D6321 CHANNEL  ; 进料伺服Z轴JOG运行速度SV
D6322 CHANNEL  ; 进料伺服Z轴JOG运行速度SV
D6331 CHANNEL  ; 进料伺服Z轴JOG停止速度SV
D6332 CHANNEL  ; 进料伺服Z轴JOG停止速度SV
D634 CHANNEL  ; #2-2腔体自检保压时间（S_UInt）
D6350 CHANNEL  ; 进料伺服Z轴待料位SV
D6351 CHANNEL  ; 进料伺服Z轴待料位SV
D6352 CHANNEL  ; 进料伺服Z轴取料位SV
D6353 CHANNEL  ; 进料伺服Z轴取料位SV
D6354 CHANNEL  ; 进料伺服Z轴#1腔放料位SV
D6355 CHANNEL  ; 进料伺服Z轴#1腔放料位SV
D6356 CHANNEL  ; 进料伺服Z轴#2腔放料位SV
D6357 CHANNEL  ; 进料伺服Z轴#2腔放料位SV
D6358 CHANNEL  ; 进料伺服Z轴#3腔放料位SV
D6359 CHANNEL  ; 进料伺服Z轴#3腔放料位SV
D636 CHANNEL  ; #2-2腔体自检保压前真空（Pa_Float）
D6360 CHANNEL  ; 进料伺服Z轴#1夹爪扫码NG放料位SV
D6361 CHANNEL  ; 进料伺服Z轴#1夹爪扫码NG放料位SV
D6362 CHANNEL  ; 进料伺服Z轴#2夹爪扫码NG放料位SV
D6363 CHANNEL  ; 进料伺服Z轴#2夹爪扫码NG放料位SV
D6364 CHANNEL  ; 进料伺服Z轴#1夹爪配对取放料位SV
D6365 CHANNEL  ; 进料伺服Z轴#1夹爪配对取放料位SV
D6366 CHANNEL  ; 进料伺服Z轴#2夹爪配对取放料位SV
D6367 CHANNEL  ; 进料伺服Z轴#2夹爪配对取放料位SV
D638 CHANNEL  ; #2-2腔体自检保压后真空（Pa_Float）
D640 CHANNEL  ; #2-2腔体自检泄漏量（Pa_Float）
D6400 CHANNEL  ; 出料伺服X轴加速比率
D6401 CHANNEL  ; 出料伺服X轴减速比率
D6402 CHANNEL  ; 出料伺服X轴目标速度
D6403 CHANNEL  ; 出料伺服X轴目标速度
D6404 CHANNEL  ; 出料伺服X轴目标位置
D6405 CHANNEL  ; 出料伺服X轴目标位置
D6406 CHANNEL  ; 出料伺服X轴启动频率
D6407 CHANNEL  ; 出料伺服X轴启动频率
D6410 CHANNEL  ; 出料伺服X轴自动加速比率SV
D6411 CHANNEL  ; 出料伺服X轴自动减速比率SV
D6412 CHANNEL  ; 出料伺服X轴自动目标速度SV
D6414 CHANNEL  ; 出料伺服X轴自动目标位置
D6416 CHANNEL  ; 出料伺服X轴自动启动频率
D642 CHANNEL  ; #2-2腔体自检结果（1-OK，2-NG,3-抽真空NG）
D6420 CHANNEL  ; 出料伺服X轴JOG运行加减速
D6421 CHANNEL  ; 出料伺服X轴JOG运行速度
D6422 CHANNEL  ; 出料伺服X轴JOG运行速度
D6430 CHANNEL  ; 出料伺服X轴JOG停止加减速
D6431 CHANNEL  ; 出料伺服X轴JOG停止速度
D6432 CHANNEL  ; 出料伺服X轴JOG停止速度
D6440 CHANNEL  ; 出料伺服X轴当前位置
D6441 CHANNEL  ; 出料伺服X轴当前位置
D6442 CHANNEL  ; 出料伺服X轴当前速度
D6443 CHANNEL  ; 出料伺服X轴当前速度
D6450 CHANNEL  ; 下料Z模组当前位置（CAENNEL）
D6500 CHANNEL  ; 出料伺服X轴加速比率SV
D6501 CHANNEL  ; 出料伺服X轴减速比率SV
D6502 CHANNEL  ; 出料伺服X轴目标速度SV
D6503 CHANNEL  ; 出料伺服X轴目标速度SV
D6504 CHANNEL  ; 出料伺服X轴目标位置（CHANNEL)
D6506 CHANNEL  ; 出料伺服X轴启动频率SV
D6507 CHANNEL  ; 出料伺服X轴启动频率SV
D6520 CHANNEL  ; 出料伺服X轴JOG运行/停止加减速SV
D6521 CHANNEL  ; 出料伺服X轴JOG运行速度SV
D6522 CHANNEL  ; 出料伺服X轴JOG运行速度SV
D6530 CHANNEL  ; 出料伺服X轴JOG停止加减速
D6531 CHANNEL  ; 出料伺服X轴JOG停止速度SV
D6532 CHANNEL  ; 出料伺服X轴JOG停止速度SV
D6540 CHANNEL  ; 出料伺服X轴当前位置（CAENNEL）
D6542 CHANNEL  ; 出料伺服X轴当前速度
D6544 CHANNEL  ; 出料伺服X轴当前位置（REAL）（mm）
D6550 CHANNEL  ; 出料伺服X轴出料OK位（设定）
D6552 CHANNEL  ; 出料伺服X轴放料位SV
D6553 CHANNEL  ; 出料伺服X轴放料位SV
D6554 CHANNEL  ; 出料伺服X轴#1腔取料位SV
D6555 CHANNEL  ; 出料伺服X轴#1腔取料位SV
D6556 CHANNEL  ; 出料伺服X轴#2腔取料位SV
D6557 CHANNEL  ; 出料伺服X轴#2腔取料位SV
D6558 CHANNEL  ; 出料伺服X轴#3腔取料位SV
D6559 CHANNEL  ; 出料伺服X轴#3腔取料位SV
D6560 CHANNEL  ; 出料伺服X轴#1夹爪氦检NG放料位SV
D6561 CHANNEL  ; 出料伺服X轴#1夹爪氦检NG放料位SV
D6562 CHANNEL  ; 出料伺服X轴#2夹爪氦检NG放料位SV
D6563 CHANNEL  ; 出料伺服X轴#2夹爪氦检NG放料位SV
D6564 CHANNEL  ; 出料伺服X轴#1夹爪配对取放料位SV
D6565 CHANNEL  ; 出料伺服X轴#1夹爪配对取放料位SV
D6566 CHANNEL  ; 出料伺服X轴#2夹爪配对取放料位SV
D6567 CHANNEL  ; 出料伺服X轴#2夹爪配对取放料位SV
D66 CHANNEL  ; 设定条码长度
D660 CHANNEL  ; #2-2氦检时真空值（标漏）
D6600 CHANNEL  ; 出料伺服Z轴加速比率
D6601 CHANNEL  ; 出料伺服Z轴减速比率
D6602 CHANNEL  ; 出料伺服Z轴目标速度
D6603 CHANNEL  ; 出料伺服Z轴目标速度
D6604 CHANNEL  ; 出料伺服Z轴目标位置
D6605 CHANNEL  ; 出料伺服Z轴目标位置
D6606 CHANNEL  ; 出料伺服Z轴启动频率
D6607 CHANNEL  ; 出料伺服Z轴启动频率
D6610 CHANNEL  ; 出料伺服Z轴自动加速比率SV
D6611 CHANNEL  ; 出料伺服Z轴自动减速比率SV
D6612 CHANNEL  ; 出料伺服Z轴自动目标速度SV
D6614 CHANNEL  ; 出料伺服Z轴自动目标位置
D6616 CHANNEL  ; 出料伺服Z轴自动启动频率
D662 CHANNEL  ; #2-2氦检漏率（标漏）
D6620 CHANNEL  ; 出料伺服Z轴JOG运行加减速
D6621 CHANNEL  ; 出料伺服Z轴JOG运行速度
D6622 CHANNEL  ; 出料伺服Z轴JOG运行速度
D6630 CHANNEL  ; 出料伺服Z轴JOG停止加减速
D6631 CHANNEL  ; 出料伺服Z轴JOG停止速度
D6632 CHANNEL  ; 出料伺服Z轴JOG停止速度
D6640 CHANNEL  ; 出料伺服Z轴当前位置
D6641 CHANNEL  ; 出料伺服Z轴当前位置
D6642 CHANNEL  ; 出料伺服Z轴当前速度
D6643 CHANNEL  ; 出料伺服Z轴当前速度
D6650 CHANNEL  ; 出料伺服X轴出料OK位
D6654 CHANNEL  ; 出料伺服Z轴#1腔取料位SV1
D6655 CHANNEL  ; 出料伺服Z轴#1腔取料位SV1
D6656 CHANNEL  ; 出料伺服Z轴#2腔取料位SV1
D6657 CHANNEL  ; 出料伺服Z轴#2腔取料位SV1
D6658 CHANNEL  ; 出料伺服Z轴#3腔取料位SV1
D6659 CHANNEL  ; 出料伺服Z轴#3腔取料位SV1
D6700 CHANNEL  ; 出料伺服Z轴加速比率SV
D6701 CHANNEL  ; 出料伺服Z轴减速比率SV
D6702 CHANNEL  ; 出料伺服Z轴目标速度SV
D6703 CHANNEL  ; 出料伺服Z轴目标速度SV
D6704 CHANNEL  ; 出料伺服Z轴目标位置(CHANNEL）
D6706 CHANNEL  ; 出料伺服Z轴启动频率SV
D6707 CHANNEL  ; 出料伺服Z轴启动频率SV
D6720 CHANNEL  ; 出料伺服Z轴JOG运行/停止加减速SV
D6721 CHANNEL  ; 出料伺服Z轴JOG运行速度SV
D6722 CHANNEL  ; 出料伺服Z轴JOG运行速度SV
D6730 CHANNEL  ; 出料伺服Z轴JOG停止加减速
D6731 CHANNEL  ; 出料伺服Z轴JOG停止速度SV
D6732 CHANNEL  ; 出料伺服Z轴JOG停止速度SV
D6742 CHANNEL  ; 出料伺服Z轴当前速度
D6750 CHANNEL  ; 出料伺服Z轴待料位SV
D6751 CHANNEL  ; 出料伺服Z轴待料位SV
D6752 CHANNEL  ; 出料伺服Z轴放料位SV
D6753 CHANNEL  ; 出料伺服Z轴放料位SV
D6754 CHANNEL  ; 出料伺服Z轴#1腔取料位SV
D6755 CHANNEL  ; 出料伺服Z轴#1腔取料位SV
D6756 CHANNEL  ; 出料伺服Z轴#2腔取料位SV
D6757 CHANNEL  ; 出料伺服Z轴#2腔取料位SV
D6758 CHANNEL  ; 出料伺服Z轴#3腔取料位SV
D6759 CHANNEL  ; 出料伺服Z轴#3腔取料位SV
D6760 CHANNEL  ; 出料伺服Z轴#1夹爪氦检NG放料位SV
D6761 CHANNEL  ; 出料伺服Z轴#1夹爪氦检NG放料位SV
D6762 CHANNEL  ; 出料伺服Z轴#2夹爪氦检NG放料位SV
D6763 CHANNEL  ; 出料伺服Z轴#2夹爪氦检NG放料位SV
D6764 CHANNEL  ; 出料伺服Z轴#1夹爪配对取放料位SV
D6765 CHANNEL  ; 出料伺服Z轴#1夹爪配对取放料位SV
D6766 CHANNEL  ; 出料伺服Z轴#2夹爪配对取放料位SV
D6767 CHANNEL  ; 出料伺服Z轴#2夹爪配对取放料位SV
D68 CHANNEL  ; 设定条码字长度
D70 CHANNEL  ; 设定条码批次号
D700 CHANNEL  ; #3-2腔体状态（0停用，1待料中，2测试中，3测试完成，4-清氦中）
D702 CHANNEL  ; #3-2腔体测试漏率（Pa.m3/s_Float）
D704 CHANNEL  ; #3-2腔体测试检漏口压力（Pa_Float）
D706 CHANNEL  ; #3-2电池充氦压力（Pa_Float）
D708 CHANNEL  ; #3-2腔体测试结果（1 OK，2腔体泄漏，3气密NG，4注氦超时，5氦检异常，6电池泄漏，7注氦NG，8氦嘴泄漏）
D710 CHANNEL  ; #3-2充氦嘴压力（Pa_Float）
D712 CHANNEL  ; #3-2腔体抽气时间（S_UInt）
D714 CHANNEL  ; #3-2腔体真空压力（Pa_Float）
D716 CHANNEL  ; #3-2电池抽气时间（S_UInt）
D718 CHANNEL  ; #3-2电池真空压力（Pa_Float）
D730 CHANNEL  ; #3-2腔体自检抽气时间（S_UInt）
D732 CHANNEL  ; #3-2腔体自检前保压时间（S_UInt）
D734 CHANNEL  ; #3-2腔体自检保压时间（S_UInt）
D736 CHANNEL  ; #3-2腔体自检保压前真空（Pa_Float）
D738 CHANNEL  ; #3-2腔体自检保压后真空（Pa_Float）
D740 CHANNEL  ; #3-2腔体自检泄漏量（Pa_Float）
D742 CHANNEL  ; #3-2腔体自检结果（1-OK，2-NG,3-抽真空NG）
D760 CHANNEL  ; #3-2氦检时真空值（标漏）
D762 CHANNEL  ; #3-2氦检漏率（标漏）
D80 CHANNEL  ; 进料#1扫码接收条码长度
D900 CHANNEL  ; #1-1电池真空偏值设定(Float)
D902 CHANNEL  ; #1-1电池实际真空值(Float)
D904 CHANNEL  ; #1-1电池真空模拟量读数(Int)
D906 CHANNEL  ; #1-1电池设定时间实际真空值(Float)
D908 CHANNEL  ; #1-2电池设定时间实际真空值(Float)
D910 CHANNEL  ; #1-2电池真空偏值设定(Float)
D912 CHANNEL  ; #1-2电池实际真空值(Float)
D914 CHANNEL  ; #1-2电池真空模拟量读数(Int)
D920 CHANNEL  ; #2-1电池真空偏值设定(Float)
D922 CHANNEL  ; #2-1电池实际真空值(Float)
D924 CHANNEL  ; #2-1电池真空模拟量读数(Int)
D926 CHANNEL  ; #2-1电池设定时间实际真空值(Float)
D928 CHANNEL  ; #2-2电池设定时间实际真空值(Float)
D930 CHANNEL  ; #2-2电池真空偏值设定(Float)
D932 CHANNEL  ; #2-2电池实际真空值(Float)
D934 CHANNEL  ; #2-2电池真空模拟量读数(Int)
D940 CHANNEL  ; #3-1电池真空偏值设定(Float)
D942 CHANNEL  ; #3-1电池实际真空值(Float)
D944 CHANNEL  ; #3-1电池真空模拟量读数(Int)
D946 CHANNEL  ; #3-1电池设定时间实际真空值(Float)
D948 CHANNEL  ; #3-2电池设定时间实际真空值(Float)
D950 CHANNEL  ; #3-2电池真空偏值设定(Float)
D952 CHANNEL  ; #3-2电池实际真空值(Float)
D954 CHANNEL  ; #3-2电池真空模拟量读数(Int)
D962 CHANNEL  ; #1腔体实际真空值(Float)
D964 CHANNEL  ; #1腔体真空模拟量读数(Int)
D968 CHANNEL  ; #1腔体读设定时间实际真空值(Float)
D972 CHANNEL  ; #2腔体实际真空值(Float)
D974 CHANNEL  ; #2腔体真空模拟量读数(Int)
D978 CHANNEL  ; #2腔体读设定时间真空值
D982 CHANNEL  ; #3腔体实际真空值(Float)
D984 CHANNEL  ; #3腔体真空模拟量读数(Int)
D988 CHANNEL  ; #3腔体读设定时间实际真空值(Float)
D990 CHANNEL  ; 实时漏率（Pa.m3/s_Float）
D992 CHANNEL  ; 实时检漏口压力（Pa_Float）
D994 CHANNEL  ; 泄漏率设定值（Pa.m3/s_Float）
D996 CHANNEL  ; 检漏口压力设定值（Pa_Float）
D998 CHANNEL  ; 清氦漏率设定值（Pa_Float）
E0_0 CHANNEL  ; PC&PLC通讯心跳检测
E0_10 CHANNEL  ; 进料拉带机构#1扫码MES入站就绪通知
E0_1000 CHANNEL  ; 进料#1扫码MES出站读取条码开始字
E0_104 CHANNEL  ; 工艺参数变更通知to pc
E0_1049 CHANNEL  ; 进料#1扫码MES出站读取条码结束字
E0_105 CHANNEL  ; 工艺变更确认
E0_1050 CHANNEL  ; 出料伺服机构#1夹爪MES出站生产数据开始字
E0_1099 CHANNEL  ; 出料伺服机构#1夹爪MES出站生产数据结束字
E0_11 CHANNEL  ; 进料拉带机构#2扫码MES入站就绪通知
E0_1100 CHANNEL  ; 进料#2扫码MES入站读取条码开始字
E0_1149 CHANNEL  ; 进料#2扫码MES入站读取条码结束字
E0_1150 CHANNEL  ; 出料伺服机构#2夹爪MES出站生产数据开始字
E0_1199 CHANNEL  ; 出料伺服机构#2夹爪MES出站生产数据结束字
E0_1.00 BOOL  ; 设备上电状态
E0_1.01 BOOL  ; 设备复位状态
E0_1.02 BOOL  ; 设备自动状态
E0_1.03 BOOL  ; 设备停止状态
E0_1.04 BOOL  ; 设备启动状态
E0_1.05 BOOL  ; 设备待料状态
E0_1.06 BOOL  ; 设备手动状态
E0_1.07 BOOL  ; 设备故障状态
E0_1.08 BOOL  ; 设备急停状态
E0_1.09 BOOL  ; 设备关电状态
E0_20 CHANNEL  ; 进料拉带机构#1扫码MES入站就绪确认
E0_2000 CHANNEL  ; 进料#1扫码MES入站读取条码开始字
E0_2049 CHANNEL  ; 进料#1扫码MES入站读取条码结束字
E0_2050 CHANNEL  ; 进料#2扫码MES入站读取条码开始字
E0_2099 CHANNEL  ; 进料#2扫码MES入站读取条码结束字
E0_21 CHANNEL  ; 进料拉带机构#2扫码MES入站就绪确认
E0_300 CHANNEL  ; 泄漏率设定值to pc（Pa.m3/s_Float)to pc
E0_302 CHANNEL  ; 检漏口压力设定值（Pa_Float）to pc
E0_304 CHANNEL  ; 腔体测试设定氦检时间（S_UInt）to pc
E0_306 CHANNEL  ; 腔体测试设定真空阈值（Pa_Float）to pc
E0_308 CHANNEL  ; 电池测试设定真空阈值（Pa_Float）to pc
E0_310 CHANNEL  ; 电池测试设定#1-1注氦压力（Pa_Float）to pc
E0_312 CHANNEL  ; 电池测试设定#1-1注氦压力（Pa_Float）to pc
E0_316 CHANNEL  ; 腔体测试设定抽真空时间上限（S_UInt）to pc
E0_318 CHANNEL  ; 电池测试设定抽真空时间上限（S_UInt）to pc
E0_320 CHANNEL  ; 腔体测试设定腔体预抽检测时间（S_UInt）to pc
E0_322 CHANNEL  ; 电池测试设定预抽检测压力（Pa_Float）to pc
E0_324 CHANNEL  ; 腔体测试设定清氦压力（Pa_Float）to pc
E0_326 CHANNEL  ; 清氦漏率设定值（Pa_Float）to pc
E0_328 CHANNEL  ; 清氦漏率设定值（Pa_Float）to pc
E0_349 CHANNEL  ; 出料伺服机构#1夹爪MES出站工艺参数结束字
E0_350 CHANNEL  ; 出料伺服机构#2夹爪MES出站工艺参数开始字
E0_399 CHANNEL  ; 出料伺服机构#2夹爪MES出站工艺参数结束字
E0_50 CHANNEL  ; 出料伺服机构#1夹爪MES出站就绪通知
E0_51 CHANNEL  ; 出料伺服机构#2夹爪MES出站就绪通知
E0_60 CHANNEL  ; 出料伺服机构#1夹爪MES出站就绪确认
E0_61 CHANNEL  ; 出料伺服机构#2夹爪MES出站就绪确认
E0_900 CHANNEL  ; 工站故障
E2_1000 CHANNEL  ; 进料#1扫码条码开始字（传递）
E2_1001 CHANNEL  ; 进料#1扫码条码开始字（传递）
E2_1030 CHANNEL  ; 进料#1扫码条码结束字（传递）
E2_1100 CHANNEL  ; 进料#2扫码条码开始字（传递）
E2_1130 CHANNEL  ; 进料#2扫码条码结束字（传递）
E2_1200 CHANNEL  ; #1进料位条码开始字（传递）
E2_1299 CHANNEL  ; #1进料位数据结束字（传递）
E2_1300 CHANNEL  ; #2进料位条码开始字（传递）
E2_1399 CHANNEL  ; #2进料位数据结束字（传递）
E2_1400 CHANNEL  ; #1进料夹爪条码开始字（传递）
E2_1499 CHANNEL  ; #1进料夹爪数据结束字（传递）
E2_1500 CHANNEL  ; #2进料夹爪条码开始字（传递）
E2_1599 CHANNEL  ; #2进料夹爪数据结束字（传递）
E2_1600 CHANNEL  ; 扫码OK缓存条码开始字（传递）
E2_1699 CHANNEL  ; 扫码OK缓存数据结束字（传递）
E2_1800 CHANNEL  ; #1-1氦检腔条码开始字（传递）
E2_1850 CHANNEL  ; #1-1氦检腔工位开始字（传递）
E2_1899 CHANNEL  ; #1-1氦检腔数据结束字（传递）
E2_1900 CHANNEL  ; #1-2氦检腔条码开始字（传递）
E2_1950 CHANNEL  ; #1-2氦检腔工位开始字（传递）
E2_1999 CHANNEL  ; #1-2氦检腔数据结束字（传递）
E2_2000 CHANNEL  ; #2-1氦检腔条码开始字（传递）
E2_2050 CHANNEL  ; #2-1氦检腔工位开始字（传递）
E2_2099 CHANNEL  ; #2-1氦检腔数据结束字（传递）
E2_2100 CHANNEL  ; #2-2氦检腔条码开始字（传递）
E2_2150 CHANNEL  ; #2-2氦检腔工位开始字（传递）
E2_2199 CHANNEL  ; #2-2氦检腔数据结束字（传递）
E2_2200 CHANNEL  ; #3-1氦检腔条码开始字（传递）
E2_2250 CHANNEL  ; #3-1氦检腔工位开始字（传递）
E2_2299 CHANNEL  ; #3-1氦检腔数据结束字（传递）
E2_2300 CHANNEL  ; #3-2氦检腔条码开始字（传递）
E2_2350 CHANNEL  ; #3-2氦检腔工位开始字（传递）
E2_2399 CHANNEL  ; #3-2氦检腔数据结束字（传递）
E2_2400 CHANNEL  ; #1出料夹爪条码开始字（传递）
E2_2450 CHANNEL  ; #1出料夹爪工位开始字（传递）
E2_2499 CHANNEL  ; #1出料夹爪数据结束字（传递）
E2_2500 CHANNEL  ; #2出料夹爪条码开始字（传递）
E2_2550 CHANNEL  ; #2出料夹爪工位开始字（传递）
E2_2599 CHANNEL  ; #2出料夹爪数据结束字（传递）
H100.00 BOOL  ; #1扫码阻挡气缸缩回位屏蔽
H100.01 BOOL  ; #1扫码阻挡气缸伸出位屏蔽
H100.02 BOOL  ; #1隔离气缸缩回位屏蔽
H100.03 BOOL  ; 0屏蔽
H100.04 BOOL  ; #2扫码阻挡气缸缩回位屏蔽
H100.05 BOOL  ; #2扫码阻挡气缸伸出位屏蔽
H100.06 BOOL  ; #2隔离气缸缩回位屏蔽
H100.07 BOOL  ; 0屏蔽
H100.08 BOOL  ; #1进料夹爪夹紧位屏蔽
H100.09 BOOL  ; #1进料夹爪松开位屏蔽
H100.10 BOOL  ; #2进料夹爪夹紧位屏蔽
H100.11 BOOL  ; #2进料夹爪松开位屏蔽
H100.12 BOOL  ; 进料夹爪变距气缸伸出位屏蔽
H100.13 BOOL  ; 进料夹爪变距气缸缩回位屏蔽
H100.14 BOOL  ; #1出料夹爪夹紧位屏蔽
H100.15 BOOL  ; #1出料夹爪松开位屏蔽
H101.00 BOOL  ; #2出料夹爪夹紧位屏蔽
H101.01 BOOL  ; #2出料夹爪松开位屏蔽
H101.02 BOOL  ; 出料夹爪变距气缸伸出位屏蔽
H101.03 BOOL  ; 出料夹爪变距气缸缩回位屏蔽
H101.04 BOOL  ; #1腔体平移一级气缸缩回位屏蔽
H101.05 BOOL  ; #1腔体平移一级气缸伸出位屏蔽
H101.06 BOOL  ; #1腔体平移二级气缸缩回位屏蔽
H101.07 BOOL  ; #1腔体平移二级气缸伸出位屏蔽
H101.08 BOOL  ; #1腔体顶伸气缸上升位屏蔽
H101.09 BOOL  ; #1腔体顶伸气缸下降位屏蔽
H101.10 BOOL  ; #1腔体氦检阀开到位屏蔽
H101.11 BOOL  ; #1腔体氦检阀关到位屏蔽
H101.12 BOOL  ; 0屏蔽
H101.13 BOOL  ; 0屏蔽
H101.14 BOOL  ; 0屏蔽
H101.15 BOOL  ; 0屏蔽
H102.00 BOOL  ; 0屏蔽
H102.01 BOOL  ; #2腔体平移一级气缸缩回位屏蔽
H102.02 BOOL  ; #2腔体平移一级气缸伸出位屏蔽
H102.03 BOOL  ; #2腔体平移二级气缸缩回位屏蔽
H102.04 BOOL  ; #2腔体平移二级气缸伸出位屏蔽
H102.05 BOOL  ; #2腔体顶伸气缸上升位屏蔽
H102.06 BOOL  ; #2腔体顶伸气缸下降位屏蔽
H102.07 BOOL  ; #2腔体氦检阀开到位屏蔽
H102.08 BOOL  ; #2腔体氦检阀关到位屏蔽
H102.09 BOOL  ; 0屏蔽
H102.10 BOOL  ; 0屏蔽
H102.11 BOOL  ; 0屏蔽
H102.12 BOOL  ; 0屏蔽
H102.13 BOOL  ; 0屏蔽
H102.14 BOOL  ; #3腔体平移一级气缸缩回位屏蔽
H102.15 BOOL  ; #3腔体平移一级气缸伸出位屏蔽
H103.00 BOOL  ; #3腔体平移二级气缸缩回位屏蔽
H103.01 BOOL  ; #3腔体平移二级气缸伸出位屏蔽
H103.02 BOOL  ; #3腔体顶伸气缸上升位屏蔽
H103.03 BOOL  ; #3腔体顶伸气缸下降位屏蔽
H103.04 BOOL  ; #3腔体氦检阀开到位屏蔽
H103.05 BOOL  ; #3腔体氦检阀关到位屏蔽
H103.06 BOOL  ; 氦检仪准备好了信号屏蔽
H103.07 BOOL  ; 氦检仪故障信号屏蔽
H103.08 BOOL  ; 0屏蔽
H103.09 BOOL  ; 0屏蔽
H103.10 BOOL  ; 0屏蔽
H103.11 BOOL  ; 进料伺服X轴准备好了信号屏蔽
H103.12 BOOL  ; 进料伺服X轴故障信号屏蔽
H103.13 BOOL  ; 进料伺服Z轴准备好了信号屏蔽
H103.14 BOOL  ; 进料伺服Z轴故障信号屏蔽
H103.15 BOOL  ; 0屏蔽
H104.00 BOOL  ; 出料伺服X轴准备好了信号屏蔽
H104.01 BOOL  ; 出料伺服X轴故障信号屏蔽
H104.02 BOOL  ; 出料伺服Z轴准备好了信号屏蔽
H104.03 BOOL  ; 出料伺服Z轴故障信号屏蔽
H104.04 BOOL  ; 0屏蔽
H104.05 BOOL  ; 腔体抽真空泵运行信号屏蔽
H104.06 BOOL  ; 腔体抽真空泵过载信号屏蔽
H104.07 BOOL  ; 氦检前置泵运行信号屏蔽
H104.08 BOOL  ; 氦检前置泵过载信号屏蔽
H104.09 BOOL  ; 启动按钮屏蔽
H104.10 BOOL  ; 停止按钮屏蔽
H104.11 BOOL  ; 复位按钮屏蔽
H104.12 BOOL  ; 急停按钮屏蔽
H104.13 BOOL  ; 手自动选择屏蔽
H104.14 BOOL  ; #1进料夹爪防下坠感应屏蔽
H104.15 BOOL  ; #2进料夹爪防下坠感应屏蔽
H105.00 BOOL  ; #1出料夹爪防下坠感应屏蔽
H105.01 BOOL  ; #2出料夹爪防下坠感应屏蔽
H105.02 BOOL  ; 0屏蔽
H105.03 BOOL  ; 进料对接输入屏蔽
H105.04 BOOL  ; 出料对接输入屏蔽
H105.05 BOOL  ; 0屏蔽
H105.06 BOOL  ; 0屏蔽
H105.07 BOOL  ; 设备总气压信号屏蔽
H105.08 BOOL  ; #1来料位有料感应屏蔽
H105.09 BOOL  ; #2来料位有料感应屏蔽
H105.10 BOOL  ; #1隔离位有料感应屏蔽
H105.11 BOOL  ; #2隔离位有料感应屏蔽
H105.12 BOOL  ; #1扫码位有料感应屏蔽
H105.13 BOOL  ; #2扫码位有料感应屏蔽
H105.14 BOOL  ; #1-1进料位有料感应屏蔽
H105.15 BOOL  ; #1-2进料位有料感应屏蔽
H106.00 BOOL  ; #2-1进料位有料感应屏蔽
H106.01 BOOL  ; #2-2进料位有料感应屏蔽
H106.02 BOOL  ; 进料夹爪柔性感应屏蔽
H106.03 BOOL  ; 出料夹爪柔性感应屏蔽
H106.04 BOOL  ; #1进料夹爪对应腔体有料感应屏蔽
H106.05 BOOL  ; #2进料夹爪对应腔体有料感应屏蔽
H106.06 BOOL  ; 扫码NG放料#1位有料感应屏蔽
H106.07 BOOL  ; 扫码NG放料#2位有料感应屏蔽
H106.08 BOOL  ; 扫码NG料满位有料感应屏蔽
H106.09 BOOL  ; 进料配对位有料感应屏蔽
H106.10 BOOL  ; 出料配对位有料感应屏蔽
H106.11 BOOL  ; 氦检NG放料#1位有料感应屏蔽
H106.12 BOOL  ; 氦检NG放料#2位有料感应屏蔽
H106.13 BOOL  ; 氦检NG料满位有料感应屏蔽
H106.14 BOOL  ; #1-1出料位有料感应屏蔽
H106.15 BOOL  ; #1-2出料位有料感应屏蔽
H107.00 BOOL  ; #2-1出料位有料感应屏蔽
H107.01 BOOL  ; #2-2出料位有料感应屏蔽
H107.02 BOOL  ; #1门磁开关屏蔽
H107.03 BOOL  ; #2门磁开关屏蔽
H107.04 BOOL  ; #3门磁开关屏蔽
H107.05 BOOL  ; #4门磁开关屏蔽
H107.06 BOOL  ; #5门磁开关屏蔽
H107.07 BOOL  ; #6门磁开关屏蔽
H107.08 BOOL  ; #7门磁开关屏蔽
H107.09 BOOL  ; #8门磁开关屏蔽
H107.10 BOOL  ; #9门磁开关屏蔽
H107.11 BOOL  ; #10门磁开关屏蔽
H107.12 BOOL  ; #11门磁开关屏蔽
H107.13 BOOL  ; 设备真空压力信号屏蔽
H107.14 BOOL  ; 设备氦气压力信号屏蔽
H107.15 BOOL  ; 精密调压阀信号屏蔽
H10.00 BOOL  ; #1扫码阻挡有料记忆
H10.01 BOOL  ; #1进料位有料记忆
H10.02 BOOL  ; #1进料位有OK料记忆
H10.03 BOOL  ; #1进料位有NG料记忆
H10.04 BOOL  ; #1扫码阻挡有OK料记忆
H10.05 BOOL  ; #1扫码阻挡有NG料记忆
H10.06 BOOL  ; #1扫码阻挡扫码完成记忆
H10.07 BOOL  ; #1扫码阻挡扫码OK料记忆
H10.08 BOOL  ; #1扫码阻挡扫码NG料记忆
H10.09 BOOL  ; #1扫码阻挡MES校验完成记忆
H10.10 BOOL  ; #1扫码阻挡MES校验OK料记忆
H10.11 BOOL  ; #1扫码阻挡MES校验NG料记忆
H11.00 BOOL  ; #1隔离气缸放料中记忆
H11.01 BOOL  ; #1扫码阻挡气缸放料中记忆
H12.00 BOOL  ; #2扫码阻挡有料记忆
H12.01 BOOL  ; #2进料位有料记忆
H12.02 BOOL  ; #2进料位有OK料记忆
H12.03 BOOL  ; #2进料位有NG料记忆
H12.04 BOOL  ; #2扫码阻挡有OK料记忆
H12.05 BOOL  ; #2扫码阻挡有NG料记忆
H12.06 BOOL  ; #2扫码阻挡扫码完成记忆
H12.07 BOOL  ; #2扫码阻挡扫码OK料记忆
H12.08 BOOL  ; #2扫码阻挡扫码NG料记忆
H12.09 BOOL  ; #2扫码阻挡MES校验完成记忆
H12.10 BOOL  ; #2扫码阻挡MES校验OK料记忆
H12.11 BOOL  ; #2扫码阻挡MES校验NG料记忆
H13.00 BOOL  ; #2隔离气缸放料中记忆
H13.01 BOOL  ; #2扫码阻挡气缸放料中记忆
H15.00 BOOL  ; 扫码NG放料位有料记忆
H17.00 BOOL  ; 氦检NG放料位有料记忆
H20.00 BOOL  ; #1进料夹爪有料记忆
H20.01 BOOL  ; #2进料夹爪有料记忆
H20.02 BOOL  ; 进料配对位有料记忆
H20.03 BOOL  ; #1进料夹爪有OK料记忆
H20.04 BOOL  ; #1进料夹爪有NG料记忆
H20.05 BOOL  ; #2进料夹爪有OK料记忆
H20.06 BOOL  ; #2进料夹爪有NG料记忆
H24.00 BOOL  ; 进料伺服X轴回原点记忆
H24.01 BOOL  ; 进料伺服Z轴回原点记Z忆
H24.02 BOOL  ; 出料伺服X轴回原点记忆
H24.03 BOOL  ; 出料伺服Z轴回原点记忆
H25.00 BOOL  ; #1-1腔体有料记忆
H25.01 BOOL  ; #1-2腔体有料记忆
H25.02 BOOL  ; #1-1腔体有OK料记忆
H25.03 BOOL  ; #1-1腔体有NG料记忆
H25.04 BOOL  ; #1-2腔体有OK料记忆
H25.05 BOOL  ; #1-2腔体有NG料记忆
H25.06 BOOL  ; #1-1腔体测试完成记忆
H25.07 BOOL  ; #1-2腔体测试完成记忆
H26.00 BOOL  ; #1-1电池泄漏
H26.01 BOOL  ; #1-2电池泄漏
H26.02 BOOL  ; #1-1电池注氦超时
H26.03 BOOL  ; #1-2电池注氦超时
H26.04 BOOL  ; #1-1腔体抽真空NG
H26.05 BOOL  ; #1-2腔体抽真空NG
H26.06 BOOL  ; #1-1腔体氦检时腔体压力过高
H26.07 BOOL  ; #1-2腔体氦检时腔体压力过高
H27.00 BOOL  ; #1腔体有清氦需求
H27.05 BOOL  ; 腔体有复测需求
H27.10 BOOL  ; #1-1腔体清氦失败，重新进行清氦流程
H30.00 BOOL  ; #2-1腔体有料记忆
H30.01 BOOL  ; #2-2腔体有料记忆
H30.02 BOOL  ; #2-1腔体有OK料记忆
H30.03 BOOL  ; #2-1腔体有NG料记忆
H30.04 BOOL  ; #2-2腔体有OK料记忆
H30.05 BOOL  ; #2-2腔体有NG料记忆
H30.06 BOOL  ; #2-1腔体测试完成记忆
H30.07 BOOL  ; #2-2腔体测试完成记忆
H31.00 BOOL  ; #2-1电池泄漏
H31.01 BOOL  ; #2-2电池泄漏
H31.02 BOOL  ; #2-1电池注氦超时
H31.03 BOOL  ; #2-2电池注氦超时
H31.04 BOOL  ; #2-1腔体抽真空NG
H31.05 BOOL  ; #2-2腔体抽真空NG
H31.06 BOOL  ; #2-1腔体氦检时腔体压力过高
H31.07 BOOL  ; #2-2腔体氦检时腔体压力过高
H32.00 BOOL  ; #2腔体有清氦需求
H32.05 BOOL  ; 腔体有复测需求
H32.10 BOOL  ; #2-1腔体清氦失败，重新进行清氦流程
H35.00 BOOL  ; #3-1腔体有料记忆
H35.01 BOOL  ; #3-2腔体有料记忆
H35.02 BOOL  ; #3-1腔体有OK料记忆
H35.03 BOOL  ; #3-1腔体有NG料记忆
H35.04 BOOL  ; #3-2腔体有OK料记忆
H35.05 BOOL  ; #3-2腔体有NG料记忆
H35.06 BOOL  ; #3-1腔体测试完成记忆
H35.07 BOOL  ; #3-2腔体测试完成记忆
H36.00 BOOL  ; #3-1电池泄漏
H36.01 BOOL  ; #3-2电池泄漏
H36.02 BOOL  ; #3-1电池注氦超时
H36.03 BOOL  ; #3-2电池注氦超时
H36.04 BOOL  ; #3-1腔体抽真空NG
H36.05 BOOL  ; #3-2腔体抽真空NG
H36.06 BOOL  ; #3-1腔体氦检时腔体压力过高
H36.07 BOOL  ; #3-2腔体氦检时腔体压力过高
H37.00 BOOL  ; #3腔体有清氦需求
H37.05 BOOL  ; 腔体有复测需求
H37.10 BOOL  ; #3-1腔体清氦失败，重新进行清氦流程
H40.00 BOOL  ; #1出料夹爪有料记忆
H40.01 BOOL  ; #2出料夹爪有料记忆
H40.02 BOOL  ; 出料配对位有料记忆
H40.03 BOOL  ; #1出料夹爪有OK料记忆
H40.04 BOOL  ; #1出料夹爪有NG料记忆
H40.05 BOOL  ; #2出料夹爪有OK料记忆
H40.06 BOOL  ; #2出料夹爪有NG料记忆
H40.07 BOOL  ; #1出料夹爪MES校验完成记忆
H40.08 BOOL  ; #2出料夹爪MES校验完成记忆
H40.15 BOOL  ; 出料变距缩回记忆
H41.00 BOOL  ; 1#取料完成
H41.01 BOOL  ; 2#取料完成
H41.02 BOOL  ; 3#取料完成
H41.03 BOOL  ; 1#放NG，2#放缓存
H41.04 BOOL  ; 1#放NG，1#取缓存
H41.05 BOOL  ; 2#放NG,1#放缓存
H41.06 BOOL  ; 2#放NG,2#取缓存
H43.00 BOOL  ; 1#腔体下料需求
H43.01 BOOL  ; 2#腔体下料需求
H43.02 BOOL  ; 3#腔体下料需求
H44.00 BOOL  ; 出料伺服X轴回原点记忆
H44.01 BOOL  ; 出料伺服Z轴回原点记忆
H5.00 BOOL  ; 扫码屏蔽（SW）
H5.01 BOOL  ; 进料拉带重新扫码模式选择（0=使用/1=屏蔽）
H5.02 BOOL  ; 氦检仪屏蔽
H5.03 BOOL  ; 1#腔体屏蔽（0=使用）
H5.04 BOOL  ; 2#腔体屏蔽（0=使用）
H5.05 BOOL  ; 3#腔体屏蔽（0=使用）
H5.07 BOOL  ; 电脑屏蔽-HMI
H5.08 BOOL  ; 门磁屏蔽(1-屏蔽)
H5.09 BOOL  ; 出料机械手放完NG料后回待料位（1-停用）
H5.10 BOOL  ; 空跑程序
H5.12 BOOL  ; 氦气源压力检测屏蔽
H5.13 BOOL  ; 复测模式（0-关闭 1-打开）
H5.14 BOOL  ; 测试模式（0-双检 1-单检）
H5.15 BOOL  ; 腔体模式（0-正压 1-负压）
H6.00 BOOL  ; 清氦模式（0-使用 1-不使用）
H6.01 BOOL  ; 氦气回收机使用（1-使用）
H6.06 BOOL  ; 出站MES校验使用（1-使用）
T0000 BOOL  ; PLC上电延时100ms
T0001 BOOL  ; 手动模式延时
T0002 BOOL  ; 自动模式延时
T0006 BOOL  ; 复位延时
T0007 BOOL  ; 自动停止完成延时
T0008 BOOL  ; 启动按钮按下1s延时
T0009 BOOL  ; 停止按钮按下延时
T0015 BOOL  ; 扫码NG取料延时
T0016 BOOL  ; 检测NG料满取料延时
T0019 BOOL  ; 清料停止完成延时
T0020 BOOL  ; 设备待料状态延时（参考进料）
T0021 BOOL  ; 设备待料状态延时（参考出料）
T0022 BOOL  ; 蜂鸣器屏蔽时间
T0024 BOOL  ; 氦检仪真空阀打开安全判定延时
T0030 BOOL  ; 腔体真空泵停机1分钟内禁止启动保护延时
T0031 BOOL  ; 氦检前置泵泵停机1分钟内禁止启动保护延时
T0045 BOOL  ; 进料#1扫码枪通信异常
T0046 BOOL  ; 进料#2扫码枪通信异常
T0047 BOOL  ; 氦检仪通信异常
T0048 BOOL  ; 氦检仪启动异常
T0049 BOOL  ; 初次上电氦检仪故障延时
T0050 BOOL  ; PC&PLC通讯心跳检测异常延时
T0062 BOOL  ; 进料伺服X轴故障报警延时
T0063 BOOL  ; 进料伺服Z轴故障报警延时
T0072 BOOL  ; 出料伺服X轴故障报警延时
T0073 BOOL  ; 出料伺服Z轴故障报警延时
T0075 BOOL  ; 1#腔体读真空设定时间
T0076 BOOL  ; 1-1电池读真空设定时间
T0077 BOOL  ; 1-2电池读真空设定时间
T0078 BOOL  ; 2#腔体读真空设定时间
T0079 BOOL  ; 2-1电池读真空设定时间
T0080 BOOL  ; 2-2电池读真空设定时间
T0081 BOOL  ; 3#腔体读真空设定时间
T0082 BOOL  ; 3-1电池读真空设定时间
T0083 BOOL  ; 3-2电池读真空设定时间
T0100 BOOL  ; #1扫码阻挡气缸缩回位报警延时
T0101 BOOL  ; #1扫码阻挡气缸伸出位报警延时
T0102 BOOL  ; #1隔离气缸缩回位报警延时
T0103 BOOL  ; 0报警延时
T0104 BOOL  ; #2扫码阻挡气缸缩回位报警延时
T0105 BOOL  ; #2扫码阻挡气缸伸出位报警延时
T0106 BOOL  ; #2隔离气缸缩回位报警延时
T0107 BOOL  ; 0报警延时
T0108 BOOL  ; #1进料夹爪夹紧位报警延时
T0109 BOOL  ; #1进料夹爪松开位报警延时
T0110 BOOL  ; #2进料夹爪夹紧位报警延时
T0111 BOOL  ; #2进料夹爪松开位报警延时
T0112 BOOL  ; 进料夹爪变距气缸伸出位报警延时
T0113 BOOL  ; 进料夹爪变距气缸缩回位报警延时
T0114 BOOL  ; #1出料夹爪夹紧位报警延时
T0115 BOOL  ; #1出料夹爪松开位报警延时
T0116 BOOL  ; #2出料夹爪夹紧位报警延时
T0117 BOOL  ; #2出料夹爪松开位报警延时
T0118 BOOL  ; 出料夹爪变距气缸伸出位报警延时
T0119 BOOL  ; 出料夹爪变距气缸缩回位报警延时
T0120 BOOL  ; #1腔体平移一级气缸缩回位报警延时
T0121 BOOL  ; #1腔体平移一级气缸伸出位报警延时
T0122 BOOL  ; #1腔体平移二级气缸缩回位报警延时
T0123 BOOL  ; #1腔体平移二级气缸伸出位报警延时
T0124 BOOL  ; #1腔体顶伸气缸上升位报警延时
T0125 BOOL  ; #1腔体顶伸气缸下降位报警延时
T0126 BOOL  ; #1腔体氦检阀开到位报警延时
T0127 BOOL  ; #1腔体氦检阀关到位报警延时
T0128 BOOL  ; 0报警延时
T0129 BOOL  ; 0报警延时
T0130 BOOL  ; 0报警延时
T0131 BOOL  ; 0报警延时
T0132 BOOL  ; 0报警延时
T0133 BOOL  ; #2腔体平移一级气缸缩回位报警延时
T0134 BOOL  ; #2腔体平移一级气缸伸出位报警延时
T0135 BOOL  ; #2腔体平移二级气缸缩回位报警延时
T0136 BOOL  ; #2腔体平移二级气缸伸出位报警延时
T0137 BOOL  ; #2腔体顶伸气缸上升位报警延时
T0138 BOOL  ; #2腔体顶伸气缸下降位报警延时
T0139 BOOL  ; #2腔体氦检阀开到位报警延时
T0140 BOOL  ; #2腔体氦检阀关到位报警延时
T0141 BOOL  ; 0报警延时
T0142 BOOL  ; 0报警延时
T0143 BOOL  ; 0报警延时
T0144 BOOL  ; 0报警延时
T0145 BOOL  ; 0报警延时
T0146 BOOL  ; #3腔体平移一级气缸缩回位报警延时
T0147 BOOL  ; #3腔体平移一级气缸伸出位报警延时
T0148 BOOL  ; #3腔体平移二级气缸缩回位报警延时
T0149 BOOL  ; #3腔体平移二级气缸伸出位报警延时
T0150 BOOL  ; #3腔体顶伸气缸上升位报警延时
T0151 BOOL  ; #3腔体顶伸气缸下降位报警延时
T0152 BOOL  ; #3腔体氦检阀开到位报警延时
T0153 BOOL  ; #3腔体氦检阀关到位报警延时
T0154 BOOL  ; 氦检仪准备好了信号报警延时
T0155 BOOL  ; 氦检仪故障信号报警延时
T0156 BOOL  ; 0报警延时
T0157 BOOL  ; 0报警延时
T0158 BOOL  ; 0报警延时
T0159 BOOL  ; 进料伺服X轴准备好了信号报警延时
T0160 BOOL  ; 进料伺服X轴故障信号报警延时
T0161 BOOL  ; 进料伺服Z轴准备好了信号报警延时
T0162 BOOL  ; 进料伺服Z轴故障信号报警延时
T0163 BOOL  ; 0报警延时
T0164 BOOL  ; 出料伺服X轴准备好了信号报警延时
T0165 BOOL  ; 出料伺服X轴故障信号报警延时
T0166 BOOL  ; 出料伺服Z轴准备好了信号报警延时
T0167 BOOL  ; 出料伺服Z轴故障信号报警延时
T0168 BOOL  ; 0报警延时
T0169 BOOL  ; 腔体抽真空泵运行信号报警延时
T0170 BOOL  ; 腔体抽真空泵过载信号报警延时
T0171 BOOL  ; 氦检前置泵运行信号报警延时
T0172 BOOL  ; 氦检前置泵过载信号报警延时
T0173 BOOL  ; 启动按钮报警延时
T0174 BOOL  ; 停止按钮报警延时
T0175 BOOL  ; 复位按钮报警延时
T0176 BOOL  ; 急停按钮报警延时
T0177 BOOL  ; 手自动选择报警延时
T0178 BOOL  ; #1进料夹爪防下坠感应报警延时
T0179 BOOL  ; #2进料夹爪防下坠感应报警延时
T0180 BOOL  ; #1出料夹爪防下坠感应报警延时
T0181 BOOL  ; #2出料夹爪防下坠感应报警延时
T0182 BOOL  ; 0报警延时
T0183 BOOL  ; 进料对接输入报警延时
T0184 BOOL  ; 出料对接输入报警延时
T0185 BOOL  ; 0报警延时
T0186 BOOL  ; 0报警延时
T0187 BOOL  ; 设备总气压信号报警延时
T0188 BOOL  ; #1来料位有料感应报警延时
T0189 BOOL  ; #2来料位有料感应报警延时
T0190 BOOL  ; #1隔离位有料感应报警延时
T0191 BOOL  ; #2隔离位有料感应报警延时
T0192 BOOL  ; #1扫码位有料感应报警延时
T0193 BOOL  ; #2扫码位有料感应报警延时
T0194 BOOL  ; #1-1进料位有料感应报警延时
T0195 BOOL  ; #1-2进料位有料感应报警延时
T0196 BOOL  ; #2-1进料位有料感应报警延时
T0197 BOOL  ; #2-2进料位有料感应报警延时
T0198 BOOL  ; 进料夹爪柔性感应报警延时
T0199 BOOL  ; 出料夹爪柔性感应报警延时
T0200 BOOL  ; #1进料夹爪对应腔体有料感应报警延时
T0201 BOOL  ; #2进料夹爪对应腔体有料感应报警延时
T0202 BOOL  ; 扫码NG放料#1位有料感应报警延时
T0203 BOOL  ; 扫码NG放料#2位有料感应报警延时
T0204 BOOL  ; 扫码NG料满位有料感应报警延时
T0205 BOOL  ; 进料配对位有料感应报警延时
T0206 BOOL  ; 出料配对位有料感应报警延时
T0207 BOOL  ; 氦检NG放料#1位有料感应报警延时
T0208 BOOL  ; 氦检NG放料#2位有料感应报警延时
T0209 BOOL  ; 氦检NG料满位有料感应报警延时
T0210 BOOL  ; #1-1出料位有料感应报警延时
T0211 BOOL  ; #1-2出料位有料感应报警延时
T0212 BOOL  ; #2-1出料位有料感应报警延时
T0213 BOOL  ; #2-2出料位有料感应报警延时
T0214 BOOL  ; #1门磁开关报警延时
T0215 BOOL  ; #2门磁开关报警延时
T0216 BOOL  ; #3门磁开关报警延时
T0217 BOOL  ; #4门磁开关报警延时
T0218 BOOL  ; #5门磁开关报警延时
T0219 BOOL  ; #6门磁开关报警延时
T0220 BOOL  ; #7门磁开关报警延时
T0221 BOOL  ; #8门磁开关报警延时
T0222 BOOL  ; #9门磁开关报警延时
T0223 BOOL  ; #10门磁开关报警延时
T0224 BOOL  ; #11门磁开关报警延时
T0225 BOOL  ; 设备真空压力信号报警延时
T0226 BOOL  ; 设备氦气压力信号报警延时
T0227 BOOL  ; 精密调压阀信号报警延时
T0280 BOOL  ; 进料扫码MES入站就绪通知&确认超时报警延时
T0281 BOOL  ; 出料伺服MES出站就绪通知&确认超时报警延时
T0308 BOOL  ; 进料伺服X轴正极限报警延时
T0309 BOOL  ; 进料伺服X轴负极限报警延时
T0310 BOOL  ; 进料伺服X轴原点报警延时
T0311 BOOL  ; 进料伺服Z轴正极限报警延时
T0312 BOOL  ; 进料伺服Z轴负极限报警延时
T0313 BOOL  ; 进料伺服Z轴原点报警延时
T0314 BOOL  ; 出料伺服X轴正极限报警延时
T0315 BOOL  ; 出料伺服X轴负极限报警延时
T0316 BOOL  ; 出料伺服X轴原点报警延时
T0317 BOOL  ; 出料伺服Z轴正极限报警延时
T0318 BOOL  ; 出料伺服Z轴负极限报警延时
T0319 BOOL  ; 出料伺服Z轴原点报警延时
T0324 BOOL  ; 氦检仪不在检漏状态[alm]
T0356 BOOL  ; #1来料位有料记忆报警延时
T0357 BOOL  ; #2来料位有料记忆报警延时
T0358 BOOL  ; #1隔离位有料记忆报警延时
T0359 BOOL  ; #2隔离位有料记忆报警延时
T0360 BOOL  ; #1扫码位有料记忆报警延时
T0361 BOOL  ; #2扫码位有料记忆报警延时
T0362 BOOL  ; #1进料位有料记忆报警延时
T0363 BOOL  ; #2进料位有料记忆报警延时
T0364 BOOL  ; #1进料夹爪有料记忆报警延时
T0365 BOOL  ; #2进料夹爪有料记忆报警延时
T0366 BOOL  ; #1出料夹爪有料记忆报警延时
T0367 BOOL  ; #2出料夹爪有料记忆报警延时
T0368 BOOL  ; #1-1腔体有料记忆报警延时
T0369 BOOL  ; #1-2腔体有料记忆报警延时
T0370 BOOL  ; #2-1腔体有料记忆报警延时
T0371 BOOL  ; #2-2腔体有料记忆报警延时
T0372 BOOL  ; #3-1腔体有料记忆报警延时
T0373 BOOL  ; #3-2腔体有料记忆报警延时
T0374 BOOL  ; 进料配对位有料记忆报警延时
T0375 BOOL  ; 出料配对位有料记忆报警延时
T0376 BOOL  ; #1出料位有料记忆报警延时
T0377 BOOL  ; #2出料位有料记忆报警延时
T0378 BOOL  ; 扫码NG放料位有料记忆报警延时
T0379 BOOL  ; 氦检NG拉带下料位有料记忆报警延时
T0388 BOOL  ; 整机复位超时报警延时
T0389 BOOL  ; 进料拉带工站复位超时报警延时
T0390 BOOL  ; 进料伺服工站复位超时报警延时
T0391 BOOL  ; #1氦检工站复位超时报警延时
T0392 BOOL  ; #2氦检工站复位超时报警延时
T0393 BOOL  ; #3氦检工站复位超时报警延时
T0394 BOOL  ; 出料伺服工站复位超时报警延时
T0400 BOOL  ; 开#1电池破真空法条件
T0401 BOOL  ; 开#2电池破真空法条件
T0402 BOOL  ; 开#3电池破真空法条件
T0500 BOOL  ; #1扫码阻挡气缸缩回延时[A]
T0501 BOOL  ; #1扫码阻挡气缸伸出延时[A]
T0502 BOOL  ; #1隔离气缸缩回延时[A]
T0503 BOOL  ; #1隔离气缸伸出延时[A]
T0504 BOOL  ; #2扫码阻挡气缸缩回延时[A]
T0505 BOOL  ; #2扫码阻挡气缸伸出延时[A]
T0506 BOOL  ; #2隔离气缸缩回延时[A]
T0507 BOOL  ; #2隔离气缸伸出延时[A]
T0508 BOOL  ; #1进料夹爪夹紧延时[A]
T0509 BOOL  ; #1进料夹爪松开延时[A]
T0510 BOOL  ; #2进料夹爪夹紧延时[A]
T0511 BOOL  ; #2进料夹爪松开延时[A]
T0512 BOOL  ; 进料夹爪变距气缸伸出延时[A]
T0513 BOOL  ; 进料夹爪变距气缸缩回延时[A]
T0514 BOOL  ; #1出料夹爪夹紧延时[A]
T0515 BOOL  ; #1出料夹爪松开延时[A]
T0516 BOOL  ; #2出料夹爪夹紧延时[A]
T0517 BOOL  ; #2出料夹爪松开延时[A]
T0518 BOOL  ; 出料夹爪变距气缸伸出延时[A]
T0519 BOOL  ; 出料夹爪变距气缸缩回延时[A]
T0520 BOOL  ; #1腔体平移一级气缸缩回延时[A]
T0521 BOOL  ; #1腔体平移一级气缸伸出延时[A]
T0522 BOOL  ; #1腔体平移二级气缸缩回延时[A]
T0523 BOOL  ; #1腔体平移二级气缸伸出延时[A]
T0524 BOOL  ; #1腔体顶伸气缸上升延时[A]
T0525 BOOL  ; #1腔体顶伸气缸下降延时[A]
T0526 BOOL  ; #1腔体氦检阀开延时[A]
T0527 BOOL  ; 氦检仪真空阀开延时[A]
T0528 BOOL  ; #1腔体抽真空阀开延时[A]
T0529 BOOL  ; #1-1腔体阀开延时[A]
T0530 BOOL  ; #1-2腔体阀开延时[A]
T0531 BOOL  ; #1腔体破真空阀开延时[A]
T0532 BOOL  ; #1腔体吹气阀开延时[A]
T0533 BOOL  ; #2腔体平移一级气缸缩回延时[A]
T0534 BOOL  ; #2腔体平移一级气缸伸出延时[A]
T0535 BOOL  ; #2腔体平移二级气缸缩回延时[A]
T0536 BOOL  ; #2腔体平移二级气缸伸出延时[A]
T0537 BOOL  ; #2腔体顶伸气缸上升延时[A]
T0538 BOOL  ; #2腔体顶伸气缸下降延时[A]
T0539 BOOL  ; #2腔体氦检阀开延时[A]
T0540 BOOL  ; 复检清洁阀开延时[A]
T0541 BOOL  ; #2腔体抽真空阀开延时[A]
T0542 BOOL  ; #2-1腔体阀开延时[A]
T0543 BOOL  ; #2-2腔体阀开延时[A]
T0544 BOOL  ; #2腔体破真空阀开延时[A]
T0545 BOOL  ; #2腔体吹气阀开延时[A]
T0546 BOOL  ; #3腔体平移一级气缸缩回延时[A]
T0547 BOOL  ; #3腔体平移一级气缸伸出延时[A]
T0548 BOOL  ; #3腔体平移二级气缸缩回延时[A]
T0549 BOOL  ; #3腔体平移二级气缸伸出延时[A]
T0550 BOOL  ; #3腔体顶伸气缸上升延时[A]
T0551 BOOL  ; #3腔体顶伸气缸下降延时[A]
T0552 BOOL  ; #3腔体氦检阀开延时[A]
T0553 BOOL  ; 0延时[A]
T0554 BOOL  ; #3腔体抽真空阀开延时[A]
T0555 BOOL  ; #3-1腔体阀开延时[A]
T0556 BOOL  ; #3-2腔体阀开延时[A]
T0557 BOOL  ; #3腔体破真空阀开延时[A]
T0558 BOOL  ; #3腔体吹气阀开延时[A]
T0559 BOOL  ; 进料伺服X轴使能延时[A]
T0560 BOOL  ; 进料伺服X轴故障复位延时[A]
T0561 BOOL  ; 进料伺服Z轴使能延时[A]
T0562 BOOL  ; 进料伺服Z轴故障复位延时[A]
T0563 BOOL  ; 进料伺服Z轴刹车延时[A]
T0564 BOOL  ; 出料伺服X轴使能延时[A]
T0565 BOOL  ; 出料伺服X轴故障复位延时[A]
T0566 BOOL  ; 出料伺服Z轴使能延时[A]
T0567 BOOL  ; 出料伺服Z轴故障复位延时[A]
T0568 BOOL  ; 出料伺服Z轴刹车延时[A]
T0569 BOOL  ; 腔体抽真空泵启动延时[A]
T0570 BOOL  ; 0延时[A]
T0571 BOOL  ; 氦检前置泵启动延时[A]
T0572 BOOL  ; 氦检仪供电延时[A]
T0573 BOOL  ; 启动按钮指示灯延时[A]
T0574 BOOL  ; 停止按钮指示灯延时[A]
T0575 BOOL  ; 复位按钮指示灯延时[A]
T0576 BOOL  ; 蜂鸣器延时[A]
T0577 BOOL  ; 三色灯（红）延时[A]
T0578 BOOL  ; 三色灯（绿）延时[A]
T0579 BOOL  ; 三色灯（黄）延时[A]
T0580 BOOL  ; 进料拉带电机启动延时[A]
T0581 BOOL  ; 扫码NG拉带电机启动延时[A]
T0582 BOOL  ; 氦检NG拉带电机启动延时[A]
T0583 BOOL  ; 进料对接输出延时[A]
T0584 BOOL  ; 出料对接输出延时[A]
T0585 BOOL  ; 0延时[A]
T0586 BOOL  ; 0延时[A]
T0587 BOOL  ; 0延时[A]
T0588 BOOL  ; 0延时[A]
T0589 BOOL  ; 0延时[A]
T0590 BOOL  ; 0延时[A]
T0591 BOOL  ; 0延时[A]
T0592 BOOL  ; 0延时[A]
T0593 BOOL  ; 0延时[A]
T0594 BOOL  ; 0延时[A]
T0595 BOOL  ; 0延时[A]
T0596 BOOL  ; #1-1电池抽真空阀开延时[A]
T0597 BOOL  ; #1-2电池抽真空阀开延时[A]
T0598 BOOL  ; #1-1电池注氦阀开延时[A]
T0599 BOOL  ; #1-2电池注氦阀开延时[A]
T0600 BOOL  ; #1-1电池破真空阀开延时[A]
T0601 BOOL  ; #1-2电池破真空阀开延时[A]
T0602 BOOL  ; #2-1电池抽真空阀开延时[A]
T0603 BOOL  ; #2-2电池抽真空阀开延时[A]
T0604 BOOL  ; #2-1电池注氦阀开延时[A]
T0605 BOOL  ; #2-2电池注氦阀开延时[A]
T0606 BOOL  ; #2-1电池破真空阀开延时[A]
T0607 BOOL  ; #2-2电池破真空阀开延时[A]
T0608 BOOL  ; #3-1电池抽真空阀开延时[A]
T0609 BOOL  ; #3-2电池抽真空阀开延时[A]
T0610 BOOL  ; #3-1电池注氦阀开延时[A]
T0611 BOOL  ; #3-2电池注氦阀开延时[A]
T0612 BOOL  ; #3-1电池破真空阀开延时[A]
T0613 BOOL  ; #3-2电池破真空阀开延时[A]
T0614 BOOL  ; 0延时[A]
T0615 BOOL  ; 0延时[A]
T0616 BOOL  ; 0延时[A]
T0617 BOOL  ; 0延时[A]
T0618 BOOL  ; 0延时[A]
T0619 BOOL  ; 0延时[A]
T0620 BOOL  ; 0延时[A]
T0621 BOOL  ; 0延时[A]
T0622 BOOL  ; 0延时[A]
T0623 BOOL  ; 0延时[A]
T0624 BOOL  ; 0延时[A]
T0625 BOOL  ; 0延时[A]
T0626 BOOL  ; 0延时[A]
T0627 BOOL  ; 0延时[A]
T0630 BOOL  ; #1扫码位有料延时
T0631 BOOL  ; #2扫码位有料延时
T0686 BOOL  ; #1腔体氦检阀关延时[A]
T0687 BOOL  ; 氦检仪真空阀关延时[A]
T0688 BOOL  ; #1腔体抽真空阀关延时[A]
T0689 BOOL  ; #1-1腔体阀关延时[A]
T0690 BOOL  ; #1-2腔体阀关延时[A]
T0691 BOOL  ; #1腔体破真空阀关延时[A]
T0692 BOOL  ; #1腔体吹气阀关延时[A]
T0693 BOOL  ; 延时[A]
T0694 BOOL  ; 延时[A]
T0695 BOOL  ; 延时[A]
T0696 BOOL  ; 延时[A]
T0697 BOOL  ; 延时[A]
T0698 BOOL  ; 延时[A]
T0699 BOOL  ; #2腔体氦检阀关延时[A]
T0700 BOOL  ; 复检清洁阀关延时[A]
T0701 BOOL  ; #2腔体抽真空阀关延时[A]
T0702 BOOL  ; #2-1腔体阀关延时[A]
T0703 BOOL  ; #2-2腔体阀关延时[A]
T0704 BOOL  ; #2腔体破真空阀关延时[A]
T0705 BOOL  ; #2腔体吹气阀关延时[A]
T0706 BOOL  ; 0延时[A]
T0707 BOOL  ; 延时[A]
T0708 BOOL  ; 延时[A]
T0709 BOOL  ; 延时[A]
T0710 BOOL  ; 延时[A]
T0711 BOOL  ; 延时[A]
T0712 BOOL  ; #3腔体氦检阀关延时[A]
T0713 BOOL  ; 0延时[A]
T0714 BOOL  ; #3腔体抽真空阀关延时[A]
T0715 BOOL  ; #3-1腔体阀关延时[A]
T0716 BOOL  ; #3-2腔体阀关延时[A]
T0717 BOOL  ; #3腔体破真空阀关延时[A]
T0718 BOOL  ; #3腔体吹气阀关延时[A]
T0719 BOOL  ; 延时[A]
T0720 BOOL  ; 延时[A]
T0721 BOOL  ; 延时[A]
T0722 BOOL  ; 延时[A]
T0723 BOOL  ; 延时[A]
T0724 BOOL  ; 延时[A]
T0725 BOOL  ; 延时[A]
T0726 BOOL  ; 延时[A]
T0727 BOOL  ; 延时[A]
T0728 BOOL  ; 延时[A]
T0729 BOOL  ; 腔体抽真空泵停止延时[A]
T0730 BOOL  ; 0延时[A]
T0731 BOOL  ; 氦检前置泵停止延时[A]
T0732 BOOL  ; 氦检仪停电延时[A]
T0733 BOOL  ; 延时[A]
T0734 BOOL  ; 延时[A]
T0735 BOOL  ; 延时[A]
T0736 BOOL  ; 延时[A]
T0737 BOOL  ; 延时[A]
T0738 BOOL  ; 延时[A]
T0739 BOOL  ; 延时[A]
T0740 BOOL  ; 进料拉带电机停止延时[A]
T0741 BOOL  ; 扫码NG拉带电机停止延时[A]
T0742 BOOL  ; 氦检NG拉带电机停止延时[A]
T0743 BOOL  ; 0延时[A]
T0744 BOOL  ; 延时[A]
T0745 BOOL  ; 延时[A]
T0746 BOOL  ; 延时[A]
T0747 BOOL  ; 延时[A]
T0748 BOOL  ; 延时[A]
T0749 BOOL  ; 延时[A]
T0750 BOOL  ; 延时[A]
T0751 BOOL  ; 延时[A]
T0752 BOOL  ; 延时[A]
T0753 BOOL  ; 延时[A]
T0754 BOOL  ; 延时[A]
T0755 BOOL  ; 延时[A]
T0756 BOOL  ; #1-1电池抽真空阀关延时[A]
T0757 BOOL  ; #1-2电池抽真空阀关延时[A]
T0758 BOOL  ; #1-1电池注氦阀关延时[A]
T0759 BOOL  ; #1-2电池注氦阀关延时[A]
T0760 BOOL  ; #1-1电池破真空阀关延时[A]
T0761 BOOL  ; #1-2电池破真空阀关延时[A]
T0762 BOOL  ; #2-1电池抽真空阀关延时[A]
T0763 BOOL  ; #2-2电池抽真空阀关延时[A]
T0764 BOOL  ; #2-1电池注氦阀关延时[A]
T0765 BOOL  ; #2-2电池注氦阀关延时[A]
T0766 BOOL  ; #2-1电池破真空阀关延时[A]
T0767 BOOL  ; #2-2电池破真空阀关延时[A]
T0768 BOOL  ; #3-1电池抽真空阀关延时[A]
T0769 BOOL  ; #3-2电池抽真空阀关延时[A]
T0770 BOOL  ; #3-1电池注氦阀关延时[A]
T0771 BOOL  ; #3-2电池注氦阀关延时[A]
T0772 BOOL  ; #3-1电池破真空阀关延时[A]
T0773 BOOL  ; #3-2电池破真空阀关延时[A]
T0774 BOOL  ; 延时[A]
T0775 BOOL  ; 延时[A]
T0776 BOOL  ; 延时[A]
T0777 BOOL  ; 延时[A]
T0778 BOOL  ; 延时[A]
T0779 BOOL  ; 延时[A]
T0780 BOOL  ; 延时[A]
T0781 BOOL  ; 延时[A]
T0782 BOOL  ; 延时[A]
T0783 BOOL  ; 延时[A]
T0784 BOOL  ; 延时[A]
T0785 BOOL  ; 延时[A]
T0786 BOOL  ; 延时[A]
T0787 BOOL  ; 延时[A]
T1000 BOOL  ; #1扫码阻挡气缸缩回位感应延时[0000.00]
T1001 BOOL  ; #1扫码阻挡气缸伸出位感应延时[0000.01]
T1002 BOOL  ; #1隔离气缸缩回位感应延时[0000.02]
T1003 BOOL  ; 0感应延时[0000.03]
T1004 BOOL  ; #2扫码阻挡气缸缩回位感应延时[0000.04]
T1005 BOOL  ; #2扫码阻挡气缸伸出位感应延时[0000.05]
T1006 BOOL  ; #2隔离气缸缩回位感应延时[0000.06]
T1007 BOOL  ; 0感应延时[0000.07]
T1008 BOOL  ; #1进料夹爪夹紧位感应延时[0000.08]
T1009 BOOL  ; #1进料夹爪松开位感应延时[0000.09]
T1010 BOOL  ; #2进料夹爪夹紧位感应延时[0000.10]
T1011 BOOL  ; #2进料夹爪松开位感应延时[0000.11]
T1012 BOOL  ; 进料夹爪变距气缸伸出位感应延时[0000.12]
T1013 BOOL  ; 进料夹爪变距气缸缩回位感应延时[0000.13]
T1014 BOOL  ; #1出料夹爪夹紧位感应延时[0000.14]
T1015 BOOL  ; #1出料夹爪松开位感应延时[0000.15]
T1016 BOOL  ; #2出料夹爪夹紧位感应延时[0001.00]
T1017 BOOL  ; #2出料夹爪松开位感应延时[0001.01]
T1018 BOOL  ; 出料夹爪变距气缸伸出位感应延时[0001.02]
T1019 BOOL  ; 出料夹爪变距气缸缩回位感应延时[0001.03]
T1020 BOOL  ; #1腔体平移一级气缸缩回位感应延时[0001.04]
T1021 BOOL  ; #1腔体平移一级气缸伸出位感应延时[0001.05]
T1022 BOOL  ; #1腔体平移二级气缸缩回位感应延时[0001.06]
T1023 BOOL  ; #1腔体平移二级气缸伸出位感应延时[0001.07]
T1024 BOOL  ; #1腔体顶伸气缸上升位感应延时[0001.08]
T1025 BOOL  ; #1腔体顶伸气缸下降位感应延时[0001.09]
T1026 BOOL  ; #1腔体氦检阀开到位感应延时[0001.10]
T1027 BOOL  ; #1腔体氦检阀关到位感应延时[0001.11]
T1028 BOOL  ; 0感应延时[0001.12]
T1029 BOOL  ; 0感应延时[0001.13]
T1030 BOOL  ; 0感应延时[0001.14]
T1031 BOOL  ; 0感应延时[0001.15]
T1032 BOOL  ; 0感应延时[0002.00]
T1033 BOOL  ; #2腔体平移一级气缸缩回位感应延时[0002.01]
T1034 BOOL  ; #2腔体平移一级气缸伸出位感应延时[0002.02]
T1035 BOOL  ; #2腔体平移二级气缸缩回位感应延时[0002.03]
T1036 BOOL  ; #2腔体平移二级气缸伸出位感应延时[0002.04]
T1037 BOOL  ; #2腔体顶伸气缸上升位感应延时[0002.05]
T1038 BOOL  ; #2腔体顶伸气缸下降位感应延时[0002.06]
T1039 BOOL  ; #2腔体氦检阀开到位感应延时[0002.07]
T1040 BOOL  ; #2腔体氦检阀关到位感应延时[0002.08]
T1041 BOOL  ; 0感应延时[0002.09]
T1042 BOOL  ; 0感应延时[0002.10]
T1043 BOOL  ; 0感应延时[0002.11]
T1044 BOOL  ; 0感应延时[0002.12]
T1045 BOOL  ; 0感应延时[0002.13]
T1046 BOOL  ; #3腔体平移一级气缸缩回位感应延时[0002.14]
T1047 BOOL  ; #3腔体平移一级气缸伸出位感应延时[0002.15]
T1048 BOOL  ; #3腔体平移二级气缸缩回位感应延时[0003.00]
T1049 BOOL  ; #3腔体平移二级气缸伸出位感应延时[0003.01]
T1050 BOOL  ; #3腔体顶伸气缸上升位感应延时[0003.02]
T1051 BOOL  ; #3腔体顶伸气缸下降位感应延时[0003.03]
T1052 BOOL  ; #3腔体氦检阀开到位感应延时[0003.04]
T1053 BOOL  ; #3腔体氦检阀关到位感应延时[0003.05]
T1054 BOOL  ; 氦检仪准备好了信号感应延时[0003.06]
T1055 BOOL  ; 氦检仪故障信号感应延时[0003.07]
T1056 BOOL  ; 0感应延时[0003.08]
T1057 BOOL  ; 0感应延时[0003.09]
T1058 BOOL  ; 0感应延时[0003.10]
T1059 BOOL  ; 进料伺服X轴准备好了信号感应延时[0003.11]
T1060 BOOL  ; 进料伺服X轴故障信号感应延时[0003.12]
T1061 BOOL  ; 进料伺服Z轴准备好了信号感应延时[0003.13]
T1062 BOOL  ; 进料伺服Z轴故障信号感应延时[0003.14]
T1063 BOOL  ; 0感应延时[0003.15]
T1064 BOOL  ; 出料伺服X轴准备好了信号感应延时[0004.00]
T1065 BOOL  ; 出料伺服X轴故障信号感应延时[0004.01]
T1066 BOOL  ; 出料伺服Z轴准备好了信号感应延时[0004.02]
T1067 BOOL  ; 出料伺服Z轴故障信号感应延时[0004.03]
T1068 BOOL  ; 0感应延时[0004.04]
T1069 BOOL  ; 腔体抽真空泵运行信号感应延时[0004.05]
T1070 BOOL  ; 腔体抽真空泵过载信号感应延时[0004.06]
T1071 BOOL  ; 氦检前置泵运行信号感应延时[0004.07]
T1072 BOOL  ; 氦检前置泵过载信号感应延时[0004.08]
T1073 BOOL  ; 启动按钮感应延时[0004.09]
T1074 BOOL  ; 停止按钮感应延时[0004.10]
T1075 BOOL  ; 复位按钮感应延时[0004.11]
T1076 BOOL  ; 急停按钮感应延时[0004.12]
T1077 BOOL  ; 手自动选择感应延时[0004.13]
T1078 BOOL  ; #1进料夹爪防下坠感应感应延时[0004.14]
T1079 BOOL  ; #2进料夹爪防下坠感应感应延时[0004.15]
T1080 BOOL  ; #1出料夹爪防下坠感应感应延时[0005.00]
T1081 BOOL  ; #2出料夹爪防下坠感应感应延时[0005.01]
T1082 BOOL  ; 0感应延时[0005.02]
T1083 BOOL  ; 进料对接输入感应延时[0005.03]
T1084 BOOL  ; 出料对接输入感应延时[0005.04]
T1085 BOOL  ; 0感应延时[0005.05]
T1086 BOOL  ; 0感应延时[0005.06]
T1087 BOOL  ; 设备总气压信号感应延时[0005.07]
T1088 BOOL  ; #1来料位有料感应感应延时[0005.08]
T1089 BOOL  ; #2来料位有料感应感应延时[0005.09]
T1090 BOOL  ; #1隔离位有料感应感应延时[0005.10]
T1091 BOOL  ; #2隔离位有料感应感应延时[0005.11]
T1092 BOOL  ; #1扫码位有料感应感应延时[0005.12]
T1093 BOOL  ; #2扫码位有料感应感应延时[0005.13]
T1094 BOOL  ; #1-1进料位有料感应感应延时[0005.14]
T1095 BOOL  ; #1-2进料位有料感应感应延时[0005.15]
T1096 BOOL  ; #2-1进料位有料感应感应延时[0006.00]
T1097 BOOL  ; #2-2进料位有料感应感应延时[0006.01]
T1098 BOOL  ; 进料夹爪柔性感应感应延时[0006.02]
T1099 BOOL  ; 出料夹爪柔性感应感应延时[0006.03]
T1100 BOOL  ; #1进料夹爪对应腔体有料感应感应延时[0006.04]
T1101 BOOL  ; #2进料夹爪对应腔体有料感应感应延时[0006.05]
T1102 BOOL  ; 扫码NG放料#1位有料感应感应延时[0006.06]
T1103 BOOL  ; 扫码NG放料#2位有料感应感应延时[0006.07]
T1104 BOOL  ; 扫码NG料满位有料感应感应延时[0006.08]
T1105 BOOL  ; 进料配对位有料感应感应延时[0006.09]
T1106 BOOL  ; 出料配对位有料感应感应延时[0006.10]
T1107 BOOL  ; 氦检NG放料#1位有料感应感应延时[0006.11]
T1108 BOOL  ; 氦检NG放料#2位有料感应感应延时[0006.12]
T1109 BOOL  ; 氦检NG料满位有料感应感应延时[0006.13]
T1110 BOOL  ; #1-1出料位有料感应感应延时[0006.14]
T1111 BOOL  ; #1-2出料位有料感应感应延时[0006.15]
T1112 BOOL  ; #2-1出料位有料感应感应延时[0007.00]
T1113 BOOL  ; #2-2出料位有料感应感应延时[0007.01]
T1114 BOOL  ; #1门磁开关感应延时[0007.02]
T1115 BOOL  ; #2门磁开关感应延时[0007.03]
T1116 BOOL  ; #3门磁开关感应延时[0007.04]
T1117 BOOL  ; #4门磁开关感应延时[0007.05]
T1118 BOOL  ; #5门磁开关感应延时[0007.06]
T1119 BOOL  ; #6门磁开关感应延时[0007.07]
T1120 BOOL  ; #7门磁开关感应延时[0007.08]
T1121 BOOL  ; #8门磁开关感应延时[0007.09]
T1122 BOOL  ; #9门磁开关感应延时[0007.10]
T1123 BOOL  ; #10门磁开关感应延时[0007.11]
T1124 BOOL  ; #11门磁开关感应延时[0007.12]
T1125 BOOL  ; 设备真空压力信号感应延时[0007.13]
T1126 BOOL  ; 设备氦气压力信号感应延时[0007.14]
T1127 BOOL  ; 精密调压阀信号感应延时[0007.15]
T1163 BOOL  ; $?St$Bk?_#[114] / #1隔离气缸伸出位感应延时 / $?St$Bk?_#[114]
T1167 BOOL  ; $?St$Bk?_#[115] / #2隔离气缸伸出位感应延时 / $?St$Bk?_#[115]
T1220 BOOL  ; 进料伺服X轴停止延时
T1221 BOOL  ; 进料伺服Z轴停止延时
T1222 BOOL  ; 出料伺服X轴停止延时
T1223 BOOL  ; 出料伺服Z轴停止延时
T1328 BOOL  ; $?St$Bk?_#[116] / 标漏阀开到位感应延时 / $?St$Bk?_#[116]
T1329 BOOL  ; $?St$Bk?_#[117] / 标漏阀关到位感应延时 / $?St$Bk?_#[117]
T1330 BOOL  ; 氦检仪真空阀开到位感应延时
T1331 BOOL  ; 氦检仪真空阀关到位感应延时
T1332 BOOL  ; 复检清洁阀开到位感应延时
T1333 BOOL  ; 复检清洁阀关到位感应延时
T1334 BOOL  ; #1腔体抽真空阀开到位感应延时
T1335 BOOL  ; #1腔体抽真空阀关到位感应延时
T1336 BOOL  ; #1-1腔体阀开到位感应延时
T1337 BOOL  ; #1-1腔体阀关到位感应延时
T1338 BOOL  ; #1-2腔体阀开到位感应延时
T1339 BOOL  ; #1-2腔体阀关到位感应延时
T1340 BOOL  ; #1腔体破真空阀开到位感应延时
T1341 BOOL  ; #1腔体破真空阀关到位感应延时
T1342 BOOL  ; #1腔体吹气阀开到位感应延时
T1343 BOOL  ; #1腔体吹气阀关到位感应延时
T1344 BOOL  ; #2腔体抽真空阀开到位感应延时
T1345 BOOL  ; #2腔体抽真空阀关到位感应延时
T1346 BOOL  ; #2-1腔体阀开到位感应延时
T1347 BOOL  ; #2-1腔体阀关到位感应延时
T1348 BOOL  ; #2-2腔体阀开到位感应延时
T1349 BOOL  ; #2-2腔体阀关到位感应延时
T1350 BOOL  ; #2腔体破真空阀开到位感应延时
T1351 BOOL  ; #2腔体破真空阀关到位感应延时
T1352 BOOL  ; #2腔体吹气阀开到位感应延时
T1353 BOOL  ; #2腔体吹气阀关到位感应延时
T1354 BOOL  ; #3腔体抽真空阀开到位感应延时
T1355 BOOL  ; #3腔体抽真空阀关到位感应延时
T1356 BOOL  ; #3-1腔体阀开到位感应延时
T1357 BOOL  ; #3-1腔体阀关到位感应延时
T1358 BOOL  ; #3-2腔体阀开到位感应延时
T1359 BOOL  ; #3-2腔体阀关到位感应延时
T1360 BOOL  ; #3腔体破真空阀开到位感应延时
T1361 BOOL  ; #3腔体破真空阀关到位感应延时
T1362 BOOL  ; #3腔体吹气阀开到位感应延时
T1363 BOOL  ; #3腔体吹气阀关到位感应延时
T1364 BOOL  ; #1-1电池抽真空阀开到位感应延时
T1365 BOOL  ; #1-1电池抽真空阀关到位感应延时
T1366 BOOL  ; #1-2电池抽真空阀开到位感应延时
T1367 BOOL  ; #1-2电池抽真空阀关到位感应延时
T1368 BOOL  ; #1-1电池注氦阀开到位感应延时
T1369 BOOL  ; #1-1电池注氦阀关到位感应延时
T1370 BOOL  ; #1-2电池注氦阀开到位感应延时
T1371 BOOL  ; #1-2电池注氦阀关到位感应延时
T1372 BOOL  ; #1-1电池破真空阀开到位感应延时
T1373 BOOL  ; #1-1电池破真空阀关到位感应延时
T1374 BOOL  ; #1-2电池破真空阀开到位感应延时
T1375 BOOL  ; #1-2电池破真空阀关到位感应延时
T1376 BOOL  ; #2-1电池抽真空阀开到位感应延时
T1377 BOOL  ; #2-1电池抽真空阀关到位感应延时
T1378 BOOL  ; #2-2电池抽真空阀开到位感应延时
T1379 BOOL  ; #2-2电池抽真空阀关到位感应延时
T1380 BOOL  ; #2-1电池注氦阀开到位感应延时
T1381 BOOL  ; #2-1电池注氦阀关到位感应延时
T1382 BOOL  ; #2-2电池注氦阀开到位感应延时
T1383 BOOL  ; #2-2电池注氦阀关到位感应延时
T1384 BOOL  ; #2-1电池破真空阀开到位感应延时
T1385 BOOL  ; #2-1电池破真空阀关到位感应延时
T1386 BOOL  ; #2-2电池破真空阀开到位感应延时
T1387 BOOL  ; #2-2电池破真空阀关到位感应延时
T1388 BOOL  ; #3-1电池抽真空阀开到位感应延时
T1389 BOOL  ; #3-1电池抽真空阀关到位感应延时
T1390 BOOL  ; #3-2电池抽真空阀开到位感应延时
T1391 BOOL  ; #3-2电池抽真空阀关到位感应延时
T1392 BOOL  ; #3-1电池注氦阀开到位感应延时
T1393 BOOL  ; #3-1电池注氦阀关到位感应延时
T1394 BOOL  ; #3-2电池注氦阀开到位感应延时
T1395 BOOL  ; #3-2电池注氦阀关到位感应延时
T1396 BOOL  ; #3-1电池破真空阀开到位感应延时
T1397 BOOL  ; #3-1电池破真空阀关到位感应延时
T1398 BOOL  ; #3-2电池破真空阀开到位感应延时
T1399 BOOL  ; #3-2电池破真空阀关到位感应延时
T1500 BOOL  ; 进料拉带机构开始运行条件延时
T1509 BOOL  ; 进料拉带机构复位完成延时
T1520 BOOL  ; 进料伺服机构开始运行条件1延时（进料拉带取料）
T1521 BOOL  ; 进料伺服机构开始运行条件2延时（扫码NG放料）
T1522 BOOL  ; 进料伺服机构开始运行条件3延时（扫码配对取/放料）
T1523 BOOL  ; 进料伺服机构开始运行条件4延时（腔体放料）
T1527 BOOL  ; 进料伺服X轴定位延时
T1528 BOOL  ; 进料伺服Z轴定位延时
T1529 BOOL  ; 进料伺服机构复位完成延时
T1530 BOOL  ; #1腔体机构开始运行条件延时(自动步)
T1531 BOOL  ; #1腔体机构数据初始化延时（自动步）
T1535 BOOL  ; #1腔体机构开始运行条件延时（自动单检步）
T1536 BOOL  ; #1腔体机构开始运行延时（清氦步）
T1539 BOOL  ; #1腔体机构复位完成延时
T1540 BOOL  ; 除#1氦检阀均关闭
T1550 BOOL  ; #2腔体机构开始运行条件延时(自动步)
T1551 BOOL  ; #2腔体机构数据初始化延时（自动步）
T1555 BOOL  ; #2腔体机构开始运行条件延时（自动单检步）
T1556 BOOL  ; #2腔体机构开始运行延时（清氦步）
T1559 BOOL  ; #2腔体机构复位完成延时
T1560 BOOL  ; 除#2氦检阀均关闭
T1570 BOOL  ; #3腔体机构开始运行条件延时(自动步)
T1571 BOOL  ; #3腔体机构数据初始化延时（自动步）
T1575 BOOL  ; #3腔体机构开始运行条件延时（自动单检步）
T1576 BOOL  ; #3腔体机构开始运行延时（清氦步）
T1579 BOOL  ; #3腔体机构复位完成延时
T1580 BOOL  ; 除#3氦检阀均关闭
T1590 BOOL  ; 出料夹爪初始状态
T1600 BOOL  ; 自动模式下X模组定位需求
T1601 BOOL  ; 自动模式下Z模组定位需求
T1602 BOOL  ; 下料模组初始化X轴到待机位
T1603 BOOL  ; 下料模组初始化z轴到待机位
T1604 BOOL  ; 出料Z模组归零触发延迟
T1605 BOOL  ; 出料X模组归零触发延迟
T1606 BOOL  ; 出料Z模组柔性报警处理延迟
T1607 BOOL  ; 手动跟踪Z模组联动
T1608 BOOL  ; 手动跟踪X模组联动
T1609 BOOL  ; 跟踪需求触发延迟
T1620 BOOL  ; #1出料夹爪有料出站就绪通知延时
T1621 BOOL  ; #2出料夹爪有料出站就绪通知延时
T1700 BOOL  ; 扫码数据初始化延时
T1701 BOOL  ; 扫码触发前延时
T1900 BOOL  ; #1-1腔体抽真空阈值到达延时（测试）
T1901 BOOL  ; #1-1腔体抽真空时间上限到达延时（测试）
T1902 BOOL  ; #1-1腔体破真空阈值到达延时（测试）
T1904 BOOL  ; #1-1腔体氦检时间（测试）
T1905 BOOL  ; #1-1腔体抽气阀关闭延时（测试）
T1906 BOOL  ; #1-1腔体氦检数据取值判定延时（测试）
T1907 BOOL  ; #1-1腔体抽残气压力到达延时（测试）
T1908 BOOL  ; #1-1腔体抽残气时间上限到达延时（测试）
T1909 BOOL  ; #1-1腔体预抽时间到达延时（测试）
T1910 BOOL  ; $?St$Bk?_#[118] / #1-1腔体真空在可氦检状态（测试） / $?St$Bk?_#[118]
T1920 BOOL  ; #1-1电池抽真空阈值到达延时（测试）
T1921 BOOL  ; #1-1电池抽真空时间上限到达延时（测试）
T1922 BOOL  ; #1-1电池破真空阈值到达延时（测试）
T1923 BOOL  ; #1-1电池破真空时间上限到达延时（测试）
T1924 BOOL  ; #1-1电池注氦压力到达延时（测试）
T1925 BOOL  ; #1-1电池注氦时间上限到达延时（测试）
T1926 BOOL  ; #1-1电池抽残气压力到达延时（测试）
T1927 BOOL  ; #1-1电池抽残气时间上限到达延时（测试）
T1928 BOOL  ; #1-1电池预抽压力正常判定延时（测试）
T1940 BOOL  ; 数据初始化延时（清氦）
T1941 BOOL  ; 清氦注氮时长（清氦）
T1980 BOOL  ; #1-1腔体数据初始化延时（标漏）
T1981 BOOL  ; #1-1腔体抽真空阀值到达延时（标漏）
T1982 BOOL  ; #1-1腔体抽真空时间上限到达延时（标漏）
T1984 BOOL  ; #1-1腔体氦检延时（标漏）
T1985 BOOL  ; #1-1腔体氦检数据取值完成判定（标漏）
T1986 BOOL  ; 氦检阀打开后，腔体压力超过氦检安全阀值，判氦检异常（标漏）
T1987 BOOL  ; 开氦检阀前抽气阀关延时（标漏）
T1990 BOOL  ; 氦检仪稳定延时（公共）
T2000 BOOL  ; #2-1腔体抽真空阈值到达延时（测试）
T2001 BOOL  ; #2-1腔体抽真空时间上限到达延时（测试）
T2002 BOOL  ; #2-1腔体破真空阈值到达延时（测试）
T2004 BOOL  ; #2-1腔体氦检时间（测试）
T2005 BOOL  ; #2-1腔体抽气阀关闭延时（测试）
T2006 BOOL  ; #2-1腔体氦检数据取值判定延时（测试）
T2007 BOOL  ; #2-1腔体抽残气压力到达延时（测试）
T2008 BOOL  ; #2-1腔体抽残气时间上限到达延时（测试）
T2009 BOOL  ; #2-1腔体预抽时间到达延时（测试）
T2010 BOOL  ; #2-1腔体真空在可氦检状态（测试）
T2020 BOOL  ; #2-1电池抽真空阈值到达延时（测试）
T2021 BOOL  ; #2-1电池抽真空时间上限到达延时（测试）
T2022 BOOL  ; #2-1电池破真空阈值到达延时（测试）
T2023 BOOL  ; #2-1电池破真空时间上限到达延时（测试）
T2024 BOOL  ; #2-1电池注氦压力到达延时（测试）
T2025 BOOL  ; #2-1电池注氦时间上限到达延时（测试）
T2026 BOOL  ; #2-1电池抽残气压力到达延时（测试）
T2027 BOOL  ; #2-1电池抽残气时间上限到达延时（测试）
T2028 BOOL  ; #2-1电池预抽压力正常判定延时（测试）
T2040 BOOL  ; #2-1数据初始化延时（清氦）
T2041 BOOL  ; #2-1清氦注氮时长（清氦）
T2081 BOOL  ; #2-1腔体抽真空阀值到达延时（标漏）
T2082 BOOL  ; #2-1腔体抽真空时间上限到达延时（标漏）
T2084 BOOL  ; #2-1腔体氦检延时（标漏）
T2085 BOOL  ; #2-1腔体氦检数据取值完成判定（标漏）
T2086 BOOL  ; #2-1氦检阀打开后，腔体压力超过氦检安全阀值，判氦检异常（标漏）
T2087 BOOL  ; #2-1开氦检阀前抽气阀关延时（标漏）
T2100 BOOL  ; #3-1腔体抽真空阈值到达延时（测试）
T2101 BOOL  ; #3-1腔体抽真空时间上限到达延时（测试）
T2102 BOOL  ; #3-1腔体破真空阈值到达延时（测试）
T2104 BOOL  ; #3-1腔体氦检时间（测试）
T2105 BOOL  ; #3-1腔体抽气阀关闭延时（测试）
T2106 BOOL  ; #3-1腔体氦检数据取值判定延时（测试）
T2107 BOOL  ; #3-1腔体抽残气压力到达延时（测试）
T2108 BOOL  ; #3-1腔体抽残气时间上限到达延时（测试）
T2109 BOOL  ; #3-1腔体预抽时间到达延时（测试）
T2110 BOOL  ; #3-1腔体真空在可氦检状态（测试）
T2120 BOOL  ; #3-1电池抽真空阈值到达延时（测试）
T2121 BOOL  ; #3-1电池抽真空时间上限到达延时（测试）
T2122 BOOL  ; #3-1电池破真空阈值到达延时（测试）
T2123 BOOL  ; #3-1电池破真空时间上限到达延时（测试）
T2124 BOOL  ; #3-1电池注氦压力到达延时（测试）
T2125 BOOL  ; #3-1电池注氦时间上限到达延时（测试）
T2126 BOOL  ; #3-1电池抽残气压力到达延时（测试）
T2127 BOOL  ; #3-1电池抽残气时间上限到达延时（测试）
T2128 BOOL  ; #3-1电池预抽压力正常判定延时（测试）
T2140 BOOL  ; #3-1数据初始化延时（清氦）
T2141 BOOL  ; #3-1清氦注氮时长（清氦）
T2181 BOOL  ; #3-1腔体抽真空阀值到达延时（标漏）
T2182 BOOL  ; #3-1腔体抽真空时间上限到达延时（标漏）
T2184 BOOL  ; #3-1腔体氦检延时（标漏）
T2185 BOOL  ; #3-1腔体氦检数据取值完成判定（标漏）
T2186 BOOL  ; #3-1氦检阀打开后，腔体压力超过氦检安全阀值，判氦检异常（标漏）
T2187 BOOL  ; #3-1开氦检阀前抽气阀关延时（标漏）
T2220 BOOL  ; #1-2电池抽真空阈值到达延时（测试）
T2221 BOOL  ; #1-2电池抽真空时间上限到达延时（测试）
T2222 BOOL  ; #1-2电池破真空阈值到达延时（测试）
T2223 BOOL  ; #1-2电池破真空时间上限到达延时（测试）
T2224 BOOL  ; #1-2电池注氦压力到达延时（测试）
T2225 BOOL  ; #1-2电池注氦时间上限到达延时（测试）
T2226 BOOL  ; #1-2电池抽残气压力到达延时（测试）
T2227 BOOL  ; #1-2电池抽残气时间上限到达延时（测试）
T2228 BOOL  ; #1-2电池预抽压力正常判定延时（测试）
T2281 BOOL  ; #1-2腔体抽真空阀值到达延时（标漏）
T2282 BOOL  ; #1-2腔体抽真空时间上限到达延时（标漏）
T2284 BOOL  ; #1-2腔体氦检延时（标漏）
T2286 BOOL  ; #1-2氦检阀打开后，腔体压力超过氦检安全阀值，判氦检异常（标漏）
T2287 BOOL  ; #1-2开氦检阀前抽气阀关延时（标漏）
T2320 BOOL  ; #2-2电池抽真空阈值到达延时（测试）
T2321 BOOL  ; #2-2电池抽真空时间上限到达延时（测试）
T2322 BOOL  ; #2-2电池破真空阈值到达延时（测试）
T2323 BOOL  ; #2-2电池破真空时间上限到达延时（测试）
T2324 BOOL  ; #2-2电池注氦压力到达延时（测试）
T2325 BOOL  ; #2-2电池注氦时间上限到达延时（测试）
T2326 BOOL  ; #2-2电池抽残气压力到达延时（测试）
T2327 BOOL  ; #2-2电池抽残气时间上限到达延时（测试）
T2328 BOOL  ; #2-2电池预抽压力正常判定延时（测试）
T2381 BOOL  ; #2-2腔体抽真空阀值到达延时（标漏）
T2382 BOOL  ; #2-2腔体抽真空时间上限到达延时（标漏）
T2384 BOOL  ; #2-2腔体氦检延时（标漏）
T2386 BOOL  ; #2-2氦检阀打开后，腔体压力超过氦检安全阀值，判氦检异常（标漏）
T2387 BOOL  ; #2-2开氦检阀前抽气阀关延时（标漏）
T2420 BOOL  ; #3-2电池抽真空阈值到达延时（测试）
T2421 BOOL  ; #3-2电池抽真空时间上限到达延时（测试）
T2422 BOOL  ; #3-2电池破真空阈值到达延时（测试）
T2423 BOOL  ; #3-2电池破真空时间上限到达延时（测试）
T2424 BOOL  ; #3-2电池注氦压力到达延时（测试）
T2425 BOOL  ; #3-2电池注氦时间上限到达延时（测试）
T2426 BOOL  ; #3-2电池抽残气压力到达延时（测试）
T2427 BOOL  ; #3-2电池抽残气时间上限到达延时（测试）
T2428 BOOL  ; #3-2电池预抽压力正常判定延时（测试）
T2481 BOOL  ; #3-2腔体抽真空阀值到达延时（标漏）
T2482 BOOL  ; #3-2腔体抽真空时间上限到达延时（标漏）
T2484 BOOL  ; #3-2腔体氦检延时（标漏）
T2486 BOOL  ; #3-2氦检阀打开后，腔体压力超过氦检安全阀值，判氦检异常（标漏）
T2487 BOOL  ; #3-2开氦检阀前抽气阀关延时（标漏）
T2521 BOOL  ; 进料#1扫码延时
T2522 BOOL  ; 接收数据清零延时发送无协议通讯TXD
T2523 BOOL  ; 进料#1扫码结果判定延时
T2524 BOOL  ; 进料#1扫码发送超时
T2531 BOOL  ; 进料#2扫码延时
T2532 BOOL  ; 扫码长度判定延时
W0.00 BOOL  ; 启动按钮（SW）
W0.01 BOOL  ; 停止按钮(SW)
W0.02 BOOL  ; 复位按钮（SW）
W0.04 BOOL  ; 整机复位按钮（SW）
W0.05 BOOL  ; 清料停止按钮（SW）
W0.06 BOOL  ; 整机记忆清除（SW）
W0.07 BOOL  ; 门磁屏蔽（SW）
W0.08 BOOL  ; 蜂鸣器屏蔽（SW）
W0.14 BOOL  ; 进料拉带#1扫码测试[SW]
W0.15 BOOL  ; 进料拉带#2扫码测试[SW]
W100.00 BOOL  ; 扫码NG料满位标志
W100.01 BOOL  ; 氦检NG料满标志
W1.00 BOOL  ; 手动模式
W1.01 BOOL  ; 自动模式
W1.09 BOOL  ; 伺服进料允许（允许=0）
W1.10 BOOL  ; 上料位有料模拟
W1.11 BOOL  ; 清料时单个料有效选择
W1.15 BOOL  ; 有料记忆异常屏蔽（手动调试）
W200.00 BOOL  ; 进料拉带机构隔离位&扫码位&进料位全有料标志
W200.01 BOOL  ; 调试1
W200.02 BOOL  ; 调试2
W200.03 BOOL  ; 调试3
W204.00 BOOL  ; 来料拉带机构单步标志
W20.00 BOOL  ; 腔体真空泵停机1分钟内禁止启动保护
W20.01 BOOL  ; 氦检前置泵停机1分钟内禁止启动保护
W210.00 BOOL  ; 进料伺服有取料需求标志
W210.01 BOOL  ; 进料伺服有放扫码NG料需求标志
W210.02 BOOL  ; 进料伺服有配对取/放料需求标志
W210.03 BOOL  ; 进料伺服有腔体放料需求标志
W211.00 BOOL  ; 进料伺服有配对放料需求标志
W211.01 BOOL  ; 进料伺服有配对取料需求标志
W211.02 BOOL  ; #1氦检腔有放料需求标志
W211.03 BOOL  ; #2氦检腔有放料需求标志
W211.04 BOOL  ; #3氦检腔有放料需求标志
W230.00 BOOL  ; 出料模组X轴初始化完成
W230.03 BOOL  ; 下料模组X/Z运行许可
W231.00 BOOL  ; 出料伺服Z轴到待机位
W231.01 BOOL  ; 出料伺服X轴到#1腔取料位
W231.02 BOOL  ; 出料伺服X轴到#2腔取料位
W231.03 BOOL  ; 出料伺服X轴到#3腔取料位
W231.04 BOOL  ; 出料伺服Z轴到#1腔取料位
W231.05 BOOL  ; 出料伺服Z轴到#2腔取料位
W231.06 BOOL  ; 出料伺服Z轴到#3腔取料位
W231.07 BOOL  ; $?St$Bk?_#[119] / 下料Z模组到待机位 / $?St$Bk?_#[119]
W231.08 BOOL  ; 下料X模组到OK下料位
W231.09 BOOL  ; 下料Z模组到OK下料位
W231.10 BOOL  ; 下料Z模组到待机位
W232 CHANNEL  ; INI_PV字
W234.00 BOOL  ; 出料Z轴到待机位
W234.01 BOOL  ; 出料X到2#爪放NG位置
W234.02 BOOL  ; 出料Z轴到2#爪放NG位置
W234.03 BOOL  ; 出料Z轴回待机位
W234.04 BOOL  ; 出料X到1#爪放NG位置
W234.05 BOOL  ; 出料Z轴到1#爪放NG位置
W234.06 BOOL  ; 出料Z轴回待机位
W236.00 BOOL  ; 出料Z模组到待机位
W236.01 BOOL  ; 出料伺服X轴到#2夹爪氦检NG放料位
W236.02 BOOL  ; 出料伺服X轴到#1夹爪氦检NG放料位
W236.03 BOOL  ; 出料伺服z轴到#2夹爪氦检NG放料位
W236.04 BOOL  ; 出料伺服Z轴到#1夹爪氦检NG放料位
W236.05 BOOL  ; 出料Z轴到待机位
W236.06 BOOL  ; 出料伺服X轴到#1夹爪配对取放料位
W236.07 BOOL  ; 出料伺服X轴到#2夹爪配对取放料位
W236.09 BOOL  ; 出料伺服Z轴到#1夹爪配对取放料位
W236.10 BOOL  ; 出料伺服Z轴到#2夹爪配对取放料位
W236.11 BOOL  ; 出料伺服Z轴到待机位
W236.12 BOOL  ; 出料伺服X轴到OK放料位
W236.13 BOOL  ; 出料伺服z轴到OK放料位
W236.14 BOOL  ; 出料Z轴到待机位
W240.00 BOOL  ; 出料模组Z轴初始化完成
W2.00 BOOL  ; 清料按钮（SW）
W2.01 BOOL  ; 设备PPM计数启动按钮（SW）
W30.00 BOOL  ; #1来料位有料标志
W30.01 BOOL  ; #1隔离位有料标志
W30.02 BOOL  ; #1扫码阻挡有料标志
W30.03 BOOL  ; #1进料位有料标志
W31.00 BOOL  ; #2来料位有料标志
W31.01 BOOL  ; #2隔离位有料标志
W31.02 BOOL  ; #2扫码阻挡有料标志
W31.03 BOOL  ; #2进料位有料标志
W360.03 BOOL  ; 进料伺服X轴取料位设定按钮(SW)
W360.04 BOOL  ; 进料伺服X轴#1腔放料位设定按钮(SW)
W360.05 BOOL  ; 进料伺服X轴#2腔放料位设定按钮(SW)
W360.06 BOOL  ; 进料伺服X轴#3腔放料位设定按钮(SW)
W360.07 BOOL  ; 进料伺服X轴#1夹爪扫码NG放料位设定按钮(SW)
W360.08 BOOL  ; 进料伺服X轴#2夹爪扫码NG放料位设定按钮(SW)
W360.09 BOOL  ; 进料伺服X轴#1夹爪配对取放料位设定按钮(SW)
W360.10 BOOL  ; 进料伺服X轴#2夹爪配对取放料位设定按钮(SW)
W360.11 BOOL  ; 进料伺服X轴#1腔有料检测位设定按钮(SW)
W360.12 BOOL  ; 进料伺服X轴#2腔有料检测位设定按钮(SW)
W360.13 BOOL  ; 进料伺服X轴#3腔有料检测位设定按钮(SW)
W361.03 BOOL  ; 进料伺服X轴取料位触发标志
W361.04 BOOL  ; 进料伺服X轴#1腔放料位触发标志
W361.05 BOOL  ; 进料伺服X轴#2腔放料位触发标志
W361.06 BOOL  ; 进料伺服X轴#3腔放料位触发标志
W361.07 BOOL  ; 进料伺服X轴#1夹爪扫码NG放料位触发标志
W361.08 BOOL  ; 进料伺服X轴#2夹爪扫码NG放料位触发标志
W361.09 BOOL  ; 进料伺服X轴#1夹爪配对取放料位触发标志
W361.10 BOOL  ; 进料伺服X轴#2夹爪配对取放料位触发标志
W361.11 BOOL  ; 进料伺服X轴#1腔有料检测位触发标志
W361.12 BOOL  ; 进料伺服X轴#2腔有料检测位触发标志
W361.13 BOOL  ; 进料伺服X轴#3腔有料检测位触发标志
W362.03 BOOL  ; 进料伺服Z轴待机位设定按钮(SW)
W363.03 BOOL  ; 进料伺服Z轴待机位触发标志
W363.04 BOOL  ; 进料伺服Z轴取料位触发标志
W363.05 BOOL  ; 进料伺服Z轴#1腔放料位触发标志
W363.06 BOOL  ; 进料伺服Z轴#2腔放料位触发标志
W363.07 BOOL  ; 进料伺服Z轴#3腔放料位触发标志
W363.08 BOOL  ; 进料伺服Z轴#1夹爪扫码NG放料位触发标志
W363.09 BOOL  ; 进料伺服Z轴#2夹爪扫码NG放料位触发标志
W363.10 BOOL  ; 进料伺服Z轴#1夹爪配对取放料位触发标志
W363.11 BOOL  ; 进料伺服Z轴#2夹爪配对取放料位触发标志
W370.03 BOOL  ; 出料伺服X轴放料位设定按钮(SW)
W370.04 BOOL  ; 出料伺服X轴#1腔取料位设定按钮(SW)
W370.05 BOOL  ; 出料伺服X轴#2腔取料位设定按钮(SW)
W370.06 BOOL  ; 出料伺服X轴#3腔取料位设定按钮(SW)
W370.07 BOOL  ; 出料伺服X轴#1夹爪氦检NG放料位设定按钮(SW)
W370.08 BOOL  ; 出料伺服X轴#2夹爪氦检NG放料位设定按钮(SW)
W370.09 BOOL  ; 出料伺服X轴#1夹爪配对取放料位设定按钮(SW)
W370.10 BOOL  ; 出料伺服X轴#2夹爪配对取放料位设定按钮(SW)
W371.03 BOOL  ; 出料伺服X轴放料位触发标志
W371.04 BOOL  ; 出料伺服X轴#1腔取料位触发标志
W371.05 BOOL  ; 出料伺服X轴#2腔取料位触发标志
W371.06 BOOL  ; 出料伺服X轴#3腔取料位触发标志
W371.07 BOOL  ; 出料伺服X轴#1夹爪氦检NG放料位触发标志
W371.08 BOOL  ; 出料伺服X轴#2夹爪氦检NG放料位触发标志
W371.09 BOOL  ; 出料伺服X轴#1夹爪配对取放料位触发标志
W371.10 BOOL  ; 出料伺服X轴#2夹爪配对取放料位触发标志
W372.03 BOOL  ; 出料伺服Z轴待机位设定按钮(SW)
W373.03 BOOL  ; 出料伺服Z轴待机位触发标志
W373.04 BOOL  ; 出料伺服Z轴放料位触发标志
W373.05 BOOL  ; 出料伺服Z轴#1腔取料位触发标志
W373.06 BOOL  ; 出料伺服Z轴#2腔取料位触发标志
W373.07 BOOL  ; 出料伺服Z轴#3腔取料位触发标志
W373.08 BOOL  ; 出料伺服Z轴#1夹爪氦检NG放料位触发标志
W373.09 BOOL  ; 出料伺服Z轴#2夹爪氦检NG放料位触发标志
W373.10 BOOL  ; 出料伺服Z轴#1夹爪配对取放料位触发标志
W373.11 BOOL  ; 出料伺服Z轴#2夹爪配对取放料位触发标志
W380.01 BOOL  ; 读氦检仪状态完成
W380.06 BOOL  ; 读氦检仪检漏口压力完成
W380.11 BOOL  ; 读氦检仪漏率完成
W380.15 BOOL  ; 氦检仪漏率低于设定值（稳态）
W381.00 BOOL  ; 氦检仪在检漏状态
W381.03 BOOL  ; 氦检仪在启动状态
W3.00 BOOL  ; 氦检单双检测选择允许
W400 CHANNEL  ; 设备故障
W400.00 BOOL  ; #1扫码阻挡气缸缩回位[alm]
W400.01 BOOL  ; #1扫码阻挡气缸伸出位[alm]
W400.02 BOOL  ; #1隔离气缸缩回位[alm]
W400.03 BOOL  ; 0[alm]
W400.04 BOOL  ; #2扫码阻挡气缸缩回位[alm]
W400.05 BOOL  ; #2扫码阻挡气缸伸出位[alm]
W400.06 BOOL  ; #2隔离气缸缩回位[alm]
W400.07 BOOL  ; 0[alm]
W400.08 BOOL  ; #1进料夹爪夹紧位[alm]
W400.09 BOOL  ; #1进料夹爪松开位[alm]
W400.10 BOOL  ; #2进料夹爪夹紧位[alm]
W400.11 BOOL  ; #2进料夹爪松开位[alm]
W400.12 BOOL  ; 进料夹爪变距气缸伸出位[alm]
W400.13 BOOL  ; 进料夹爪变距气缸缩回位[alm]
W400.14 BOOL  ; #1出料夹爪夹紧位[alm]
W400.15 BOOL  ; #1出料夹爪松开位[alm]
W401.00 BOOL  ; #2出料夹爪夹紧位[alm]
W401.01 BOOL  ; #2出料夹爪松开位[alm]
W401.02 BOOL  ; 出料夹爪变距气缸伸出位[alm]
W401.03 BOOL  ; 出料夹爪变距气缸缩回位[alm]
W401.04 BOOL  ; #1腔体平移一级气缸缩回位[alm]
W401.05 BOOL  ; #1腔体平移一级气缸伸出位[alm]
W401.06 BOOL  ; #1腔体平移二级气缸缩回位[alm]
W401.07 BOOL  ; #1腔体平移二级气缸伸出位[alm]
W401.08 BOOL  ; #1腔体顶伸气缸上升位[alm]
W401.09 BOOL  ; #1腔体顶伸气缸下降位[alm]
W401.10 BOOL  ; #1腔体氦检阀开到位[alm]
W401.11 BOOL  ; #1腔体氦检阀关到位[alm]
W401.12 BOOL  ; 0[alm]
W401.13 BOOL  ; 0[alm]
W401.14 BOOL  ; 0[alm]
W401.15 BOOL  ; 0[alm]
W402.00 BOOL  ; 0[alm]
W402.01 BOOL  ; #2腔体平移一级气缸缩回位[alm]
W402.02 BOOL  ; #2腔体平移一级气缸伸出位[alm]
W402.03 BOOL  ; #2腔体平移二级气缸缩回位[alm]
W402.04 BOOL  ; #2腔体平移二级气缸伸出位[alm]
W402.05 BOOL  ; #2腔体顶伸气缸上升位[alm]
W402.06 BOOL  ; #2腔体顶伸气缸下降位[alm]
W402.07 BOOL  ; #2腔体氦检阀开到位[alm]
W402.08 BOOL  ; #2腔体氦检阀关到位[alm]
W402.09 BOOL  ; 0[alm]
W402.10 BOOL  ; 0[alm]
W402.11 BOOL  ; 0[alm]
W402.12 BOOL  ; 0[alm]
W402.13 BOOL  ; 0[alm]
W402.14 BOOL  ; #3腔体平移一级气缸缩回位[alm]
W402.15 BOOL  ; #3腔体平移一级气缸伸出位[alm]
W403.00 BOOL  ; #3腔体平移二级气缸缩回位[alm]
W403.01 BOOL  ; #3腔体平移二级气缸伸出位[alm]
W403.02 BOOL  ; #3腔体顶伸气缸上升位[alm]
W403.03 BOOL  ; #3腔体顶伸气缸下降位[alm]
W403.04 BOOL  ; #3腔体氦检阀开到位[alm]
W403.05 BOOL  ; #3腔体氦检阀关到位[alm]
W403.06 BOOL  ; 氦检仪准备好了信号[alm]
W403.07 BOOL  ; 氦检仪故障信号[alm]
W403.08 BOOL  ; 0[alm]
W403.09 BOOL  ; 0[alm]
W403.10 BOOL  ; 0[alm]
W403.11 BOOL  ; 进料伺服X轴准备好了信号[alm]
W403.12 BOOL  ; 进料伺服X轴故障信号[alm]
W403.13 BOOL  ; 进料伺服Z轴准备好了信号[alm]
W403.14 BOOL  ; 进料伺服Z轴故障信号[alm]
W403.15 BOOL  ; 0[alm]
W404.00 BOOL  ; 出料伺服X轴准备好了信号[alm]
W404.01 BOOL  ; 出料伺服X轴故障信号[alm]
W404.02 BOOL  ; 出料伺服Z轴准备好了信号[alm]
W404.03 BOOL  ; 出料伺服Z轴故障信号[alm]
W404.04 BOOL  ; 0[alm]
W404.05 BOOL  ; 腔体抽真空泵运行信号[alm]
W404.06 BOOL  ; 腔体抽真空泵过载信号[alm]
W404.07 BOOL  ; 氦检前置泵运行信号[alm]
W404.08 BOOL  ; 氦检前置泵过载信号[alm]
W404.09 BOOL  ; 启动按钮[alm]
W404.10 BOOL  ; 停止按钮[alm]
W404.11 BOOL  ; 复位按钮[alm]
W404.12 BOOL  ; 急停按钮[alm]
W404.13 BOOL  ; 手自动选择[alm]
W404.14 BOOL  ; #1进料夹爪防下坠感应[alm]
W404.15 BOOL  ; #2进料夹爪防下坠感应[alm]
W405.00 BOOL  ; #1出料夹爪防下坠感应[alm]
W405.01 BOOL  ; #2出料夹爪防下坠感应[alm]
W405.02 BOOL  ; 0[alm]
W405.03 BOOL  ; 进料对接输入[alm]
W405.04 BOOL  ; 出料对接输入[alm]
W405.05 BOOL  ; 0[alm]
W405.06 BOOL  ; 0[alm]
W405.07 BOOL  ; 设备总气压信号[alm]
W405.08 BOOL  ; #1来料位有料感应[alm]
W405.09 BOOL  ; #2来料位有料感应[alm]
W405.10 BOOL  ; #1隔离位有料感应[alm]
W405.11 BOOL  ; #2隔离位有料感应[alm]
W405.12 BOOL  ; #1扫码位有料感应[alm]
W405.13 BOOL  ; #2扫码位有料感应[alm]
W405.14 BOOL  ; #1-1进料位有料感应[alm]
W405.15 BOOL  ; #1-2进料位有料感应[alm]
W406.00 BOOL  ; #2-1进料位有料感应[alm]
W406.01 BOOL  ; #2-2进料位有料感应[alm]
W406.02 BOOL  ; 进料夹爪柔性感应[alm]
W406.03 BOOL  ; 出料夹爪柔性感应[alm]
W406.04 BOOL  ; #1进料夹爪对应腔体有料感应[alm]
W406.05 BOOL  ; #2进料夹爪对应腔体有料感应[alm]
W406.06 BOOL  ; 扫码NG放料#1位有料感应[alm]
W406.07 BOOL  ; 扫码NG放料#2位有料感应[alm]
W406.08 BOOL  ; 扫码NG料满位有料感应[alm]
W406.09 BOOL  ; 进料配对位有料感应[alm]
W406.10 BOOL  ; 出料配对位有料感应[alm]
W406.11 BOOL  ; 氦检NG放料#1位有料感应[alm]
W406.12 BOOL  ; 氦检NG放料#2位有料感应[alm]
W406.13 BOOL  ; 氦检NG料满位有料感应[alm]
W406.14 BOOL  ; #1-1出料位有料感应[alm]
W406.15 BOOL  ; #1-2出料位有料感应[alm]
W407.00 BOOL  ; #2-1出料位有料感应[alm]
W407.01 BOOL  ; #2-2出料位有料感应[alm]
W407.02 BOOL  ; #1门磁开关[alm]
W407.03 BOOL  ; #2门磁开关[alm]
W407.04 BOOL  ; #3门磁开关[alm]
W407.05 BOOL  ; #4门磁开关[alm]
W407.06 BOOL  ; #5门磁开关[alm]
W407.07 BOOL  ; #6门磁开关[alm]
W407.08 BOOL  ; #7门磁开关[alm]
W407.09 BOOL  ; #8门磁开关[alm]
W407.10 BOOL  ; #9门磁开关[alm]
W407.11 BOOL  ; #10门磁开关[alm]
W407.12 BOOL  ; #11门磁开关[alm]
W407.13 BOOL  ; 设备真空压力信号[alm]
W407.14 BOOL  ; 设备氦气压力信号[alm]
W407.15 BOOL  ; 精密调压阀信号[alm]
W411.00 BOOL  ; 电脑软件未启动[alm]
W411.01 BOOL  ; 氦检仪通信异常[alm]
W411.02 BOOL  ; #1扫码枪通讯异常[alm]
W411.03 BOOL  ; #2扫码枪通讯异常[alm]
W411.04 BOOL  ; 进料扫码MES入站就绪通知&确认超时[alm]
W411.05 BOOL  ; 出料伺服MES出站就绪通知&确认超时[alm]
W413.00 BOOL  ; 进料伺服X轴正极限[alm]
W413.01 BOOL  ; 进料伺服X轴负极限[alm]
W413.02 BOOL  ; 进料伺服X轴原点[alm]
W413.03 BOOL  ; 进料伺服Z轴正极限[alm]
W413.04 BOOL  ; 进料伺服Z轴负极限[alm]
W413.05 BOOL  ; 进料伺服Z轴原点[alm]
W413.06 BOOL  ; 出料伺服X轴正极限[alm]
W413.07 BOOL  ; 出料伺服X轴负极限[alm]
W413.08 BOOL  ; 出料伺服X轴原点[alm]
W413.09 BOOL  ; 出料伺服Z轴正极限[alm]
W413.10 BOOL  ; 出料伺服Z轴负极限[alm]
W413.11 BOOL  ; 出料伺服Z轴原点[alm]
W414.00 BOOL  ; 氦检仪不在检漏状态[alm]
W416.00 BOOL  ; #1来料位有料记忆[alm]
W416.01 BOOL  ; #2来料位有料记忆[alm]
W416.02 BOOL  ; #1隔离位有料记忆[alm]
W416.03 BOOL  ; #2隔离位有料记忆[alm]
W416.04 BOOL  ; #1扫码位有料记忆[alm]
W416.05 BOOL  ; #2扫码位有料记忆[alm]
W416.06 BOOL  ; #1进料位有料记忆[alm]
W416.07 BOOL  ; #2进料位有料记忆[alm]
W416.08 BOOL  ; #1进料夹爪有料记忆[alm]
W416.09 BOOL  ; #2进料夹爪有料记忆[alm]
W416.10 BOOL  ; #1出料夹爪有料记忆[alm]
W416.11 BOOL  ; #2出料夹爪有料记忆[alm]
W416.12 BOOL  ; #1-1腔体有料记忆[alm]
W416.13 BOOL  ; #1-2腔体有料记忆[alm]
W416.14 BOOL  ; #2-1腔体有料记忆[alm]
W416.15 BOOL  ; #2-2腔体有料记忆[alm]
W417.00 BOOL  ; #3-1腔体有料记忆[alm]
W417.01 BOOL  ; #3-2腔体有料记忆[alm]
W417.02 BOOL  ; 进料配对位有料记忆[alm]
W417.03 BOOL  ; 出料配对位有料记忆[alm]
W417.04 BOOL  ; #1出料位有料记忆[alm]
W417.05 BOOL  ; #2出料位有料记忆[alm]
W417.06 BOOL  ; 扫码NG放料位有料记忆[alm]
W417.07 BOOL  ; 氦检NG拉带下料位有料记忆[alm]
W418.00 BOOL  ; 整机复位超时[alm]
W418.01 BOOL  ; 进料拉带工站复位超时[alm]
W418.02 BOOL  ; 进料伺服工站复位超时[alm]
W418.03 BOOL  ; #1氦检工站复位超时[alm]
W418.04 BOOL  ; #2氦检工站复位超时[alm]
W418.05 BOOL  ; #3氦检工站复位超时[alm]
W418.06 BOOL  ; 出料伺服工站复位超时[alm]
W4.00 BOOL  ; 初次上电#1腔体平移一级气缸伸出条件
W4.01 BOOL  ; 初次上电#1腔体平移二级气缸伸出条件
W4.02 BOOL  ; 初次上电#2腔体平移一级气缸伸出条件
W4.03 BOOL  ; 初次上电#2腔体平移二级气缸伸出条件
W4.04 BOOL  ; 初次上电#3腔体平移一级气缸伸出条件
W4.05 BOOL  ; 初次上电#3腔体平移二级气缸伸出条件
W5.05 BOOL  ; #1扫码料到位
W5.06 BOOL  ; #2扫码料到位
W65.00 BOOL  ; 进料#1扫码
W65.01 BOOL  ; 进料#1扫码发送
W65.02 BOOL  ; 进料#1扫码失败
W65.03 BOOL  ; 进料#1扫码成功
W65.04 BOOL  ; 进料#1扫码接收
W65.05 BOOL  ; 进料扫码重新触发
W75.00 BOOL  ; 进料#2扫码
W75.01 BOOL  ; 进料#2扫码发送
W75.02 BOOL  ; 进料#2扫码失败
W75.03 BOOL  ; 进料#2扫码成功
W75.04 BOOL  ; 进料#2扫码接收
W75.05 BOOL  ; 进料#2扫码重新触发
Battery_Vaccum_1_1 SMC混压表
Battery_Vaccum_1_2 SMC混压表
Battery_Vaccum_2_1 SMC混压表
Battery_Vaccum_2_2 SMC混压表
Battery_Vaccum_3_1 SMC混压表
Battery_Vaccum_3_2 SMC混压表
HJY 氦检仪
Vaccum_1 真空计
Vaccum_2 真空计
Vaccum_3 真空计
二号腔体自检 腔体自检
三号腔体自检 腔体自检
一号腔体自检 腔体自检

## Program Main (cyclic task 0)
Local symbols
D CHANNEL  ; 进料#1扫码数据开始字

### Section Main

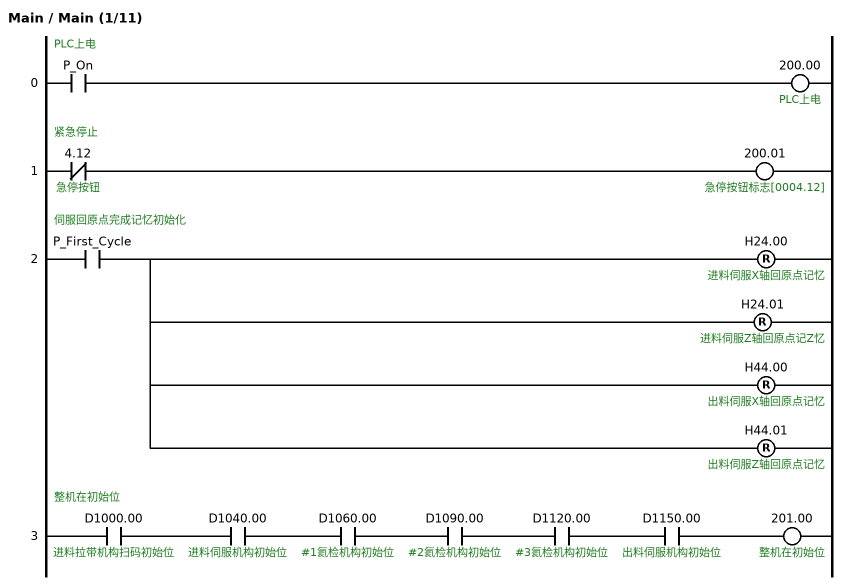
; rung 0: PLC上电
LD P_On
OUT 200.00  ; PLC上电
; rung 1: 紧急停止
LDNOT 4.12  ; 急停按钮
OUT 200.01  ; 急停按钮标志[0004.12]
; rung 2: 伺服回原点完成记忆初始化
LD P_First_Cycle
RSET H24.00  ; 进料伺服X轴回原点记忆
RSET H24.01  ; 进料伺服Z轴回原点记Z忆
RSET H44.00  ; 出料伺服X轴回原点记忆
RSET H44.01  ; 出料伺服Z轴回原点记忆
; rung 3: 整机在初始位
LD D1000.00  ; 进料拉带机构扫码初始位
AND D1040.00  ; 进料伺服机构初始位
AND D1060.00  ; #1氦检机构初始位
AND D1090.00  ; #2氦检机构初始位
AND D1120.00  ; #3氦检机构初始位
AND D1150.00  ; 出料伺服机构初始位
OUT 201.00  ; 整机在初始位

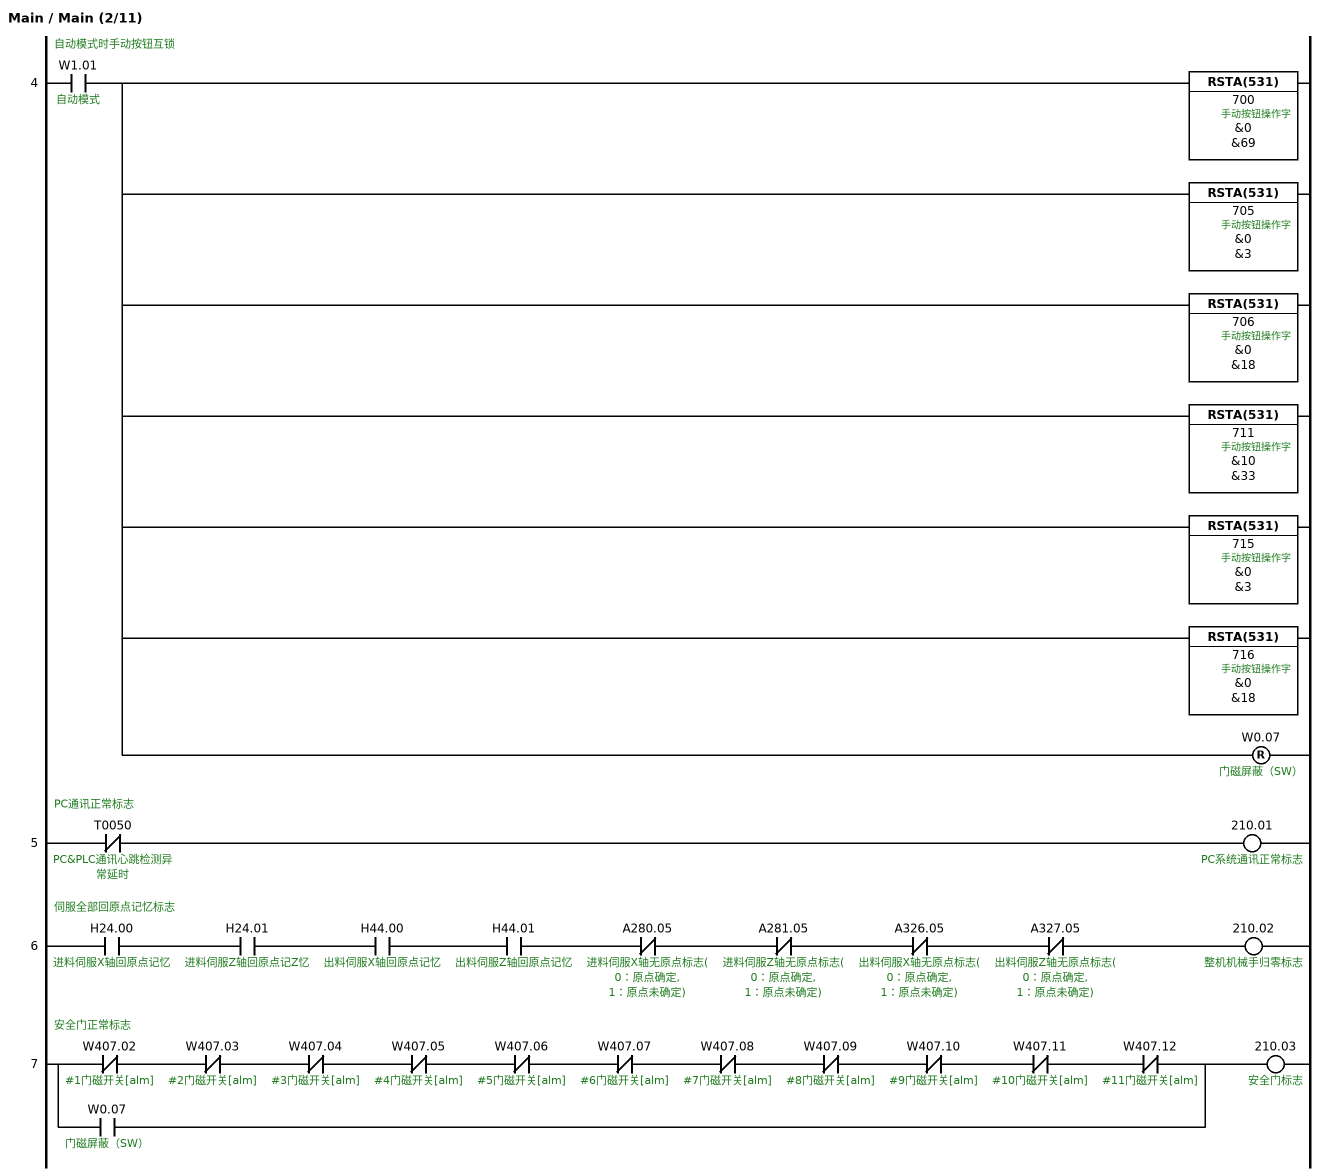
; rung 4: 自动模式时手动按钮互锁
LD W1.01  ; 自动模式
RSTA(531) 700 &0 &69  ; 手动按钮操作字
RSTA(531) 705 &0 &3  ; 手动按钮操作字
RSTA(531) 706 &0 &18  ; 手动按钮操作字
RSTA(531) 711 &10 &33  ; 手动按钮操作字
RSTA(531) 715 &0 &3  ; 手动按钮操作字
RSTA(531) 716 &0 &18  ; 手动按钮操作字
RSET W0.07  ; 门磁屏蔽（SW）
; rung 5: PC通讯正常标志
LDNOT T0050  ; PC&PLC通讯心跳检测异常延时
OUT 210.01  ; PC系统通讯正常标志
; rung 6: 伺服全部回原点记忆标志
LD H24.00  ; 进料伺服X轴回原点记忆
AND H24.01  ; 进料伺服Z轴回原点记Z忆
AND H44.00  ; 出料伺服X轴回原点记忆
AND H44.01  ; 出料伺服Z轴回原点记忆
ANDNOT A280.05  ; 进料伺服X轴无原点标志(0：原点确定,1：原点未确定)
ANDNOT A281.05  ; 进料伺服Z轴无原点标志(0：原点确定,1：原点未确定)
ANDNOT A326.05  ; 出料伺服X轴无原点标志(0：原点确定,1：原点未确定)
ANDNOT A327.05  ; 出料伺服Z轴无原点标志(0：原点确定,1：原点未确定)
OUT 210.02  ; 整机机械手归零标志
; rung 7: 安全门正常标志
LDNOT W407.02  ; #1门磁开关[alm]
ANDNOT W407.03  ; #2门磁开关[alm]
ANDNOT W407.04  ; #3门磁开关[alm]
ANDNOT W407.05  ; #4门磁开关[alm]
ANDNOT W407.06  ; #5门磁开关[alm]
ANDNOT W407.07  ; #6门磁开关[alm]
ANDNOT W407.08  ; #7门磁开关[alm]
ANDNOT W407.09  ; #8门磁开关[alm]
ANDNOT W407.10  ; #9门磁开关[alm]
ANDNOT W407.11  ; #10门磁开关[alm]
ANDNOT W407.12  ; #11门磁开关[alm]
OR W0.07  ; 门磁屏蔽（SW）
OUT 210.03  ; 安全门标志

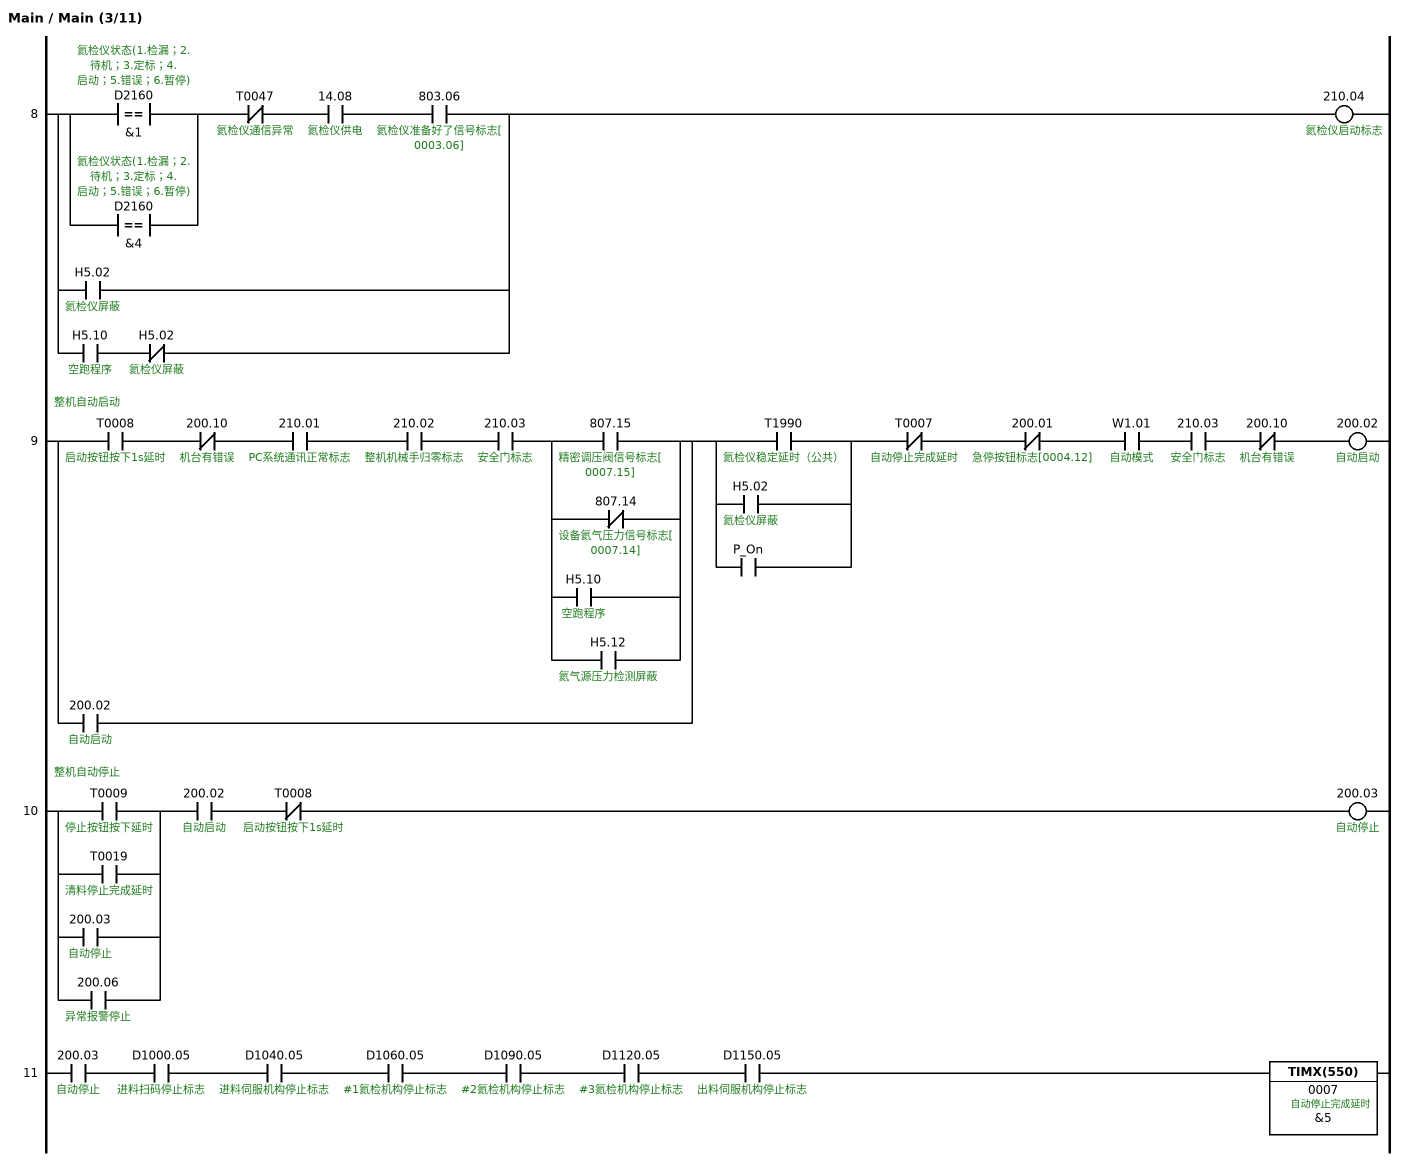
; rung 8
LD=(300) D2160 &1  ; 氦检仪状态(1.检漏；2.待机；3.定标；4.启动；5.错误；6.暂停)
OR=(300) D2160 &4  ; 氦检仪状态(1.检漏；2.待机；3.定标；4.启动；5.错误；6.暂停)
ANDNOT T0047  ; 氦检仪通信异常
AND 14.08  ; 氦检仪供电
AND 803.06  ; 氦检仪准备好了信号标志[0003.06]
OR H5.02  ; 氦检仪屏蔽
LD H5.10  ; 空跑程序
ANDNOT H5.02  ; 氦检仪屏蔽
ORLD
OUT 210.04  ; 氦检仪启动标志
; rung 9: 整机自动启动
LD T0008  ; 启动按钮按下1s延时
ANDNOT 200.10  ; 机台有错误
AND 210.01  ; PC系统通讯正常标志
AND 210.02  ; 整机机械手归零标志
AND 210.03  ; 安全门标志
LD 807.15  ; 精密调压阀信号标志[0007.15]
ORNOT 807.14  ; 设备氦气压力信号标志[0007.14]
OR H5.10  ; 空跑程序
OR H5.12  ; 氦气源压力检测屏蔽
ANDLD
OR 200.02  ; 自动启动
LD T1990  ; 氦检仪稳定延时（公共）
OR H5.02  ; 氦检仪屏蔽
OR P_On
ANDLD
ANDNOT T0007  ; 自动停止完成延时
ANDNOT 200.01  ; 急停按钮标志[0004.12]
AND W1.01  ; 自动模式
AND 210.03  ; 安全门标志
ANDNOT 200.10  ; 机台有错误
OUT 200.02  ; 自动启动
; rung 10: 整机自动停止
LD T0009  ; 停止按钮按下延时
OR T0019  ; 清料停止完成延时
OR 200.03  ; 自动停止
OR 200.06  ; 异常报警停止
AND 200.02  ; 自动启动
ANDNOT T0008  ; 启动按钮按下1s延时
OUT 200.03  ; 自动停止
; rung 11
LD 200.03  ; 自动停止
AND D1000.05  ; 进料扫码停止标志
AND D1040.05  ; 进料伺服机构停止标志
AND D1060.05  ; #1氦检机构停止标志
AND D1090.05  ; #2氦检机构停止标志
AND D1120.05  ; #3氦检机构停止标志
AND D1150.05  ; 出料伺服机构停止标志
TIMX(550) 0007 &5  ; 自动停止完成延时

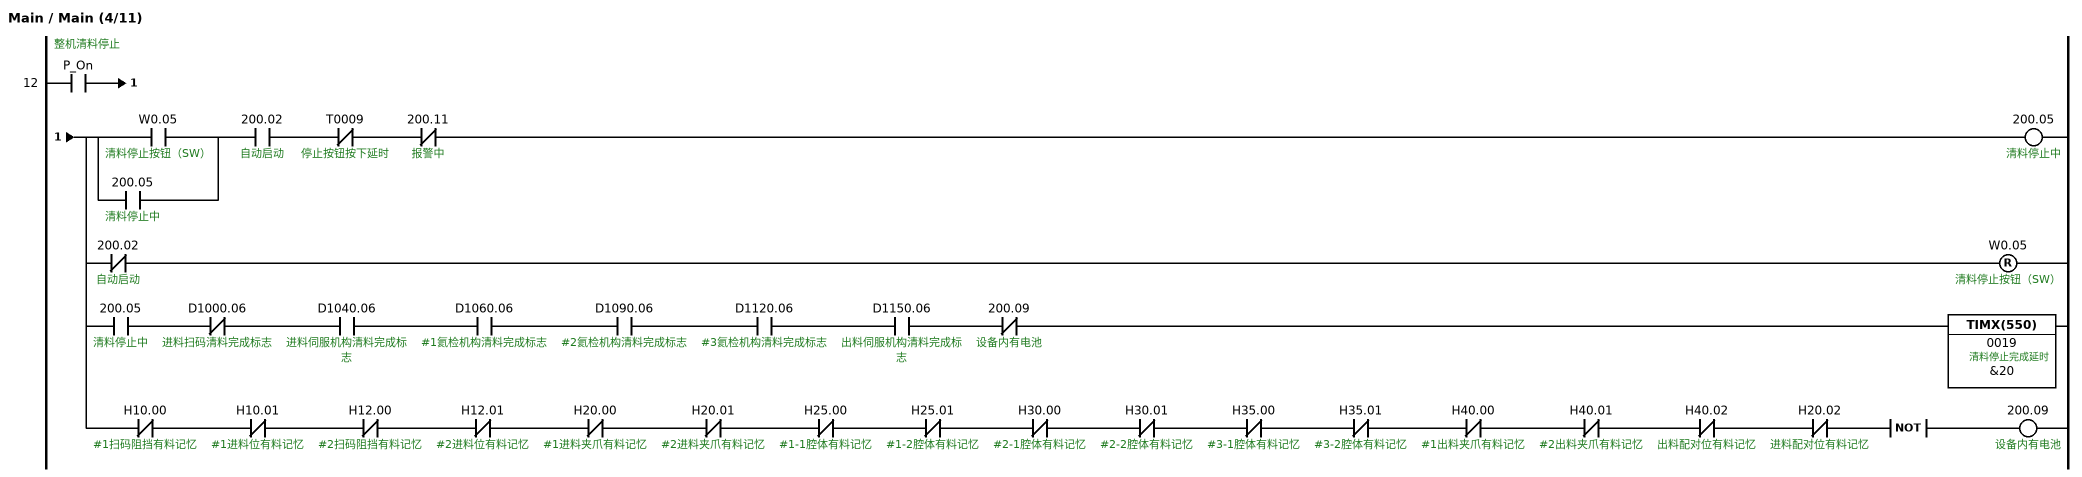
; rung 12: 整机清料停止
LD P_On
OUT TR0
LD W0.05  ; 清料停止按钮（SW）
OR 200.05  ; 清料停止中
ANDLD
AND 200.02  ; 自动启动
ANDNOT T0009  ; 停止按钮按下延时
ANDNOT 200.11  ; 报警中
OUT 200.05  ; 清料停止中
LD TR0
ANDNOT 200.02  ; 自动启动
RSET W0.05  ; 清料停止按钮（SW）
LD TR0
AND 200.05  ; 清料停止中
ANDNOT D1000.06  ; 进料扫码清料完成标志
AND D1040.06  ; 进料伺服机构清料完成标志
AND D1060.06  ; #1氦检机构清料完成标志
AND D1090.06  ; #2氦检机构清料完成标志
AND D1120.06  ; #3氦检机构清料完成标志
AND D1150.06  ; 出料伺服机构清料完成标志
ANDNOT 200.09  ; 设备内有电池
TIMX(550) 0019 &20  ; 清料停止完成延时
LD TR0
ANDNOT H10.00  ; #1扫码阻挡有料记忆
ANDNOT H10.01  ; #1进料位有料记忆
ANDNOT H12.00  ; #2扫码阻挡有料记忆
ANDNOT H12.01  ; #2进料位有料记忆
ANDNOT H20.00  ; #1进料夹爪有料记忆
ANDNOT H20.01  ; #2进料夹爪有料记忆
ANDNOT H25.00  ; #1-1腔体有料记忆
ANDNOT H25.01  ; #1-2腔体有料记忆
ANDNOT H30.00  ; #2-1腔体有料记忆
ANDNOT H30.01  ; #2-2腔体有料记忆
ANDNOT H35.00  ; #3-1腔体有料记忆
ANDNOT H35.01  ; #3-2腔体有料记忆
ANDNOT H40.00  ; #1出料夹爪有料记忆
ANDNOT H40.01  ; #2出料夹爪有料记忆
ANDNOT H40.02  ; 出料配对位有料记忆
ANDNOT H20.02  ; 进料配对位有料记忆
NOT(520)
OUT 200.09  ; 设备内有电池

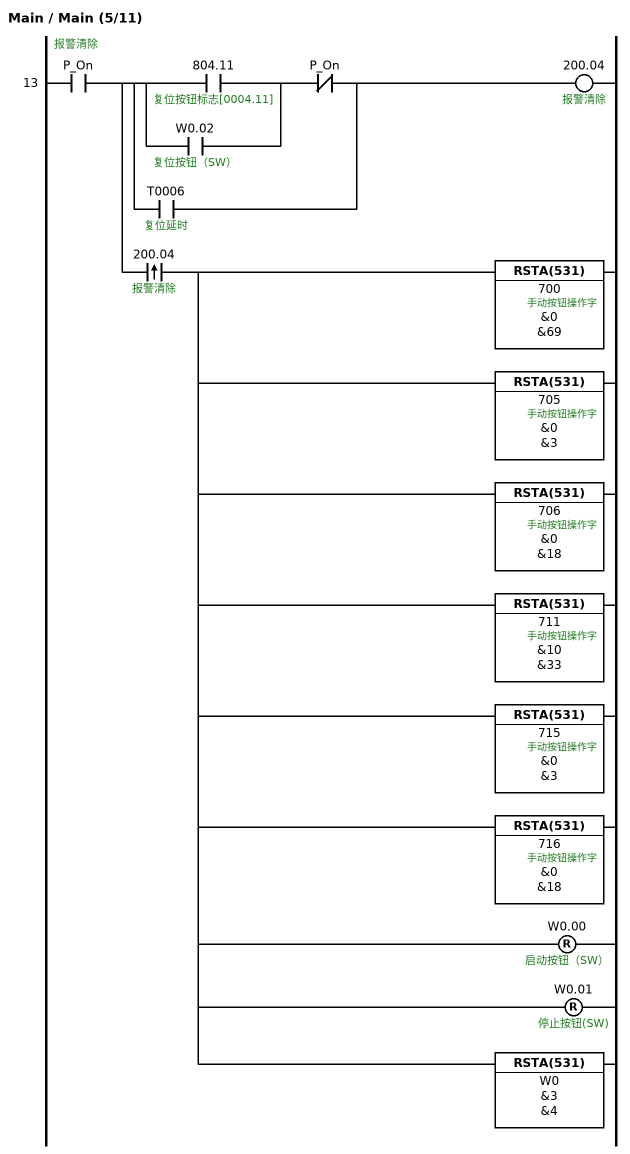
; rung 13: 报警清除
LD P_On
OUT TR0
LD 804.11  ; 复位按钮标志[0004.11]
OR W0.02  ; 复位按钮（SW）
ANDNOT P_On
OR T0006  ; 复位延时
ANDLD
OUT 200.04  ; 报警清除
LD TR0
@AND 200.04  ; 报警清除
RSTA(531) 700 &0 &69  ; 手动按钮操作字
RSTA(531) 705 &0 &3  ; 手动按钮操作字
RSTA(531) 706 &0 &18  ; 手动按钮操作字
RSTA(531) 711 &10 &33  ; 手动按钮操作字
RSTA(531) 715 &0 &3  ; 手动按钮操作字
RSTA(531) 716 &0 &18  ; 手动按钮操作字
RSET W0.00  ; 启动按钮（SW）
RSET W0.01  ; 停止按钮(SW)
RSTA(531) W0 &3 &4

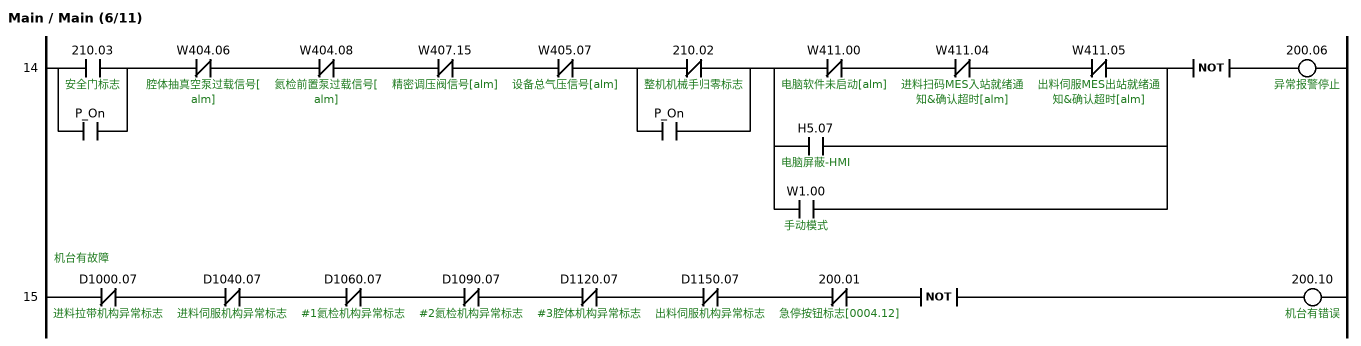
; rung 14
LD 210.03  ; 安全门标志
OR P_On
ANDNOT W404.06  ; 腔体抽真空泵过载信号[alm]
ANDNOT W404.08  ; 氦检前置泵过载信号[alm]
ANDNOT W407.15  ; 精密调压阀信号[alm]
ANDNOT W405.07  ; 设备总气压信号[alm]
LDNOT 210.02  ; 整机机械手归零标志
OR P_On
ANDLD
LDNOT W411.00  ; 电脑软件未启动[alm]
ANDNOT W411.04  ; 进料扫码MES入站就绪通知&确认超时[alm]
ANDNOT W411.05  ; 出料伺服MES出站就绪通知&确认超时[alm]
OR H5.07  ; 电脑屏蔽-HMI
OR W1.00  ; 手动模式
ANDLD
NOT(520)
OUT 200.06  ; 异常报警停止
; rung 15: 机台有故障
LDNOT D1000.07  ; 进料拉带机构异常标志
ANDNOT D1040.07  ; 进料伺服机构异常标志
ANDNOT D1060.07  ; #1氦检机构异常标志
ANDNOT D1090.07  ; #2氦检机构异常标志
ANDNOT D1120.07  ; #3腔体机构异常标志
ANDNOT D1150.07  ; 出料伺服机构异常标志
ANDNOT 200.01  ; 急停按钮标志[0004.12]
NOT(520)
OUT 200.10  ; 机台有错误

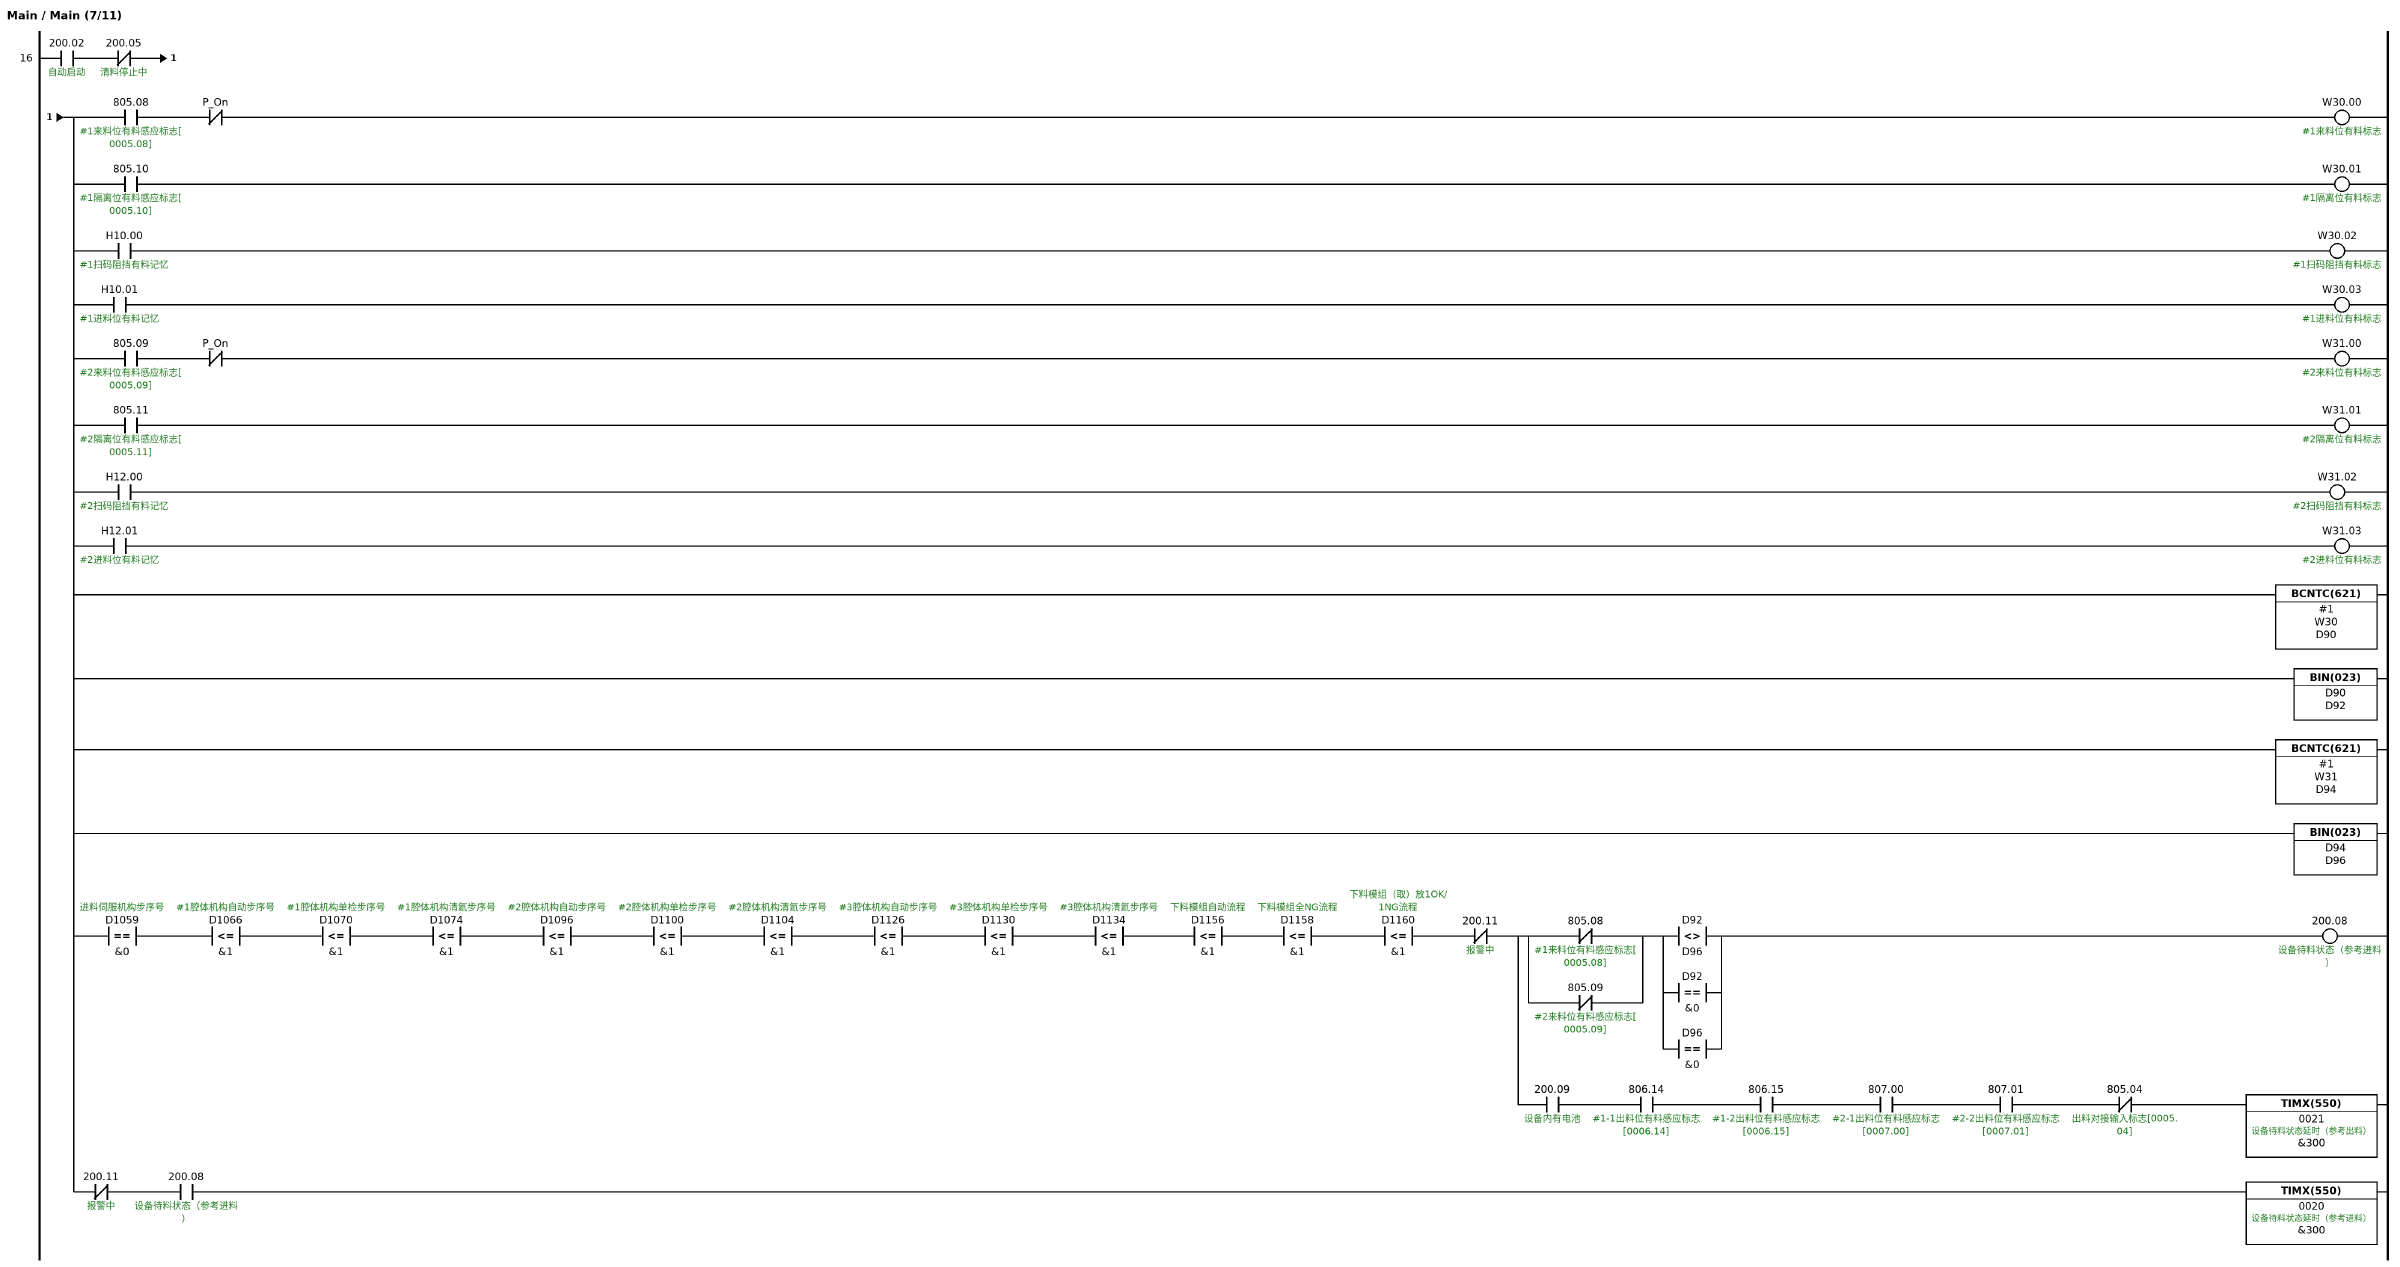
; rung 16
LD 200.02  ; 自动启动
ANDNOT 200.05  ; 清料停止中
OUT TR0
AND 805.08  ; #1来料位有料感应标志[0005.08]
ANDNOT P_On
OUT W30.00  ; #1来料位有料标志
LD TR0
AND 805.10  ; #1隔离位有料感应标志[0005.10]
OUT W30.01  ; #1隔离位有料标志
LD TR0
AND H10.00  ; #1扫码阻挡有料记忆
OUT W30.02  ; #1扫码阻挡有料标志
LD TR0
AND H10.01  ; #1进料位有料记忆
OUT W30.03  ; #1进料位有料标志
LD TR0
AND 805.09  ; #2来料位有料感应标志[0005.09]
ANDNOT P_On
OUT W31.00  ; #2来料位有料标志
LD TR0
AND 805.11  ; #2隔离位有料感应标志[0005.11]
OUT W31.01  ; #2隔离位有料标志
LD TR0
AND H12.00  ; #2扫码阻挡有料记忆
OUT W31.02  ; #2扫码阻挡有料标志
LD TR0
AND H12.01  ; #2进料位有料记忆
OUT W31.03  ; #2进料位有料标志
LD TR0
BCNTC(621) #1 W30 D90
BIN(023) D90 D92
BCNTC(621) #1 W31 D94
BIN(023) D94 D96
AND=(300) D1059 &0  ; 进料伺服机构步序号
AND<=L(316) D1066 &1  ; #1腔体机构自动步序号
AND<=L(316) D1070 &1  ; #1腔体机构单检步序号
AND<=L(316) D1074 &1  ; #1腔体机构清氦步序号
AND<=L(316) D1096 &1  ; #2腔体机构自动步序号
AND<=L(316) D1100 &1  ; #2腔体机构单检步序号
AND<=L(316) D1104 &1  ; #2腔体机构清氦步序号
AND<=L(316) D1126 &1  ; #3腔体机构自动步序号
AND<=L(316) D1130 &1  ; #3腔体机构单检步序号
AND<=L(316) D1134 &1  ; #3腔体机构清氦步序号
AND<=L(316) D1156 &1  ; 下料模组自动流程
AND<=L(316) D1158 &1  ; 下料模组全NG流程
AND<=L(316) D1160 &1  ; 下料模组（取）放1OK/1NG流程
ANDNOT 200.11  ; 报警中
OUT TR1
LDNOT 805.08  ; #1来料位有料感应标志[0005.08]
ORNOT 805.09  ; #2来料位有料感应标志[0005.09]
ANDLD
LD<>(305) D92 D96
OR=(300) D92 &0
OR=(300) D96 &0
ANDLD
OUT 200.08  ; 设备待料状态（参考进料）
LD TR1
AND 200.09  ; 设备内有电池
AND 806.14  ; #1-1出料位有料感应标志[0006.14]
AND 806.15  ; #1-2出料位有料感应标志[0006.15]
AND 807.00  ; #2-1出料位有料感应标志[0007.00]
AND 807.01  ; #2-2出料位有料感应标志[0007.01]
ANDNOT 805.04  ; 出料对接输入标志[0005.04]
TIMX(550) 0021 &300  ; 设备待料状态延时（参考出料）
LD TR0
ANDNOT 200.11  ; 报警中
AND 200.08  ; 设备待料状态（参考进料）
TIMX(550) 0020 &300  ; 设备待料状态延时（参考进料）

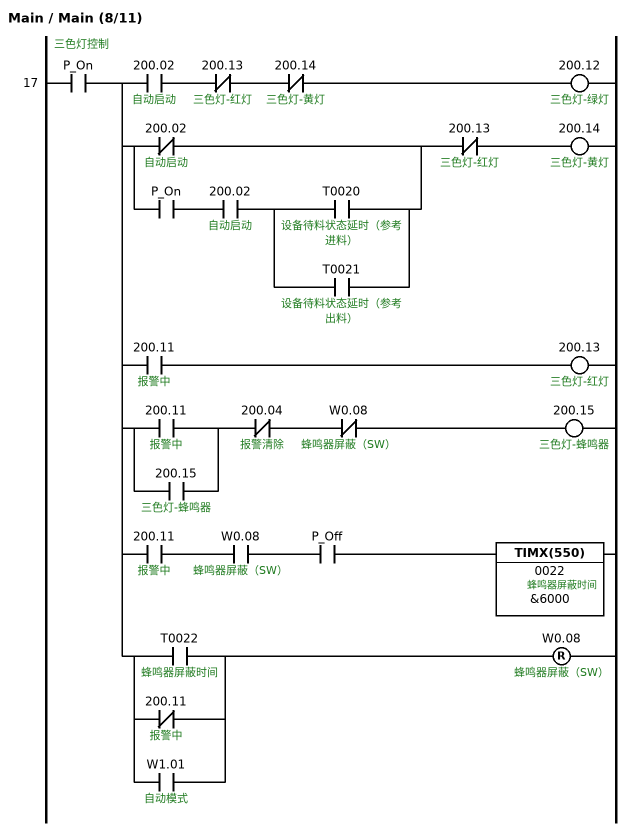
; rung 17: 三色灯控制
LD P_On
OUT TR0
AND 200.02  ; 自动启动
ANDNOT 200.13  ; 三色灯-红灯
ANDNOT 200.14  ; 三色灯-黄灯
OUT 200.12  ; 三色灯-绿灯
LD TR0
LDNOT 200.02  ; 自动启动
LD P_On
AND 200.02  ; 自动启动
LD T0020  ; 设备待料状态延时（参考进料）
OR T0021  ; 设备待料状态延时（参考出料）
ANDLD
ORLD
ANDLD
ANDNOT 200.13  ; 三色灯-红灯
OUT 200.14  ; 三色灯-黄灯
LD TR0
AND 200.11  ; 报警中
OUT 200.13  ; 三色灯-红灯
LD TR0
LD 200.11  ; 报警中
OR 200.15  ; 三色灯-蜂鸣器
ANDLD
ANDNOT 200.04  ; 报警清除
ANDNOT W0.08  ; 蜂鸣器屏蔽（SW）
OUT 200.15  ; 三色灯-蜂鸣器
LD TR0
AND 200.11  ; 报警中
AND W0.08  ; 蜂鸣器屏蔽（SW）
AND P_Off
TIMX(550) 0022 &6000  ; 蜂鸣器屏蔽时间
LD TR0
LD T0022  ; 蜂鸣器屏蔽时间
ORNOT 200.11  ; 报警中
OR W1.01  ; 自动模式
ANDLD
RSET W0.08  ; 蜂鸣器屏蔽（SW）

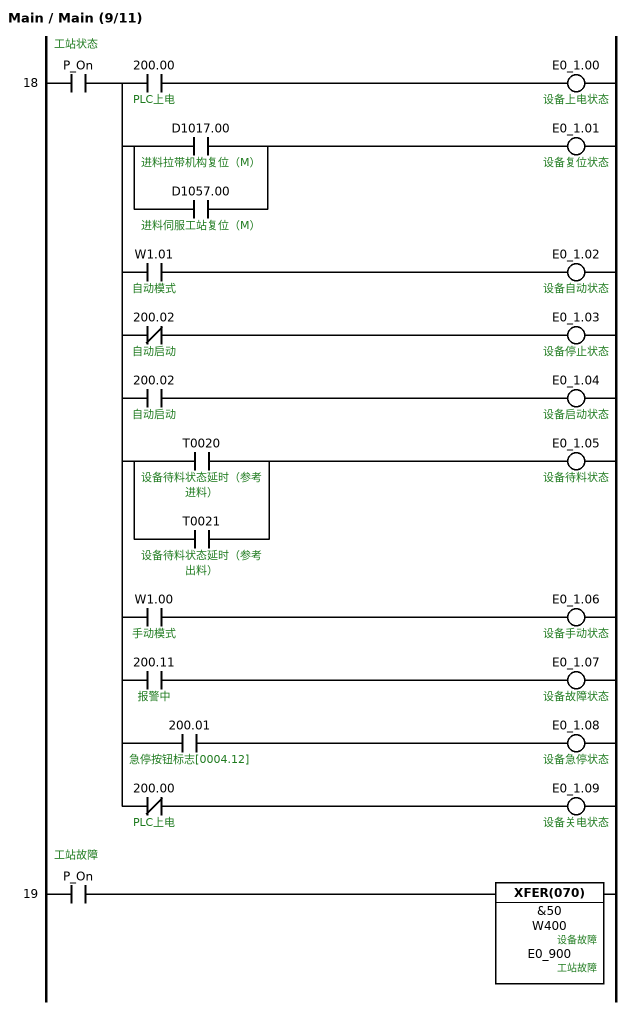
; rung 18: 工站状态
LD P_On
OUT TR0
AND 200.00  ; PLC上电
OUT E0_1.00  ; 设备上电状态
LD TR0
LD D1017.00  ; 进料拉带机构复位（M）
OR D1057.00  ; 进料伺服工站复位（M）
ANDLD
OUT E0_1.01  ; 设备复位状态
LD TR0
AND W1.01  ; 自动模式
OUT E0_1.02  ; 设备自动状态
LD TR0
ANDNOT 200.02  ; 自动启动
OUT E0_1.03  ; 设备停止状态
LD TR0
AND 200.02  ; 自动启动
OUT E0_1.04  ; 设备启动状态
LD TR0
LD T0020  ; 设备待料状态延时（参考进料）
OR T0021  ; 设备待料状态延时（参考出料）
ANDLD
OUT E0_1.05  ; 设备待料状态
LD TR0
AND W1.00  ; 手动模式
OUT E0_1.06  ; 设备手动状态
LD TR0
AND 200.11  ; 报警中
OUT E0_1.07  ; 设备故障状态
LD TR0
AND 200.01  ; 急停按钮标志[0004.12]
OUT E0_1.08  ; 设备急停状态
LD TR0
ANDNOT 200.00  ; PLC上电
OUT E0_1.09  ; 设备关电状态
; rung 19: 工站故障
LD P_On
XFER(070) &50 W400 E0_900  ; 设备故障, 工站故障

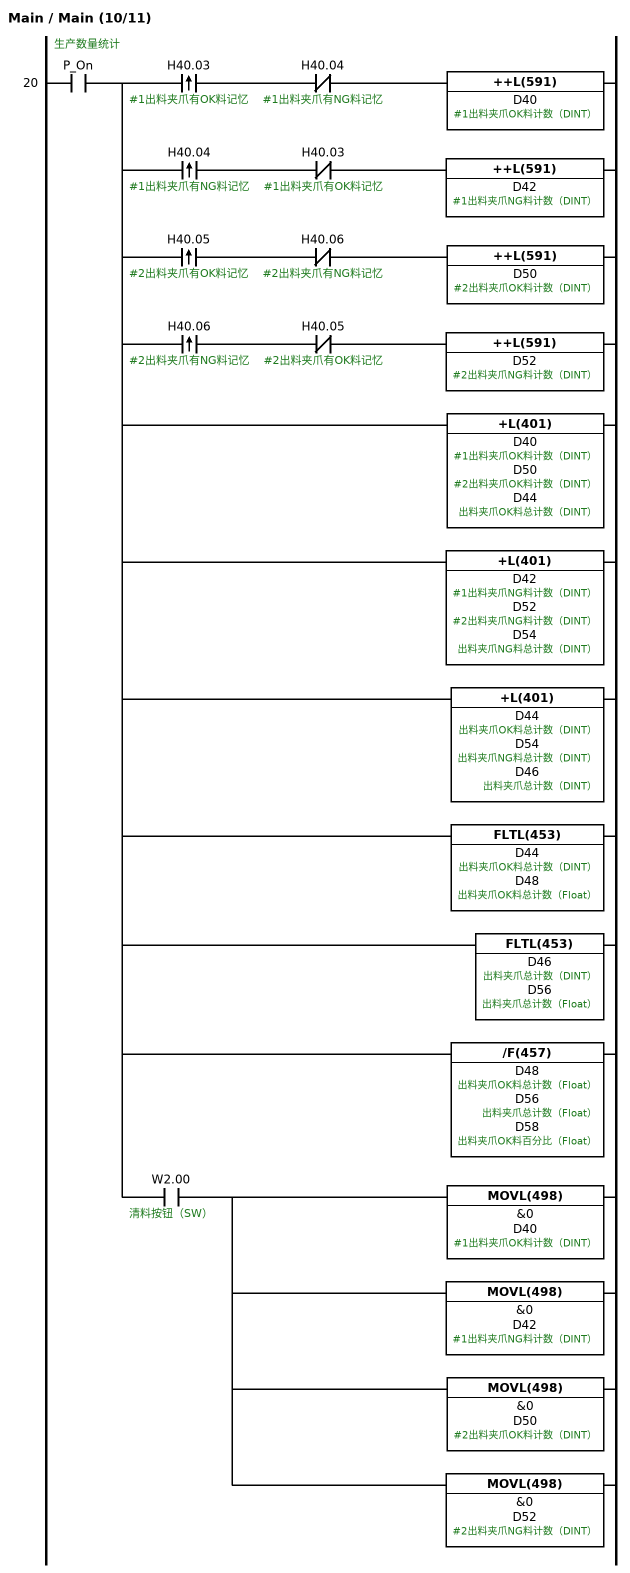
; rung 20: 生产数量统计
LD P_On
OUT TR0
@AND H40.03  ; #1出料夹爪有OK料记忆
ANDNOT H40.04  ; #1出料夹爪有NG料记忆
++L(591) D40  ; #1出料夹爪OK料计数（DINT）
LD TR0
@AND H40.04  ; #1出料夹爪有NG料记忆
ANDNOT H40.03  ; #1出料夹爪有OK料记忆
++L(591) D42  ; #1出料夹爪NG料计数（DINT）
LD TR0
@AND H40.05  ; #2出料夹爪有OK料记忆
ANDNOT H40.06  ; #2出料夹爪有NG料记忆
++L(591) D50  ; #2出料夹爪OK料计数（DINT）
LD TR0
@AND H40.06  ; #2出料夹爪有NG料记忆
ANDNOT H40.05  ; #2出料夹爪有OK料记忆
++L(591) D52  ; #2出料夹爪NG料计数（DINT）
LD TR0
+L(401) D40 D50 D44  ; #1出料夹爪OK料计数（DINT）, #2出料夹爪OK料计数（DINT）, 出料夹爪OK料总计数（DINT）
+L(401) D42 D52 D54  ; #1出料夹爪NG料计数（DINT）, #2出料夹爪NG料计数（DINT）, 出料夹爪NG料总计数（DINT）
+L(401) D44 D54 D46  ; 出料夹爪OK料总计数（DINT）, 出料夹爪NG料总计数（DINT）, 出料夹爪总计数（DINT）
FLTL(453) D44 D48  ; 出料夹爪OK料总计数（DINT）, 出料夹爪OK料总计数（Float）
FLTL(453) D46 D56  ; 出料夹爪总计数（DINT）, 出料夹爪总计数（Float）
/F(457) D48 D56 D58  ; 出料夹爪OK料总计数（Float）, 出料夹爪总计数（Float）, 出料夹爪OK料百分比（Float）
AND W2.00  ; 清料按钮（SW）
MOVL(498) &0 D40  ; #1出料夹爪OK料计数（DINT）
MOVL(498) &0 D42  ; #1出料夹爪NG料计数（DINT）
MOVL(498) &0 D50  ; #2出料夹爪OK料计数（DINT）
MOVL(498) &0 D52  ; #2出料夹爪NG料计数（DINT）

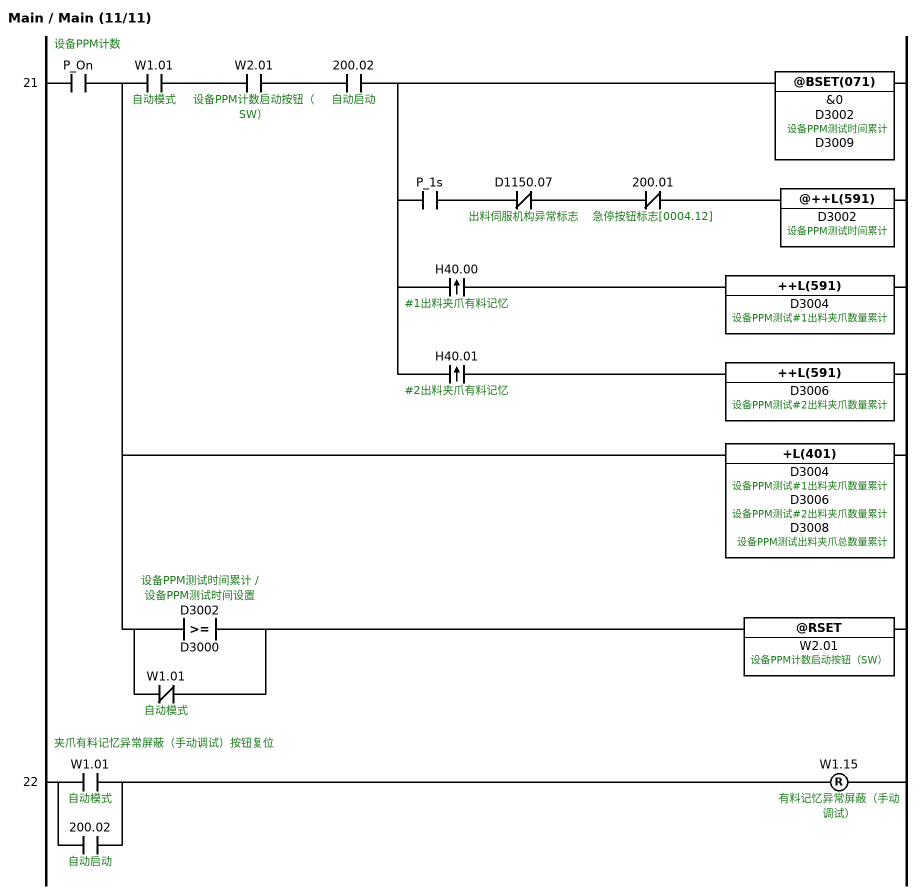
; rung 21: 设备PPM计数
LD P_On
OUT TR0
AND W1.01  ; 自动模式
AND W2.01  ; 设备PPM计数启动按钮（SW）  // HMI《切换开关》按钮
AND 200.02  ; 自动启动
OUT TR1
@BSET(071) &0 D3002 D3009  ; 设备PPM测试时间累计
AND P_1s
ANDNOT D1150.07  ; 出料伺服机构异常标志
ANDNOT 200.01  ; 急停按钮标志[0004.12]
@++L(591) D3002  ; 设备PPM测试时间累计
LD TR1
@AND H40.00  ; #1出料夹爪有料记忆
++L(591) D3004  ; 设备PPM测试#1出料夹爪数量累计
LD TR1
@AND H40.01  ; #2出料夹爪有料记忆
++L(591) D3006  ; 设备PPM测试#2出料夹爪数量累计
LD TR0
+L(401) D3004 D3006 D3008  ; 设备PPM测试#1出料夹爪数量累计, 设备PPM测试#2出料夹爪数量累计, 设备PPM测试出料夹爪总数量累计
LD>=L(326) D3002 D3000  ; 设备PPM测试时间累计, 设备PPM测试时间设置
ORNOT W1.01  ; 自动模式
ANDLD
@RSET W2.01  ; 设备PPM计数启动按钮（SW）
; rung 22: 夹爪有料记忆异常屏蔽（手动调试）按钮复位
LD W1.01  ; 自动模式
OR 200.02  ; 自动启动
RSET W1.15  ; 有料记忆异常屏蔽（手动调试）
; rung 23: 对接信号

### Section 氦检仪通讯

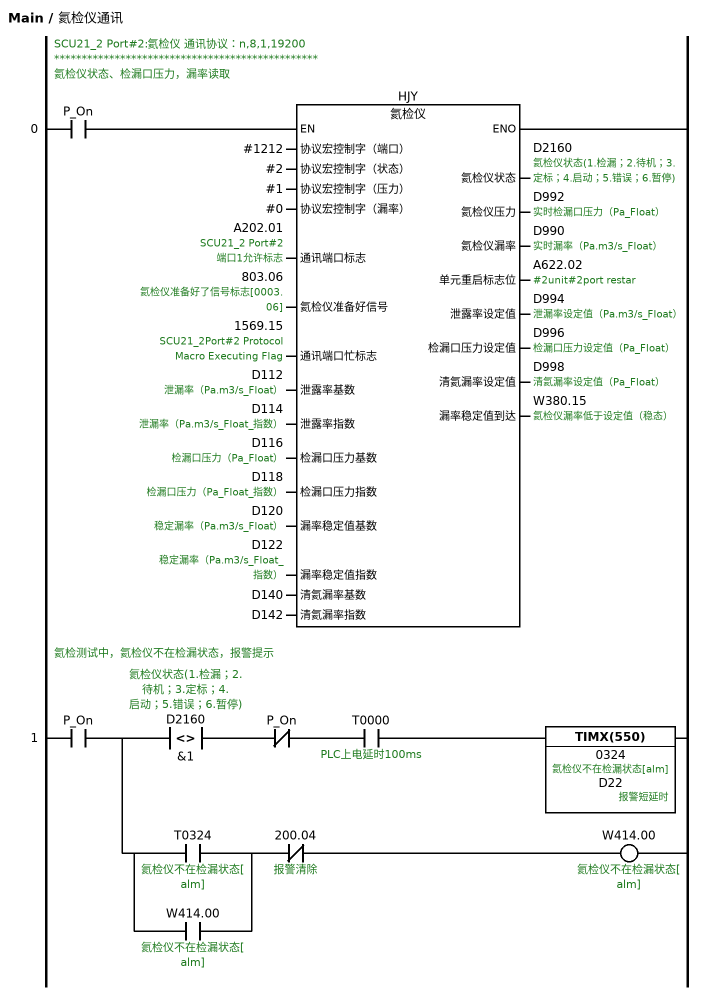
; rung 0: SCU21_2 Port#2:氦检仪 通讯协议：n,8,1,19200 / ************************************************ / 氦检仪状态、检漏口压力，漏率读取
LD P_On
CALL HJY : 氦检仪 (协议宏控制字（端口） := #1212, 协议宏控制字（状态） := #2, 协议宏控制字（压力） := #1, 协议宏控制字（漏率） := #0, 通讯端口标志 := A202.01, 氦检仪准备好信号 := 803.06, 通讯端口忙标志 := 1569.15, 泄露率基数 := D112, 泄露率指数 := D114, 检漏口压力基数 := D116, 检漏口压力指数 := D118, 漏率稳定值基数 := D120, 漏率稳定值指数 := D122, 清氦漏率基数 := D140, 清氦漏率指数 := D142, 氦检仪状态 => D2160, 氦检仪压力 => D992, 氦检仪漏率 => D990, 单元重启标志位 => A622.02, 泄露率设定值 => D994, 检漏口压力设定值 => D996, 清氦漏率设定值 => D998, 漏率稳定值到达 => W380.15)  ; SCU21_2 Port#2 端口1允许标志, 氦检仪准备好了信号标志[0003.06], SCU21_2Port#2 Protocol Macro Executing Flag, 泄漏率（Pa.m3/s_Float）, 泄漏率（Pa.m3/s_Float_指数）, 检漏口压力（Pa_Float）, 检漏口压力（Pa_Float_指数）, 稳定漏率（Pa.m3/s_Float）, 稳定漏率（Pa.m3/s_Float_指数）, 氦检仪状态(1.检漏；2.待机；3.定标；4.启动；5.错误；6.暂停), 实时检漏口压力（Pa_Float）, 实时漏率（Pa.m3/s_Float）, #2unit#2port restar, 泄漏率设定值（Pa.m3/s_Float）, 检漏口压力设定值（Pa_Float）, 清氦漏率设定值（Pa_Float）, 氦检仪漏率低于设定值（稳态）
; rung 1: 氦检测试中，氦检仪不在检漏状态，报警提示
LD P_On
OUT TR0
AND<>(305) D2160 &1  ; 氦检仪状态(1.检漏；2.待机；3.定标；4.启动；5.错误；6.暂停)
ANDNOT P_On  // 各腔体氦检步DXXXX.00=1
AND T0000  ; PLC上电延时100ms
TIMX(550) 0324 D22  ; 报警短延时, 氦检仪不在检漏状态[alm]
LD TR0
LD T0324  ; 氦检仪不在检漏状态[alm]
OR W414.00  ; 氦检仪不在检漏状态[alm]
ANDLD
ANDNOT 200.04  ; 报警清除
OUT W414.00  ; 氦检仪不在检漏状态[alm]

### Section 入料扫码通讯

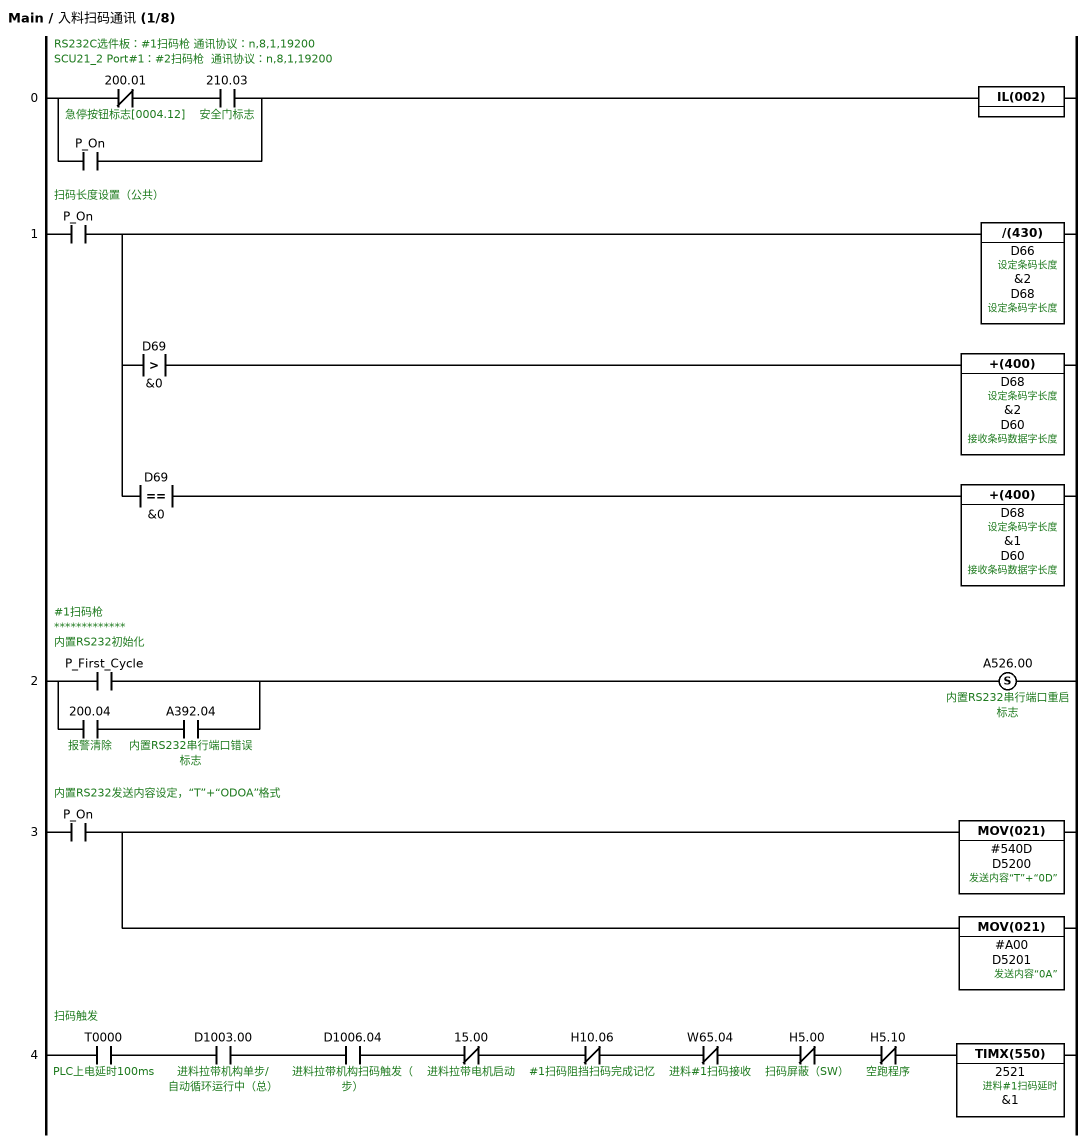
; rung 0: RS232C选件板：#1扫码枪 通讯协议：n,8,1,19200 / SCU21_2 Port#1：#2扫码枪  通讯协议：n,8,1,19200
LDNOT 200.01  ; 急停按钮标志[0004.12]
AND 210.03  ; 安全门标志
OR P_On
IL(002)
; rung 1: 扫码长度设置（公共）
LD P_On
OUT TR0
/(430) D66 &2 D68  ; 设定条码长度, 设定条码字长度
AND>(320) D69 &0
+(400) D68 &2 D60  ; 设定条码字长度, 接收条码数据字长度
LD TR0
AND=(300) D69 &0
+(400) D68 &1 D60  ; 设定条码字长度, 接收条码数据字长度
; rung 2: #1扫码枪 / ************* / 内置RS232初始化
LD P_First_Cycle
LD 200.04  ; 报警清除
AND A392.04  ; 内置RS232串行端口错误标志
ORLD
SET A526.00  ; 内置RS232串行端口重启标志
; rung 3: 内置RS232发送内容设定，“T”+“ODOA”格式
LD P_On
MOV(021) #540D D5200  ; 发送内容“T”+“0D”
MOV(021) #A00 D5201  ; 发送内容“0A”
; rung 4: 扫码触发
LD T0000  ; PLC上电延时100ms
AND D1003.00  ; 进料拉带机构单步/自动循环运行中（总）
AND D1006.04  ; 进料拉带机构扫码触发（步）
ANDNOT 15.00  ; 进料拉带电机启动
ANDNOT H10.06  ; #1扫码阻挡扫码完成记忆
ANDNOT W65.04  ; 进料#1扫码接收
ANDNOT H5.00  ; 扫码屏蔽（SW）
ANDNOT H5.10  ; 空跑程序
TIMX(550) 2521 &1  ; 进料#1扫码延时

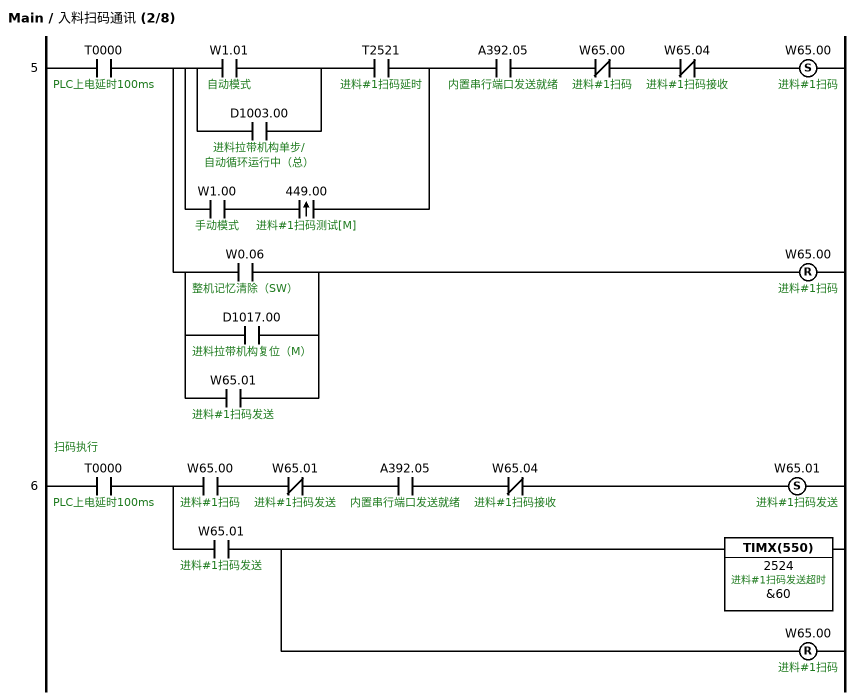
; rung 5
LD T0000  ; PLC上电延时100ms
OUT TR0
LD W1.01  ; 自动模式
OR D1003.00  ; 进料拉带机构单步/自动循环运行中（总）
AND T2521  ; 进料#1扫码延时
LD W1.00  ; 手动模式
@AND 449.00  ; 进料#1扫码测试[M]
ORLD
ANDLD
AND A392.05  ; 内置串行端口发送就绪
ANDNOT W65.00  ; 进料#1扫码
ANDNOT W65.04  ; 进料#1扫码接收
SET W65.00  ; 进料#1扫码
LD TR0
LD W0.06  ; 整机记忆清除（SW）
OR D1017.00  ; 进料拉带机构复位（M）
OR W65.01  ; 进料#1扫码发送
ANDLD
RSET W65.00  ; 进料#1扫码
; rung 6: 扫码执行
LD T0000  ; PLC上电延时100ms
OUT TR0
AND W65.00  ; 进料#1扫码
ANDNOT W65.01  ; 进料#1扫码发送
AND A392.05  ; 内置串行端口发送就绪
ANDNOT W65.04  ; 进料#1扫码接收
SET W65.01  ; 进料#1扫码发送
LD TR0
AND W65.01  ; 进料#1扫码发送
TIMX(550) 2524 &60  ; 进料#1扫码发送超时
RSET W65.00  ; 进料#1扫码

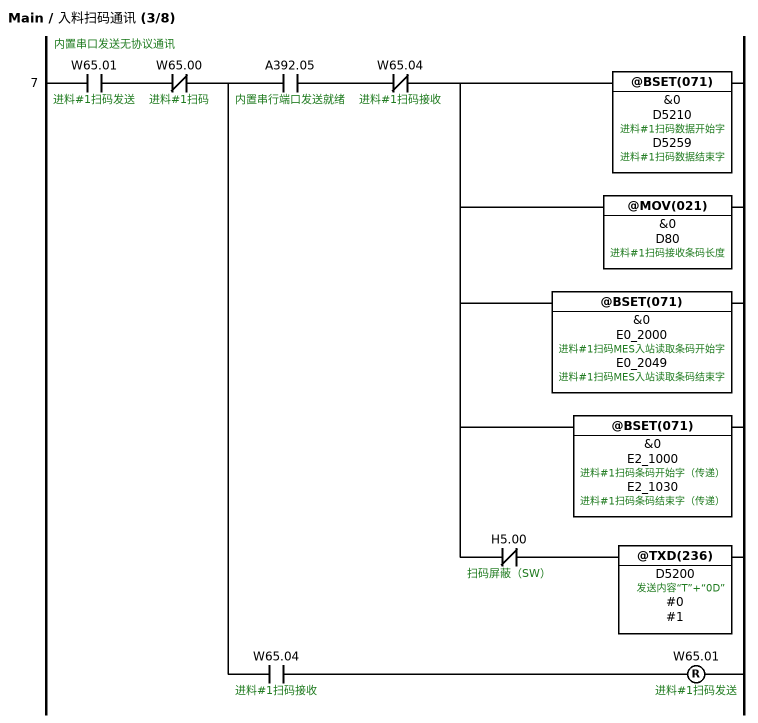
; rung 7: 内置串口发送无协议通讯
LD W65.01  ; 进料#1扫码发送
ANDNOT W65.00  ; 进料#1扫码
OUT TR0
AND A392.05  ; 内置串行端口发送就绪
ANDNOT W65.04  ; 进料#1扫码接收
@BSET(071) &0 D5210 D5259  ; 进料#1扫码数据开始字, 进料#1扫码数据结束字
@MOV(021) &0 D80  ; 进料#1扫码接收条码长度
@BSET(071) &0 E0_2000 E0_2049  ; 进料#1扫码MES入站读取条码开始字, 进料#1扫码MES入站读取条码结束字
@BSET(071) &0 E2_1000 E2_1030  ; 进料#1扫码条码开始字（传递）, 进料#1扫码条码结束字（传递）
ANDNOT H5.00  ; 扫码屏蔽（SW）
@TXD(236) D5200 #0 #1  ; 发送内容“T”+“0D”
LD TR0
AND W65.04  ; 进料#1扫码接收
RSET W65.01  ; 进料#1扫码发送

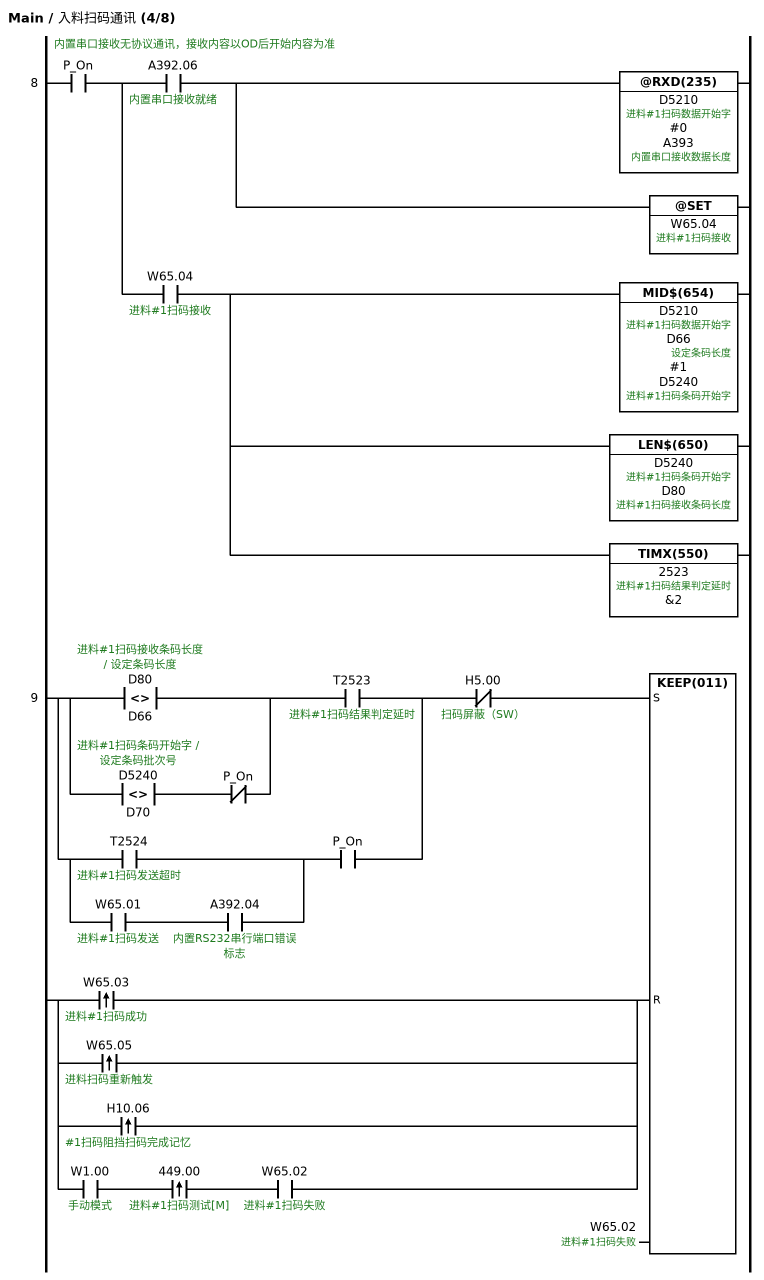
; rung 8: 内置串口接收无协议通讯，接收内容以OD后开始内容为准
LD P_On
OUT TR0
AND A392.06  ; 内置串口接收就绪
@RXD(235) D5210 #0 A393  ; 进料#1扫码数据开始字, 内置串口接收数据长度
@SET W65.04  ; 进料#1扫码接收
LD TR0
AND W65.04  ; 进料#1扫码接收
MID$(654) D5210 D66 #1 D5240  ; 进料#1扫码数据开始字, 设定条码长度, 进料#1扫码条码开始字
LEN$(650) D5240 D80  ; 进料#1扫码条码开始字, 进料#1扫码接收条码长度
TIMX(550) 2523 &2  ; 进料#1扫码结果判定延时
; rung 9
LD<>(305) D80 D66  ; 进料#1扫码接收条码长度, 设定条码长度
LD<>$(671) D5240 D70  ; 进料#1扫码条码开始字, 设定条码批次号
ANDNOT P_On
ORLD
AND T2523  ; 进料#1扫码结果判定延时
LD T2524  ; 进料#1扫码发送超时
LD W65.01  ; 进料#1扫码发送
AND A392.04  ; 内置RS232串行端口错误标志
ORLD
AND P_On
ORLD
ANDNOT H5.00  ; 扫码屏蔽（SW）
@LD W65.03  ; 进料#1扫码成功
@OR W65.05  ; 进料扫码重新触发
@OR H10.06  ; #1扫码阻挡扫码完成记忆
LD W1.00  ; 手动模式
@AND 449.00  ; 进料#1扫码测试[M]
AND W65.02  ; 进料#1扫码失败
ORLD
KEEP(011) W65.02  ; 进料#1扫码失败

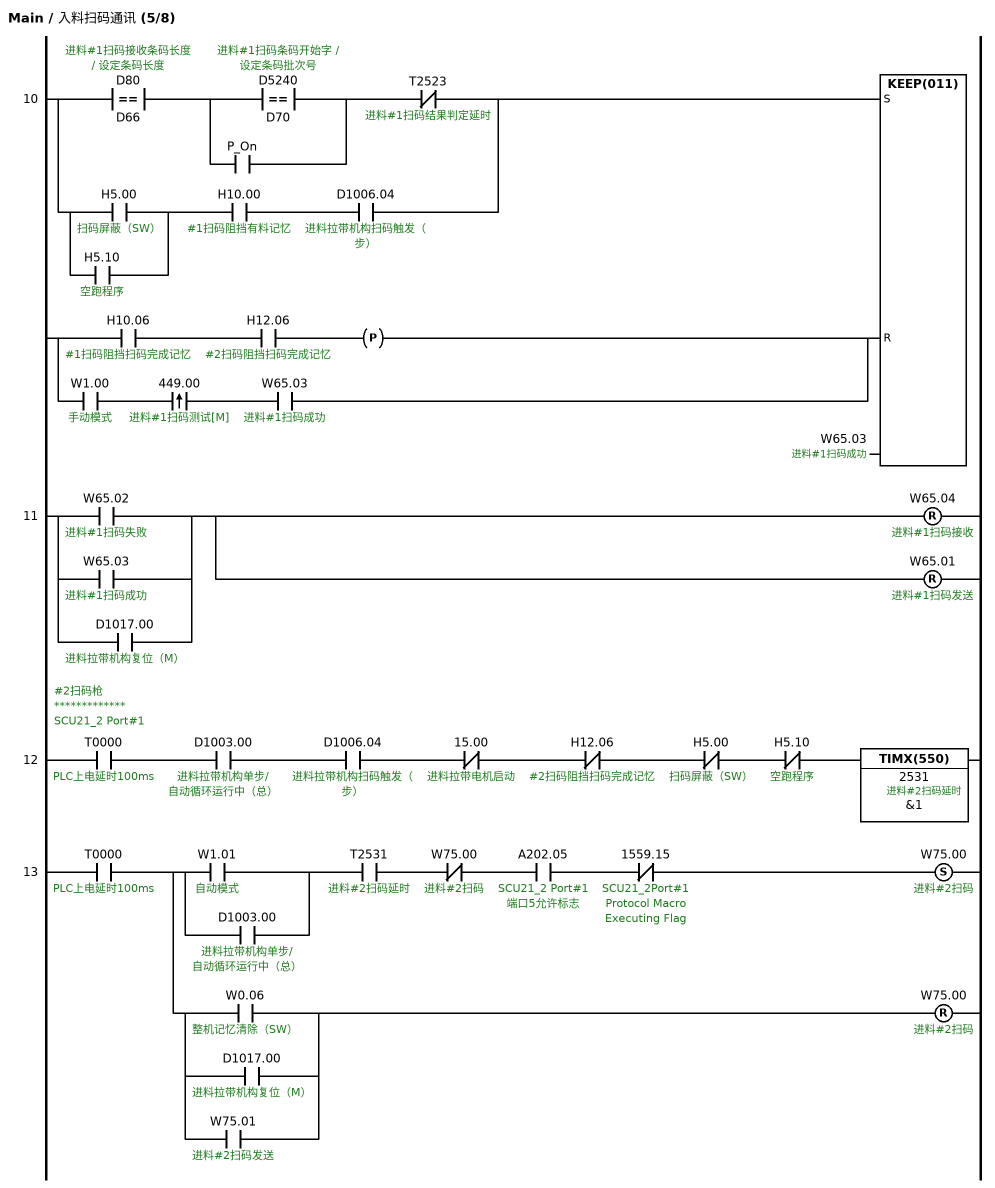
; rung 10
LD=(300) D80 D66  ; 进料#1扫码接收条码长度, 设定条码长度
LD=$(670) D5240 D70  ; 进料#1扫码条码开始字, 设定条码批次号
OR P_On
ANDLD
ANDNOT T2523  ; 进料#1扫码结果判定延时
LD H5.00  ; 扫码屏蔽（SW）
OR H5.10  ; 空跑程序
AND H10.00  ; #1扫码阻挡有料记忆
AND D1006.04  ; 进料拉带机构扫码触发（步）
ORLD
LD H10.06  ; #1扫码阻挡扫码完成记忆
AND H12.06  ; #2扫码阻挡扫码完成记忆
UP(521)
LD W1.00  ; 手动模式
@AND 449.00  ; 进料#1扫码测试[M]
AND W65.03  ; 进料#1扫码成功
ORLD
KEEP(011) W65.03  ; 进料#1扫码成功
; rung 11
LD W65.02  ; 进料#1扫码失败
OR W65.03  ; 进料#1扫码成功
OR D1017.00  ; 进料拉带机构复位（M）
RSET W65.04  ; 进料#1扫码接收
RSET W65.01  ; 进料#1扫码发送
; rung 12: #2扫码枪 / ************* / SCU21_2 Port#1
LD T0000  ; PLC上电延时100ms
AND D1003.00  ; 进料拉带机构单步/自动循环运行中（总）
AND D1006.04  ; 进料拉带机构扫码触发（步）
ANDNOT 15.00  ; 进料拉带电机启动
ANDNOT H12.06  ; #2扫码阻挡扫码完成记忆
ANDNOT H5.00  ; 扫码屏蔽（SW）
ANDNOT H5.10  ; 空跑程序
TIMX(550) 2531 &1  ; 进料#2扫码延时
; rung 13
LD T0000  ; PLC上电延时100ms
OUT TR0
LD W1.01  ; 自动模式
OR D1003.00  ; 进料拉带机构单步/自动循环运行中（总）
ANDLD
AND T2531  ; 进料#2扫码延时
ANDNOT W75.00  ; 进料#2扫码
AND A202.05  ; SCU21_2 Port#1 端口5允许标志
ANDNOT 1559.15  ; SCU21_2Port#1 Protocol Macro Executing Flag
SET W75.00  ; 进料#2扫码
LD TR0
LD W0.06  ; 整机记忆清除（SW）
OR D1017.00  ; 进料拉带机构复位（M）
OR W75.01  ; 进料#2扫码发送
ANDLD
RSET W75.00  ; 进料#2扫码

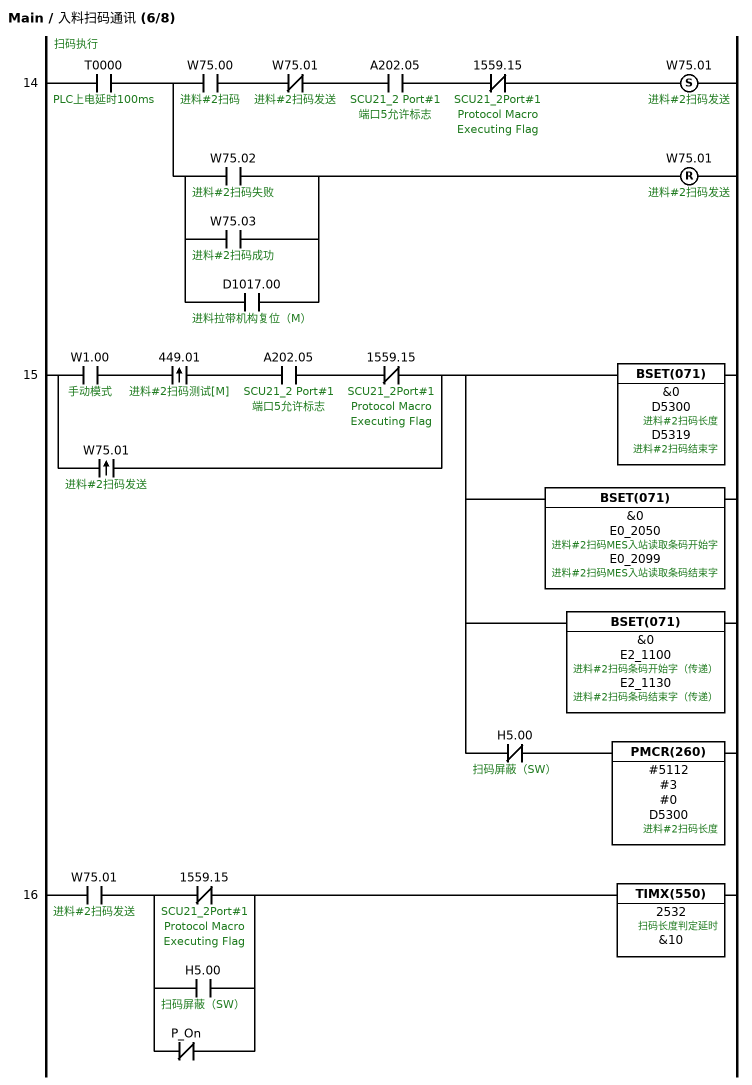
; rung 14: 扫码执行
LD T0000  ; PLC上电延时100ms
OUT TR0
AND W75.00  ; 进料#2扫码
ANDNOT W75.01  ; 进料#2扫码发送
AND A202.05  ; SCU21_2 Port#1 端口5允许标志
ANDNOT 1559.15  ; SCU21_2Port#1 Protocol Macro Executing Flag
SET W75.01  ; 进料#2扫码发送
LD TR0
LD W75.02  ; 进料#2扫码失败
OR W75.03  ; 进料#2扫码成功
OR D1017.00  ; 进料拉带机构复位（M）
ANDLD
RSET W75.01  ; 进料#2扫码发送
; rung 15
LD W1.00  ; 手动模式
@AND 449.01  ; 进料#2扫码测试[M]
AND A202.05  ; SCU21_2 Port#1 端口5允许标志
ANDNOT 1559.15  ; SCU21_2Port#1 Protocol Macro Executing Flag
@OR W75.01  ; 进料#2扫码发送
BSET(071) &0 D5300 D5319  ; 进料#2扫码长度, 进料#2扫码结束字
BSET(071) &0 E0_2050 E0_2099  ; 进料#2扫码MES入站读取条码开始字, 进料#2扫码MES入站读取条码结束字
BSET(071) &0 E2_1100 E2_1130  ; 进料#2扫码条码开始字（传递）, 进料#2扫码条码结束字（传递）
ANDNOT H5.00  ; 扫码屏蔽（SW）
PMCR(260) #5112 #3 #0 D5300  ; 进料#2扫码长度
; rung 16
LD W75.01  ; 进料#2扫码发送
LDNOT 1559.15  ; SCU21_2Port#1 Protocol Macro Executing Flag
OR H5.00  ; 扫码屏蔽（SW）
ORNOT P_On
ANDLD
TIMX(550) 2532 &10  ; 扫码长度判定延时

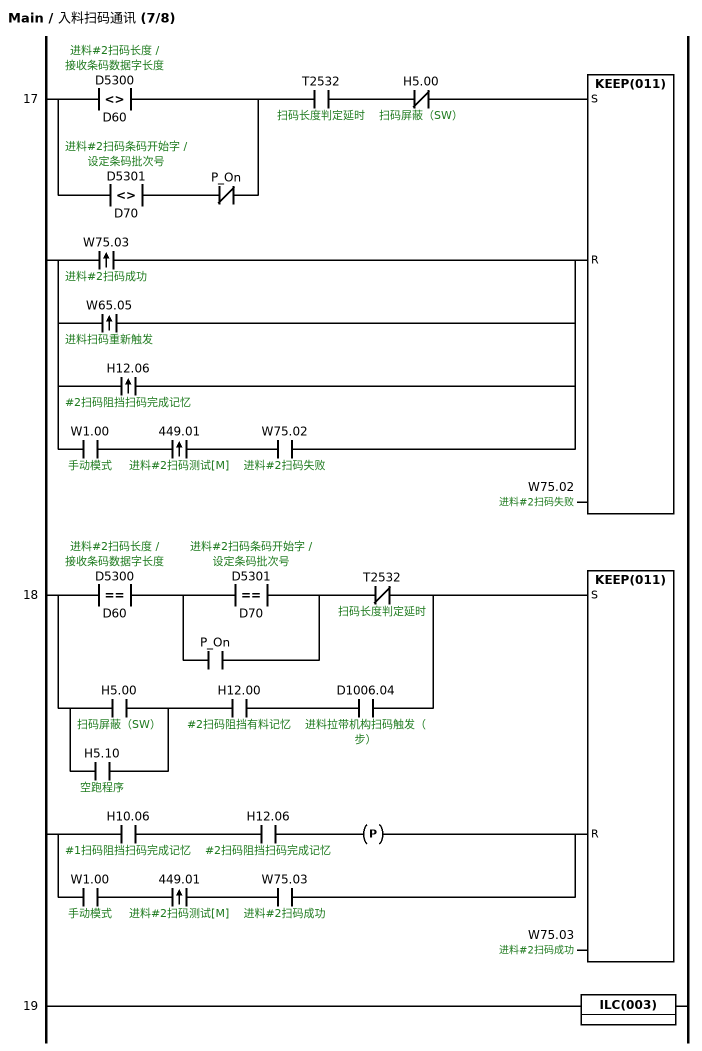
; rung 17
LD<>(305) D5300 D60  ; 进料#2扫码长度, 接收条码数据字长度
LD<>$(671) D5301 D70  ; 进料#2扫码条码开始字, 设定条码批次号
ANDNOT P_On
ORLD
AND T2532  ; 扫码长度判定延时
ANDNOT H5.00  ; 扫码屏蔽（SW）
@LD W75.03  ; 进料#2扫码成功
@OR W65.05  ; 进料扫码重新触发
@OR H12.06  ; #2扫码阻挡扫码完成记忆
LD W1.00  ; 手动模式
@AND 449.01  ; 进料#2扫码测试[M]
AND W75.02  ; 进料#2扫码失败
ORLD
KEEP(011) W75.02  ; 进料#2扫码失败
; rung 18
LD=(300) D5300 D60  ; 进料#2扫码长度, 接收条码数据字长度
LD=$(670) D5301 D70  ; 进料#2扫码条码开始字, 设定条码批次号
OR P_On
ANDLD
ANDNOT T2532  ; 扫码长度判定延时
LD H5.00  ; 扫码屏蔽（SW）
OR H5.10  ; 空跑程序
AND H12.00  ; #2扫码阻挡有料记忆
AND D1006.04  ; 进料拉带机构扫码触发（步）
ORLD
LD H10.06  ; #1扫码阻挡扫码完成记忆
AND H12.06  ; #2扫码阻挡扫码完成记忆
UP(521)
LD W1.00  ; 手动模式
@AND 449.01  ; 进料#2扫码测试[M]
AND W75.03  ; 进料#2扫码成功
ORLD
KEEP(011) W75.03  ; 进料#2扫码成功
; rung 19
ILC(003)

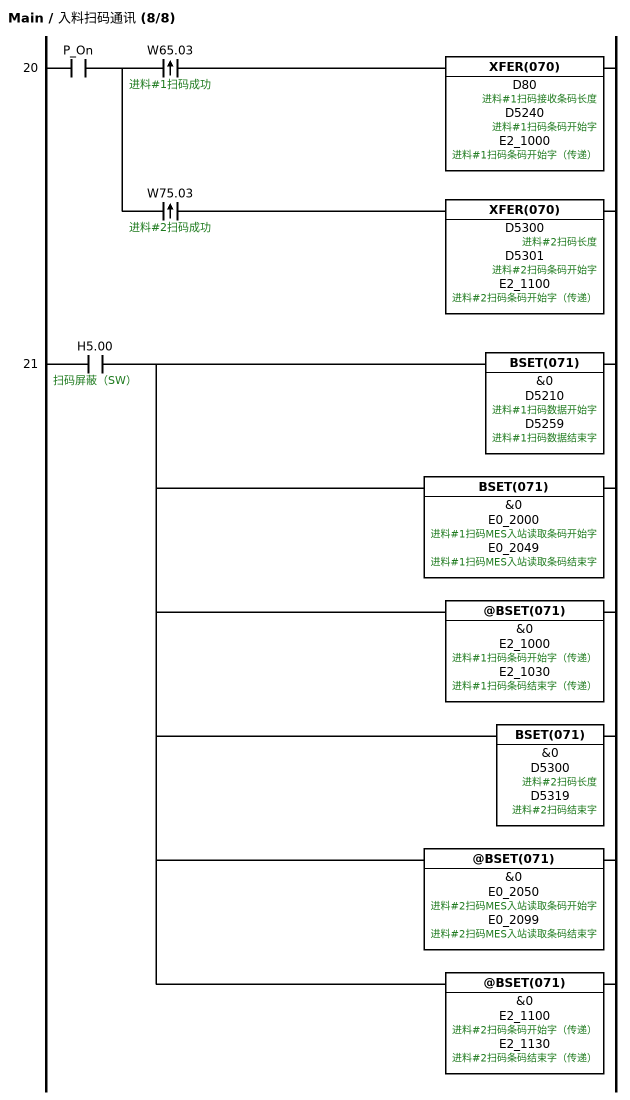
; rung 20
LD P_On
OUT TR0
@AND W65.03  ; 进料#1扫码成功
XFER(070) D80 D5240 E2_1000  ; 进料#1扫码接收条码长度, 进料#1扫码条码开始字, 进料#1扫码条码开始字（传递）
LD TR0
@AND W75.03  ; 进料#2扫码成功
XFER(070) D5300 D5301 E2_1100  ; 进料#2扫码长度, 进料#2扫码条码开始字, 进料#2扫码条码开始字（传递）
; rung 21
LD H5.00  ; 扫码屏蔽（SW）
BSET(071) &0 D5210 D5259  ; 进料#1扫码数据开始字, 进料#1扫码数据结束字
BSET(071) &0 E0_2000 E0_2049  ; 进料#1扫码MES入站读取条码开始字, 进料#1扫码MES入站读取条码结束字
@BSET(071) &0 E2_1000 E2_1030  ; 进料#1扫码条码开始字（传递）, 进料#1扫码条码结束字（传递）
BSET(071) &0 D5300 D5319  ; 进料#2扫码长度, 进料#2扫码结束字
@BSET(071) &0 E0_2050 E0_2099  ; 进料#2扫码MES入站读取条码开始字, 进料#2扫码MES入站读取条码结束字
@BSET(071) &0 E2_1100 E2_1130  ; 进料#2扫码条码开始字（传递）, 进料#2扫码条码结束字（传递）

### Section 真空计算

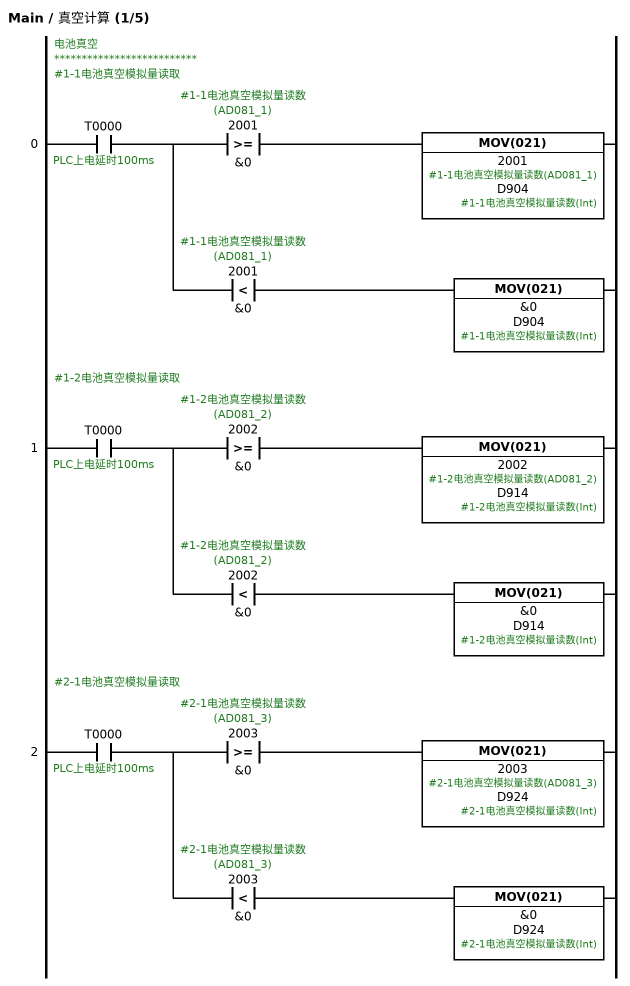
; rung 0: 电池真空 / ************************** / #1-1电池真空模拟量读取
LD T0000  ; PLC上电延时100ms
OUT TR0
AND>=S(327) 2001 &0  ; #1-1电池真空模拟量读数(AD081_1)
MOV(021) 2001 D904  ; #1-1电池真空模拟量读数(AD081_1), #1-1电池真空模拟量读数(Int)
LD TR0
AND<S(312) 2001 &0  ; #1-1电池真空模拟量读数(AD081_1)
MOV(021) &0 D904  ; #1-1电池真空模拟量读数(Int)
; rung 1: #1-2电池真空模拟量读取
LD T0000  ; PLC上电延时100ms
OUT TR0
AND>=S(327) 2002 &0  ; #1-2电池真空模拟量读数(AD081_2)
MOV(021) 2002 D914  ; #1-2电池真空模拟量读数(AD081_2), #1-2电池真空模拟量读数(Int)
LD TR0
AND<S(312) 2002 &0  ; #1-2电池真空模拟量读数(AD081_2)
MOV(021) &0 D914  ; #1-2电池真空模拟量读数(Int)
; rung 2: #2-1电池真空模拟量读取
LD T0000  ; PLC上电延时100ms
OUT TR0
AND>=S(327) 2003 &0  ; #2-1电池真空模拟量读数(AD081_3)
MOV(021) 2003 D924  ; #2-1电池真空模拟量读数(AD081_3), #2-1电池真空模拟量读数(Int)
LD TR0
AND<S(312) 2003 &0  ; #2-1电池真空模拟量读数(AD081_3)
MOV(021) &0 D924  ; #2-1电池真空模拟量读数(Int)

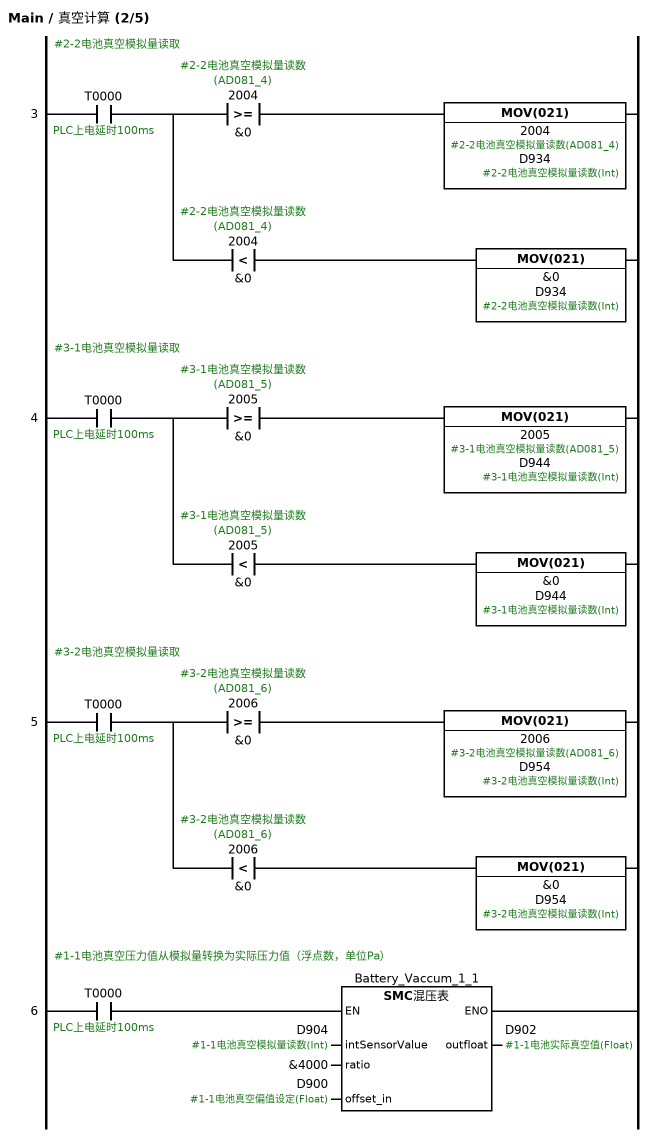
; rung 3: #2-2电池真空模拟量读取
LD T0000  ; PLC上电延时100ms
OUT TR0
AND>=S(327) 2004 &0  ; #2-2电池真空模拟量读数(AD081_4)
MOV(021) 2004 D934  ; #2-2电池真空模拟量读数(AD081_4), #2-2电池真空模拟量读数(Int)
LD TR0
AND<S(312) 2004 &0  ; #2-2电池真空模拟量读数(AD081_4)
MOV(021) &0 D934  ; #2-2电池真空模拟量读数(Int)
; rung 4: #3-1电池真空模拟量读取
LD T0000  ; PLC上电延时100ms
OUT TR0
AND>=S(327) 2005 &0  ; #3-1电池真空模拟量读数(AD081_5)
MOV(021) 2005 D944  ; #3-1电池真空模拟量读数(AD081_5), #3-1电池真空模拟量读数(Int)
LD TR0
AND<S(312) 2005 &0  ; #3-1电池真空模拟量读数(AD081_5)
MOV(021) &0 D944  ; #3-1电池真空模拟量读数(Int)
; rung 5: #3-2电池真空模拟量读取
LD T0000  ; PLC上电延时100ms
OUT TR0
AND>=S(327) 2006 &0  ; #3-2电池真空模拟量读数(AD081_6)
MOV(021) 2006 D954  ; #3-2电池真空模拟量读数(AD081_6), #3-2电池真空模拟量读数(Int)
LD TR0
AND<S(312) 2006 &0  ; #3-2电池真空模拟量读数(AD081_6)
MOV(021) &0 D954  ; #3-2电池真空模拟量读数(Int)
; rung 6: #1-1电池真空压力值从模拟量转换为实际压力值（浮点数，单位Pa）
LD T0000  ; PLC上电延时100ms
CALL Battery_Vaccum_1_1 : SMC混压表 (intSensorValue := D904, ratio := &4000, offset_in := D900, outfloat => D902)  ; #1-1电池真空模拟量读数(Int), #1-1电池真空偏值设定(Float), #1-1电池实际真空值(Float)

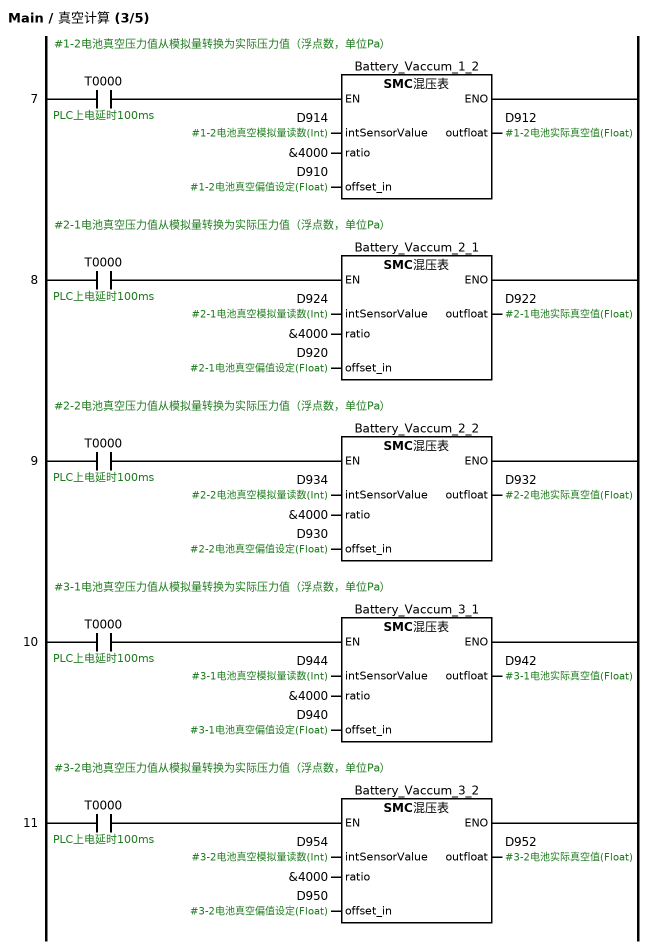
; rung 7: #1-2电池真空压力值从模拟量转换为实际压力值（浮点数，单位Pa）
LD T0000  ; PLC上电延时100ms
CALL Battery_Vaccum_1_2 : SMC混压表 (intSensorValue := D914, ratio := &4000, offset_in := D910, outfloat => D912)  ; #1-2电池真空模拟量读数(Int), #1-2电池真空偏值设定(Float), #1-2电池实际真空值(Float)
; rung 8: #2-1电池真空压力值从模拟量转换为实际压力值（浮点数，单位Pa）
LD T0000  ; PLC上电延时100ms
CALL Battery_Vaccum_2_1 : SMC混压表 (intSensorValue := D924, ratio := &4000, offset_in := D920, outfloat => D922)  ; #2-1电池真空模拟量读数(Int), #2-1电池真空偏值设定(Float), #2-1电池实际真空值(Float)
; rung 9: #2-2电池真空压力值从模拟量转换为实际压力值（浮点数，单位Pa）
LD T0000  ; PLC上电延时100ms
CALL Battery_Vaccum_2_2 : SMC混压表 (intSensorValue := D934, ratio := &4000, offset_in := D930, outfloat => D932)  ; #2-2电池真空模拟量读数(Int), #2-2电池真空偏值设定(Float), #2-2电池实际真空值(Float)
; rung 10: #3-1电池真空压力值从模拟量转换为实际压力值（浮点数，单位Pa）
LD T0000  ; PLC上电延时100ms
CALL Battery_Vaccum_3_1 : SMC混压表 (intSensorValue := D944, ratio := &4000, offset_in := D940, outfloat => D942)  ; #3-1电池真空模拟量读数(Int), #3-1电池真空偏值设定(Float), #3-1电池实际真空值(Float)
; rung 11: #3-2电池真空压力值从模拟量转换为实际压力值（浮点数，单位Pa）
LD T0000  ; PLC上电延时100ms
CALL Battery_Vaccum_3_2 : SMC混压表 (intSensorValue := D954, ratio := &4000, offset_in := D950, outfloat => D952)  ; #3-2电池真空模拟量读数(Int), #3-2电池真空偏值设定(Float), #3-2电池实际真空值(Float)

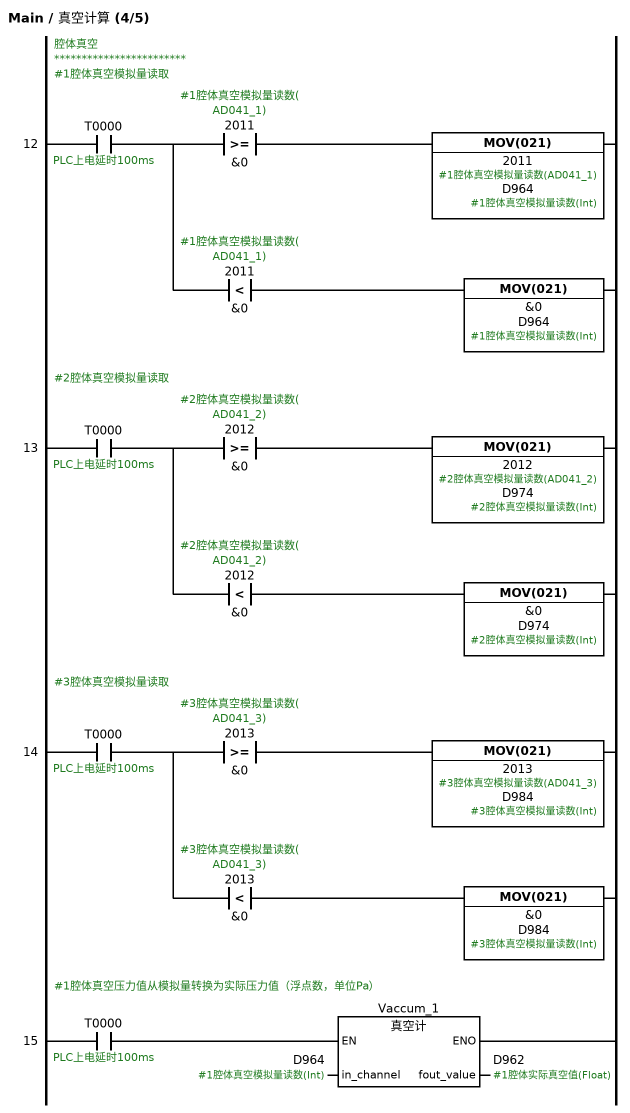
; rung 12: 腔体真空 / ************************ / #1腔体真空模拟量读取
LD T0000  ; PLC上电延时100ms
OUT TR0
AND>=S(327) 2011 &0  ; #1腔体真空模拟量读数(AD041_1)
MOV(021) 2011 D964  ; #1腔体真空模拟量读数(AD041_1), #1腔体真空模拟量读数(Int)
LD TR0
AND<S(312) 2011 &0  ; #1腔体真空模拟量读数(AD041_1)
MOV(021) &0 D964  ; #1腔体真空模拟量读数(Int)
; rung 13: #2腔体真空模拟量读取
LD T0000  ; PLC上电延时100ms
OUT TR0
AND>=S(327) 2012 &0  ; #2腔体真空模拟量读数(AD041_2)
MOV(021) 2012 D974  ; #2腔体真空模拟量读数(AD041_2), #2腔体真空模拟量读数(Int)
LD TR0
AND<S(312) 2012 &0  ; #2腔体真空模拟量读数(AD041_2)
MOV(021) &0 D974  ; #2腔体真空模拟量读数(Int)
; rung 14: #3腔体真空模拟量读取
LD T0000  ; PLC上电延时100ms
OUT TR0
AND>=S(327) 2013 &0  ; #3腔体真空模拟量读数(AD041_3)
MOV(021) 2013 D984  ; #3腔体真空模拟量读数(AD041_3), #3腔体真空模拟量读数(Int)
LD TR0
AND<S(312) 2013 &0  ; #3腔体真空模拟量读数(AD041_3)
MOV(021) &0 D984  ; #3腔体真空模拟量读数(Int)
; rung 15: #1腔体真空压力值从模拟量转换为实际压力值（浮点数，单位Pa）
LD T0000  ; PLC上电延时100ms
CALL Vaccum_1 : 真空计 (in_channel := D964, fout_value => D962)  ; #1腔体真空模拟量读数(Int), #1腔体实际真空值(Float)

